// TIA Portal V17 export
// export: Created 2025-05-22T06:00:37.3823488Z, ExportSetting WithDefaults, DisplayName Totally Integrated Automation Portal, DisplayVersion V17 Update 8, DisplayName TIA Portal Openness, DisplayVersion V17 Update 8, DisplayName TIA Portal Version Control Interface, DisplayVersion V17, DisplayName SINAMICS Startdrive Advanced, DisplayVersion V17 SP2, DisplayName SINAMICS Startdrive G110M, G120, G120C, G120D, G120P, G115D, DisplayVersion V17 SP2, DisplayName SINAMICS Startdrive G130, G150, S120, S150, SINAMICS MV, S210, DisplayVersion V17 SP2, DisplayName STEP 7 Professional, DisplayVersion V17 Update 8, DisplayName SINUMERIK ONE STEP 7 Toolbox, DisplayVersion V17 Update 12, DisplayName SINUMERIK ONE PLC Basic Program Plus, DisplayVersion V17 Update 12, DisplayName SINUMERIK 840D sl STEP 7 Toolbox, DisplayVersion V17 Update 12, DisplayName STEP 7 Safety, DisplayVersion V17 Update 6, DisplayName WinCC Advanced, DisplayVersion V17 Update 8
FUNCTION "FC16011_METHOD_CALLS_U1_STA3_MEAS" : Void   // FC16011, LAD
{ S7_Optimized_Access := 'FALSE' }
VERSION : 0.1
// STATUS VALUES:
// 0 = IDLE
// 1 = CALIBRATING
// 2 = ANALYZING DISTANCE
// 3 = ANALYZING LAYER THICKNESS
// -1 = ERROR
// stored: AutoNumber false, IsIECCheckEnabled false, SetENOAutomatically false, UDAEnableTagReadback false
   VAR_TEMP
      AUX_WSTRING_PART_ID_STA3 : WString;
      AUX_WCHARS : Array[0..63] of WChar;
      index : Int;
      ALARM_AUX : Bool;
      STATUS_BLKMOV : Int;   // STATUS BLKMOV
      ZERO : Int;
   END_VAR
   VAR CONSTANT
      VERSIONS_MAJOR : UInt := 2;
      VERSIONS_MINOR : UInt;
      FC_NUMBER : DInt := 16011;
   END_VAR
   VAR_TEMP   // added for the SCL form of the ladder/FBD networks
      _w1 : Bool;
      _w2 : Bool;
      _w3 : Bool;
      _s5time1 : S5Time;
      _w4 : Bool;
   END_VAR
BEGIN

REGION Network 1: ZERO
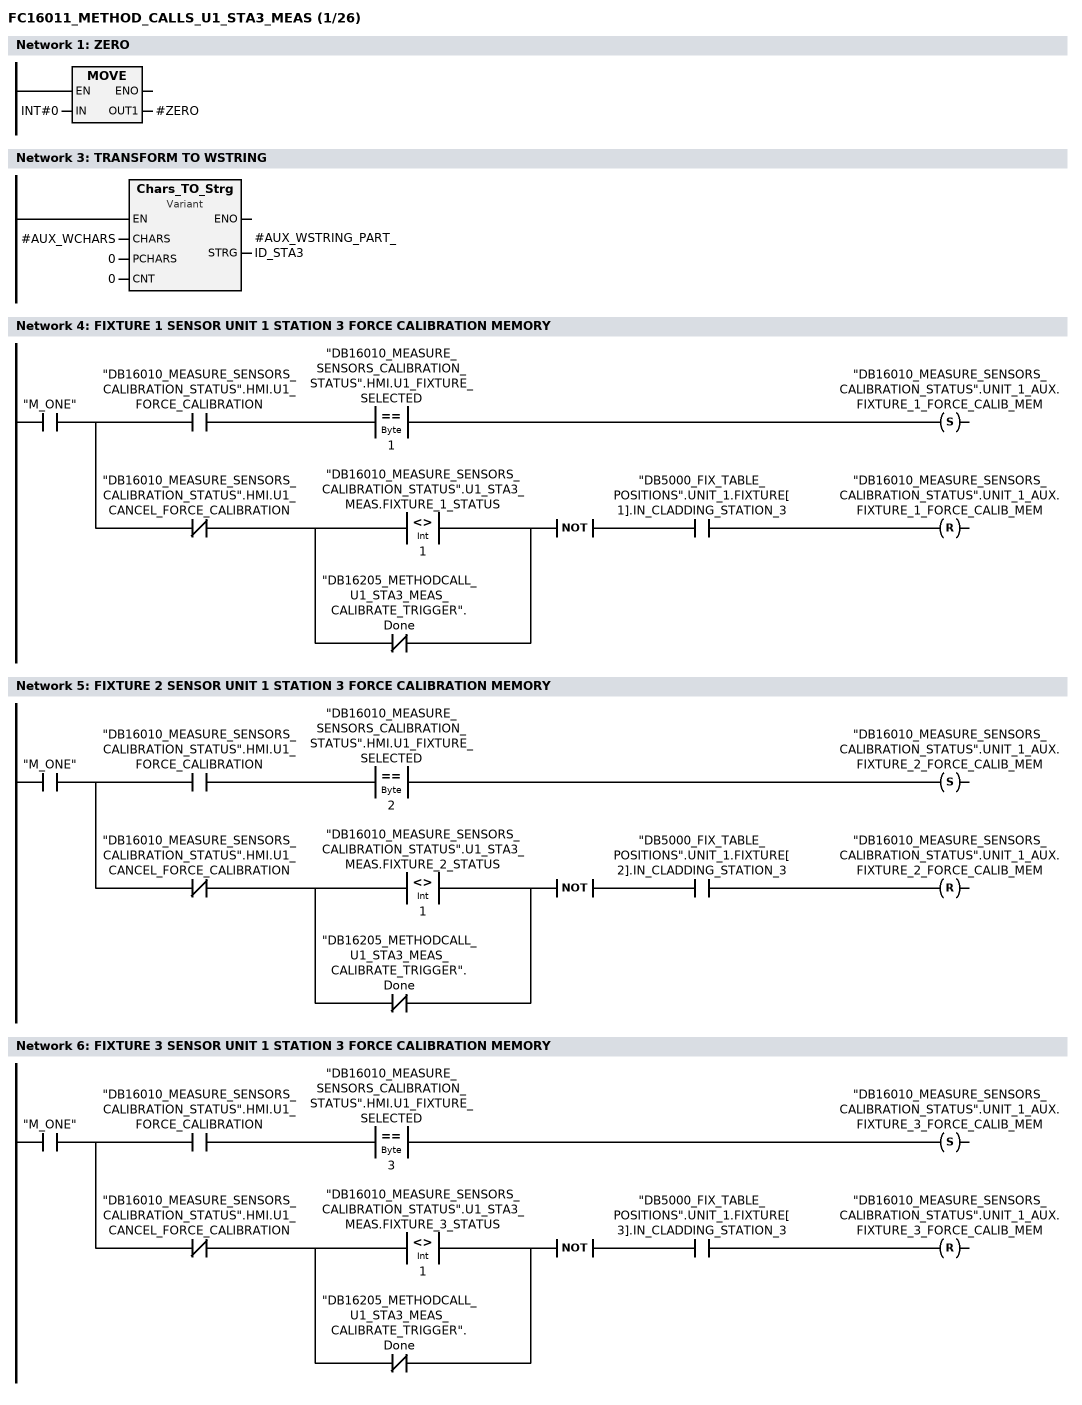
   RUNG wire#powerrail
      { S7_GenerateENO := "TRUE" } Move(in := INT#0, out1 => #ZERO)
   END_RUNG
   // the same network as SCL:
   #ZERO := INT#0;
END_REGION

REGION Network 2 (SCL): TRANSFORM TO WCHARS
   FOR #index := 0 TO 63 DO
       #AUX_WCHARS[#index] := CHAR_TO_WCHAR("DB8000_PART_STATUS".UNIT_1.STATION_3.PART_A.PART_ID[#index]);
   END_FOR;
END_REGION

REGION Network 3: TRANSFORM TO WSTRING
   RUNG wire#powerrail
      { S7_Templates := "[ptr_type := Variant, str_type := WString]" } Chars_TO_Strg(Chars := #AUX_WCHARS, pChars := 0, Cnt := 0, Strg => #AUX_WSTRING_PART_ID_STA3)
   END_RUNG
   // the same network as SCL:
   Chars_TO_Strg(Chars := #AUX_WCHARS, pChars := 0, Cnt := 0, Strg => #AUX_WSTRING_PART_ID_STA3);
END_REGION

REGION Network 4: FIXTURE 1 SENSOR UNIT 1 STATION 3 FORCE CALIBRATION MEMORY
   RUNG wire#powerrail
      Contact( "M_ONE" )
      wire#w1
      Contact( "DB16010_MEASURE_SENSORS_CALIBRATION_STATUS".HMI.U1_FORCE_CALIBRATION )
      { S7_Templates := "SrcType := Byte" } EQ_Contact(in1 := "DB16010_MEASURE_SENSORS_CALIBRATION_STATUS".HMI.U1_FIXTURE_SELECTED, in2 := 1)
      S_Coil( "DB16010_MEASURE_SENSORS_CALIBRATION_STATUS".UNIT_1_AUX.FIXTURE_1_FORCE_CALIB_MEM )
   END_RUNG
   RUNG wire#w1
      I_Contact( "DB16010_MEASURE_SENSORS_CALIBRATION_STATUS".HMI.U1_CANCEL_FORCE_CALIBRATION )
      wire#w2
      { S7_Templates := "SrcType := Int" } NE_Contact(in1 := "DB16010_MEASURE_SENSORS_CALIBRATION_STATUS".U1_STA3_MEAS.FIXTURE_1_STATUS, in2 := 1)
      wire#w3
      Not()
      Contact( "DB5000_FIX_TABLE_POSITIONS".UNIT_1.FIXTURE[1].IN_CLADDING_STATION_3 )
      R_Coil( "DB16010_MEASURE_SENSORS_CALIBRATION_STATUS".UNIT_1_AUX.FIXTURE_1_FORCE_CALIB_MEM )
   END_RUNG
   RUNG wire#w2
      I_Contact( "DB16205_METHODCALL_U1_STA3_MEAS_CALIBRATE_TRIGGER".Done )
   END_RUNG wire#w3
   // the same network as SCL:
   IF "M_ONE" AND "DB16010_MEASURE_SENSORS_CALIBRATION_STATUS".HMI.U1_FORCE_CALIBRATION AND ("DB16010_MEASURE_SENSORS_CALIBRATION_STATUS".HMI.U1_FIXTURE_SELECTED = 1) THEN
       "DB16010_MEASURE_SENSORS_CALIBRATION_STATUS".UNIT_1_AUX.FIXTURE_1_FORCE_CALIB_MEM := TRUE;
   END_IF;
   IF NOT ("M_ONE" AND NOT "DB16010_MEASURE_SENSORS_CALIBRATION_STATUS".HMI.U1_CANCEL_FORCE_CALIBRATION AND (("DB16010_MEASURE_SENSORS_CALIBRATION_STATUS".U1_STA3_MEAS.FIXTURE_1_STATUS <> 1) OR NOT "DB16205_METHODCALL_U1_STA3_MEAS_CALIBRATE_TRIGGER".Done)) AND "DB5000_FIX_TABLE_POSITIONS".UNIT_1.FIXTURE[1].IN_CLADDING_STATION_3 THEN
       "DB16010_MEASURE_SENSORS_CALIBRATION_STATUS".UNIT_1_AUX.FIXTURE_1_FORCE_CALIB_MEM := FALSE;
   END_IF;
END_REGION

REGION Network 5: FIXTURE 2 SENSOR UNIT 1 STATION 3 FORCE CALIBRATION MEMORY
   RUNG wire#powerrail
      Contact( "M_ONE" )
      wire#w1
      Contact( "DB16010_MEASURE_SENSORS_CALIBRATION_STATUS".HMI.U1_FORCE_CALIBRATION )
      { S7_Templates := "SrcType := Byte" } EQ_Contact(in1 := "DB16010_MEASURE_SENSORS_CALIBRATION_STATUS".HMI.U1_FIXTURE_SELECTED, in2 := 2)
      S_Coil( "DB16010_MEASURE_SENSORS_CALIBRATION_STATUS".UNIT_1_AUX.FIXTURE_2_FORCE_CALIB_MEM )
   END_RUNG
   RUNG wire#w1
      I_Contact( "DB16010_MEASURE_SENSORS_CALIBRATION_STATUS".HMI.U1_CANCEL_FORCE_CALIBRATION )
      wire#w2
      { S7_Templates := "SrcType := Int" } NE_Contact(in1 := "DB16010_MEASURE_SENSORS_CALIBRATION_STATUS".U1_STA3_MEAS.FIXTURE_2_STATUS, in2 := 1)
      wire#w3
      Not()
      Contact( "DB5000_FIX_TABLE_POSITIONS".UNIT_1.FIXTURE[2].IN_CLADDING_STATION_3 )
      R_Coil( "DB16010_MEASURE_SENSORS_CALIBRATION_STATUS".UNIT_1_AUX.FIXTURE_2_FORCE_CALIB_MEM )
   END_RUNG
   RUNG wire#w2
      I_Contact( "DB16205_METHODCALL_U1_STA3_MEAS_CALIBRATE_TRIGGER".Done )
   END_RUNG wire#w3
   // the same network as SCL:
   IF "M_ONE" AND "DB16010_MEASURE_SENSORS_CALIBRATION_STATUS".HMI.U1_FORCE_CALIBRATION AND ("DB16010_MEASURE_SENSORS_CALIBRATION_STATUS".HMI.U1_FIXTURE_SELECTED = 2) THEN
       "DB16010_MEASURE_SENSORS_CALIBRATION_STATUS".UNIT_1_AUX.FIXTURE_2_FORCE_CALIB_MEM := TRUE;
   END_IF;
   IF NOT ("M_ONE" AND NOT "DB16010_MEASURE_SENSORS_CALIBRATION_STATUS".HMI.U1_CANCEL_FORCE_CALIBRATION AND (("DB16010_MEASURE_SENSORS_CALIBRATION_STATUS".U1_STA3_MEAS.FIXTURE_2_STATUS <> 1) OR NOT "DB16205_METHODCALL_U1_STA3_MEAS_CALIBRATE_TRIGGER".Done)) AND "DB5000_FIX_TABLE_POSITIONS".UNIT_1.FIXTURE[2].IN_CLADDING_STATION_3 THEN
       "DB16010_MEASURE_SENSORS_CALIBRATION_STATUS".UNIT_1_AUX.FIXTURE_2_FORCE_CALIB_MEM := FALSE;
   END_IF;
END_REGION

REGION Network 6: FIXTURE 3 SENSOR UNIT 1 STATION 3 FORCE CALIBRATION MEMORY
   RUNG wire#powerrail
      Contact( "M_ONE" )
      wire#w1
      Contact( "DB16010_MEASURE_SENSORS_CALIBRATION_STATUS".HMI.U1_FORCE_CALIBRATION )
      { S7_Templates := "SrcType := Byte" } EQ_Contact(in1 := "DB16010_MEASURE_SENSORS_CALIBRATION_STATUS".HMI.U1_FIXTURE_SELECTED, in2 := 3)
      S_Coil( "DB16010_MEASURE_SENSORS_CALIBRATION_STATUS".UNIT_1_AUX.FIXTURE_3_FORCE_CALIB_MEM )
   END_RUNG
   RUNG wire#w1
      I_Contact( "DB16010_MEASURE_SENSORS_CALIBRATION_STATUS".HMI.U1_CANCEL_FORCE_CALIBRATION )
      wire#w2
      { S7_Templates := "SrcType := Int" } NE_Contact(in1 := "DB16010_MEASURE_SENSORS_CALIBRATION_STATUS".U1_STA3_MEAS.FIXTURE_3_STATUS, in2 := 1)
      wire#w3
      Not()
      Contact( "DB5000_FIX_TABLE_POSITIONS".UNIT_1.FIXTURE[3].IN_CLADDING_STATION_3 )
      R_Coil( "DB16010_MEASURE_SENSORS_CALIBRATION_STATUS".UNIT_1_AUX.FIXTURE_3_FORCE_CALIB_MEM )
   END_RUNG
   RUNG wire#w2
      I_Contact( "DB16205_METHODCALL_U1_STA3_MEAS_CALIBRATE_TRIGGER".Done )
   END_RUNG wire#w3
   // the same network as SCL:
   IF "M_ONE" AND "DB16010_MEASURE_SENSORS_CALIBRATION_STATUS".HMI.U1_FORCE_CALIBRATION AND ("DB16010_MEASURE_SENSORS_CALIBRATION_STATUS".HMI.U1_FIXTURE_SELECTED = 3) THEN
       "DB16010_MEASURE_SENSORS_CALIBRATION_STATUS".UNIT_1_AUX.FIXTURE_3_FORCE_CALIB_MEM := TRUE;
   END_IF;
   IF NOT ("M_ONE" AND NOT "DB16010_MEASURE_SENSORS_CALIBRATION_STATUS".HMI.U1_CANCEL_FORCE_CALIBRATION AND (("DB16010_MEASURE_SENSORS_CALIBRATION_STATUS".U1_STA3_MEAS.FIXTURE_3_STATUS <> 1) OR NOT "DB16205_METHODCALL_U1_STA3_MEAS_CALIBRATE_TRIGGER".Done)) AND "DB5000_FIX_TABLE_POSITIONS".UNIT_1.FIXTURE[3].IN_CLADDING_STATION_3 THEN
       "DB16010_MEASURE_SENSORS_CALIBRATION_STATUS".UNIT_1_AUX.FIXTURE_3_FORCE_CALIB_MEM := FALSE;
   END_IF;
END_REGION

REGION Network 7: FIXTURE 4 SENSOR UNIT 1 STATION 3 FORCE CALIBRATION MEMORY
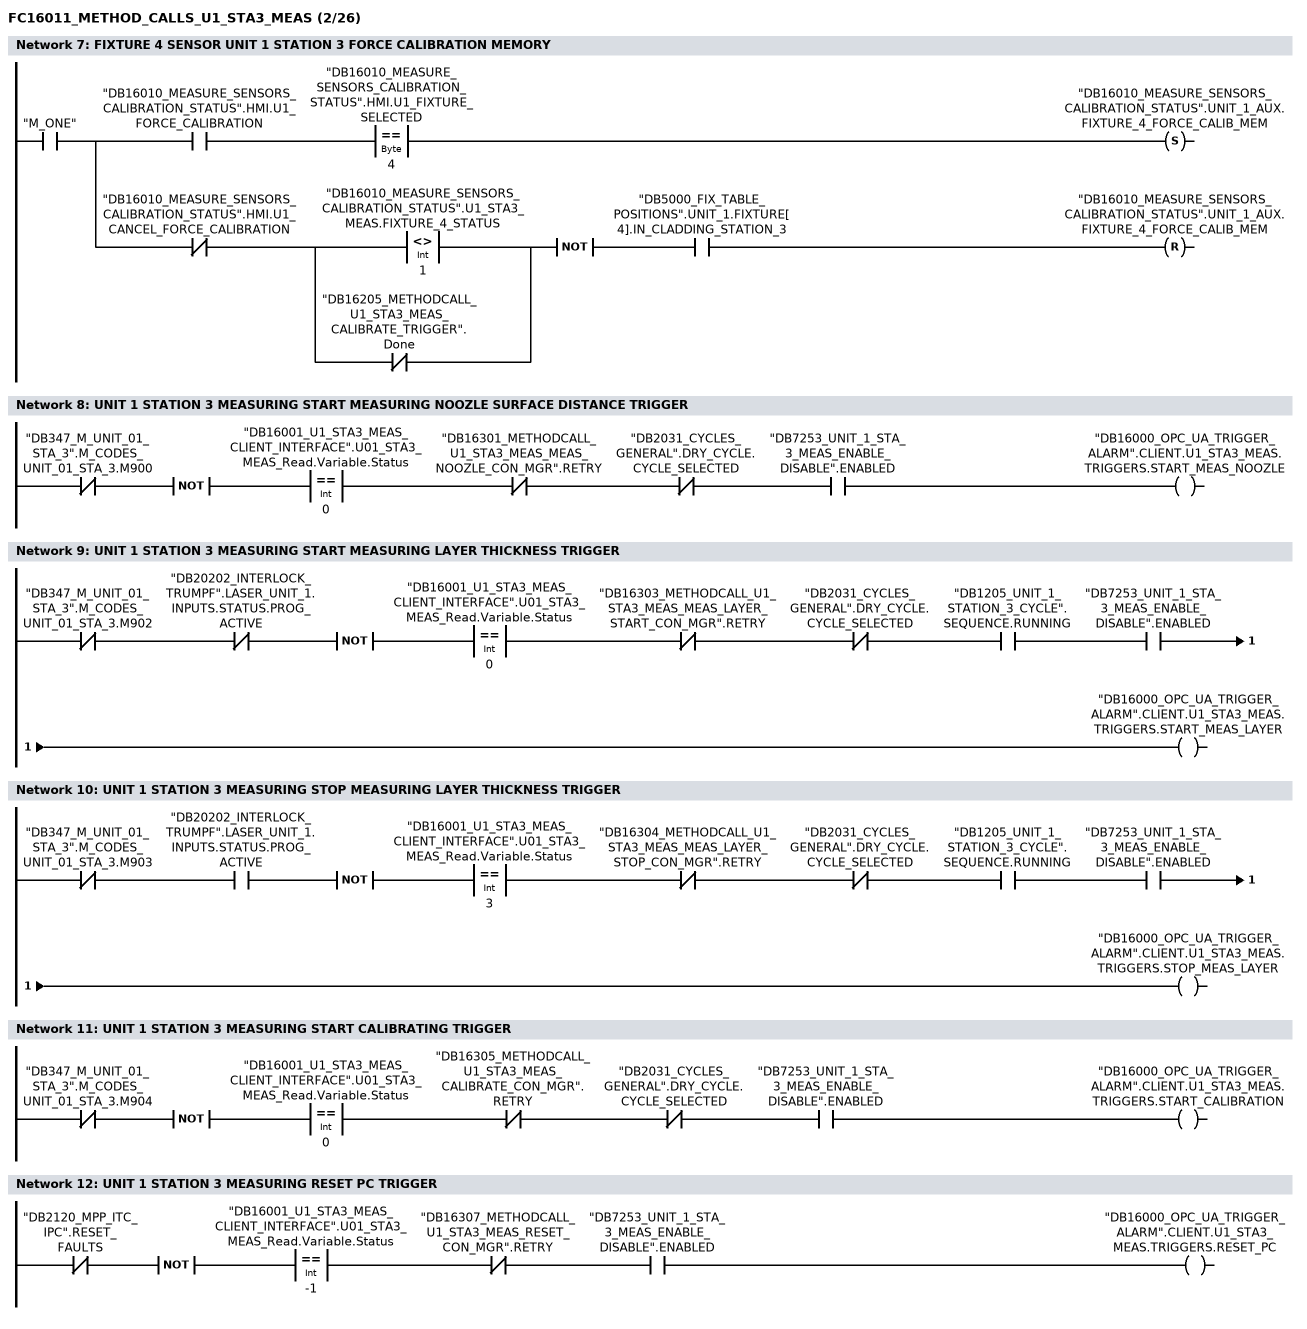
   RUNG wire#powerrail
      Contact( "M_ONE" )
      wire#w1
      Contact( "DB16010_MEASURE_SENSORS_CALIBRATION_STATUS".HMI.U1_FORCE_CALIBRATION )
      { S7_Templates := "SrcType := Byte" } EQ_Contact(in1 := "DB16010_MEASURE_SENSORS_CALIBRATION_STATUS".HMI.U1_FIXTURE_SELECTED, in2 := 4)
      S_Coil( "DB16010_MEASURE_SENSORS_CALIBRATION_STATUS".UNIT_1_AUX.FIXTURE_4_FORCE_CALIB_MEM )
   END_RUNG
   RUNG wire#w1
      I_Contact( "DB16010_MEASURE_SENSORS_CALIBRATION_STATUS".HMI.U1_CANCEL_FORCE_CALIBRATION )
      wire#w2
      { S7_Templates := "SrcType := Int" } NE_Contact(in1 := "DB16010_MEASURE_SENSORS_CALIBRATION_STATUS".U1_STA3_MEAS.FIXTURE_4_STATUS, in2 := 1)
      wire#w3
      Not()
      Contact( "DB5000_FIX_TABLE_POSITIONS".UNIT_1.FIXTURE[4].IN_CLADDING_STATION_3 )
      R_Coil( "DB16010_MEASURE_SENSORS_CALIBRATION_STATUS".UNIT_1_AUX.FIXTURE_4_FORCE_CALIB_MEM )
   END_RUNG
   RUNG wire#w2
      I_Contact( "DB16205_METHODCALL_U1_STA3_MEAS_CALIBRATE_TRIGGER".Done )
   END_RUNG wire#w3
   // the same network as SCL:
   IF "M_ONE" AND "DB16010_MEASURE_SENSORS_CALIBRATION_STATUS".HMI.U1_FORCE_CALIBRATION AND ("DB16010_MEASURE_SENSORS_CALIBRATION_STATUS".HMI.U1_FIXTURE_SELECTED = 4) THEN
       "DB16010_MEASURE_SENSORS_CALIBRATION_STATUS".UNIT_1_AUX.FIXTURE_4_FORCE_CALIB_MEM := TRUE;
   END_IF;
   IF NOT ("M_ONE" AND NOT "DB16010_MEASURE_SENSORS_CALIBRATION_STATUS".HMI.U1_CANCEL_FORCE_CALIBRATION AND (("DB16010_MEASURE_SENSORS_CALIBRATION_STATUS".U1_STA3_MEAS.FIXTURE_4_STATUS <> 1) OR NOT "DB16205_METHODCALL_U1_STA3_MEAS_CALIBRATE_TRIGGER".Done)) AND "DB5000_FIX_TABLE_POSITIONS".UNIT_1.FIXTURE[4].IN_CLADDING_STATION_3 THEN
       "DB16010_MEASURE_SENSORS_CALIBRATION_STATUS".UNIT_1_AUX.FIXTURE_4_FORCE_CALIB_MEM := FALSE;
   END_IF;
END_REGION

REGION Network 8: UNIT 1 STATION 3 MEASURING START MEASURING NOOZLE SURFACE DISTANCE TRIGGER
   RUNG wire#powerrail
      I_Contact( "DB347_M_UNIT_01_STA_3".M_CODES_UNIT_01_STA_3.M900 )
      Not()
      { S7_Templates := "SrcType := Int" } EQ_Contact(in1 := "DB16001_U1_STA3_MEAS_CLIENT_INTERFACE".U01_STA3_MEAS_Read.Variable.Status, in2 := 0)
      I_Contact( "DB16301_METHODCALL_U1_STA3_MEAS_MEAS_NOOZLE_CON_MGR".RETRY )
      I_Contact( "DB2031_CYCLES_GENERAL".DRY_CYCLE.CYCLE_SELECTED )
      Contact( "DB7253_UNIT_1_STA_3_MEAS_ENABLE_DISABLE".ENABLED )
      Coil( "DB16000_OPC_UA_TRIGGER_ALARM".CLIENT.U1_STA3_MEAS.TRIGGERS.START_MEAS_NOOZLE )
   END_RUNG
   // the same network as SCL:
   "DB16000_OPC_UA_TRIGGER_ALARM".CLIENT.U1_STA3_MEAS.TRIGGERS.START_MEAS_NOOZLE := NOT (NOT "DB347_M_UNIT_01_STA_3".M_CODES_UNIT_01_STA_3.M900) AND ("DB16001_U1_STA3_MEAS_CLIENT_INTERFACE".U01_STA3_MEAS_Read.Variable.Status = 0) AND NOT "DB16301_METHODCALL_U1_STA3_MEAS_MEAS_NOOZLE_CON_MGR".RETRY AND NOT "DB2031_CYCLES_GENERAL".DRY_CYCLE.CYCLE_SELECTED AND "DB7253_UNIT_1_STA_3_MEAS_ENABLE_DISABLE".ENABLED;
END_REGION

REGION Network 9: UNIT 1 STATION 3 MEASURING START MEASURING LAYER THICKNESS TRIGGER
   RUNG wire#powerrail
      I_Contact( "DB347_M_UNIT_01_STA_3".M_CODES_UNIT_01_STA_3.M902 )
      I_Contact( "DB20202_INTERLOCK_TRUMPF".LASER_UNIT_1.INPUTS.STATUS.PROG_ACTIVE )
      Not()
      { S7_Templates := "SrcType := Int" } EQ_Contact(in1 := "DB16001_U1_STA3_MEAS_CLIENT_INTERFACE".U01_STA3_MEAS_Read.Variable.Status, in2 := 0)
      I_Contact( "DB16303_METHODCALL_U1_STA3_MEAS_MEAS_LAYER_START_CON_MGR".RETRY )
      I_Contact( "DB2031_CYCLES_GENERAL".DRY_CYCLE.CYCLE_SELECTED )
      Contact( "DB1205_UNIT_1_STATION_3_CYCLE".SEQUENCE.RUNNING )
      Contact( "DB7253_UNIT_1_STA_3_MEAS_ENABLE_DISABLE".ENABLED )
      Coil( "DB16000_OPC_UA_TRIGGER_ALARM".CLIENT.U1_STA3_MEAS.TRIGGERS.START_MEAS_LAYER )
   END_RUNG
   // the same network as SCL:
   "DB16000_OPC_UA_TRIGGER_ALARM".CLIENT.U1_STA3_MEAS.TRIGGERS.START_MEAS_LAYER := NOT (NOT "DB347_M_UNIT_01_STA_3".M_CODES_UNIT_01_STA_3.M902 AND NOT "DB20202_INTERLOCK_TRUMPF".LASER_UNIT_1.INPUTS.STATUS.PROG_ACTIVE) AND ("DB16001_U1_STA3_MEAS_CLIENT_INTERFACE".U01_STA3_MEAS_Read.Variable.Status = 0) AND NOT "DB16303_METHODCALL_U1_STA3_MEAS_MEAS_LAYER_START_CON_MGR".RETRY AND NOT "DB2031_CYCLES_GENERAL".DRY_CYCLE.CYCLE_SELECTED AND "DB1205_UNIT_1_STATION_3_CYCLE".SEQUENCE.RUNNING AND "DB7253_UNIT_1_STA_3_MEAS_ENABLE_DISABLE".ENABLED;
END_REGION

REGION Network 10: UNIT 1 STATION 3 MEASURING STOP MEASURING LAYER THICKNESS TRIGGER
   RUNG wire#powerrail
      I_Contact( "DB347_M_UNIT_01_STA_3".M_CODES_UNIT_01_STA_3.M903 )
      Contact( "DB20202_INTERLOCK_TRUMPF".LASER_UNIT_1.INPUTS.STATUS.PROG_ACTIVE )
      Not()
      { S7_Templates := "SrcType := Int" } EQ_Contact(in1 := "DB16001_U1_STA3_MEAS_CLIENT_INTERFACE".U01_STA3_MEAS_Read.Variable.Status, in2 := 3)
      I_Contact( "DB16304_METHODCALL_U1_STA3_MEAS_MEAS_LAYER_STOP_CON_MGR".RETRY )
      I_Contact( "DB2031_CYCLES_GENERAL".DRY_CYCLE.CYCLE_SELECTED )
      Contact( "DB1205_UNIT_1_STATION_3_CYCLE".SEQUENCE.RUNNING )
      Contact( "DB7253_UNIT_1_STA_3_MEAS_ENABLE_DISABLE".ENABLED )
      Coil( "DB16000_OPC_UA_TRIGGER_ALARM".CLIENT.U1_STA3_MEAS.TRIGGERS.STOP_MEAS_LAYER )
   END_RUNG
   // the same network as SCL:
   "DB16000_OPC_UA_TRIGGER_ALARM".CLIENT.U1_STA3_MEAS.TRIGGERS.STOP_MEAS_LAYER := NOT (NOT "DB347_M_UNIT_01_STA_3".M_CODES_UNIT_01_STA_3.M903 AND "DB20202_INTERLOCK_TRUMPF".LASER_UNIT_1.INPUTS.STATUS.PROG_ACTIVE) AND ("DB16001_U1_STA3_MEAS_CLIENT_INTERFACE".U01_STA3_MEAS_Read.Variable.Status = 3) AND NOT "DB16304_METHODCALL_U1_STA3_MEAS_MEAS_LAYER_STOP_CON_MGR".RETRY AND NOT "DB2031_CYCLES_GENERAL".DRY_CYCLE.CYCLE_SELECTED AND "DB1205_UNIT_1_STATION_3_CYCLE".SEQUENCE.RUNNING AND "DB7253_UNIT_1_STA_3_MEAS_ENABLE_DISABLE".ENABLED;
END_REGION

REGION Network 11: UNIT 1 STATION 3 MEASURING START CALIBRATING TRIGGER
   RUNG wire#powerrail
      I_Contact( "DB347_M_UNIT_01_STA_3".M_CODES_UNIT_01_STA_3.M904 )
      Not()
      { S7_Templates := "SrcType := Int" } EQ_Contact(in1 := "DB16001_U1_STA3_MEAS_CLIENT_INTERFACE".U01_STA3_MEAS_Read.Variable.Status, in2 := 0)
      I_Contact( "DB16305_METHODCALL_U1_STA3_MEAS_CALIBRATE_CON_MGR".RETRY )
      I_Contact( "DB2031_CYCLES_GENERAL".DRY_CYCLE.CYCLE_SELECTED )
      Contact( "DB7253_UNIT_1_STA_3_MEAS_ENABLE_DISABLE".ENABLED )
      Coil( "DB16000_OPC_UA_TRIGGER_ALARM".CLIENT.U1_STA3_MEAS.TRIGGERS.START_CALIBRATION )
   END_RUNG
   // the same network as SCL:
   "DB16000_OPC_UA_TRIGGER_ALARM".CLIENT.U1_STA3_MEAS.TRIGGERS.START_CALIBRATION := NOT (NOT "DB347_M_UNIT_01_STA_3".M_CODES_UNIT_01_STA_3.M904) AND ("DB16001_U1_STA3_MEAS_CLIENT_INTERFACE".U01_STA3_MEAS_Read.Variable.Status = 0) AND NOT "DB16305_METHODCALL_U1_STA3_MEAS_CALIBRATE_CON_MGR".RETRY AND NOT "DB2031_CYCLES_GENERAL".DRY_CYCLE.CYCLE_SELECTED AND "DB7253_UNIT_1_STA_3_MEAS_ENABLE_DISABLE".ENABLED;
END_REGION

REGION Network 12: UNIT 1 STATION 3 MEASURING RESET PC TRIGGER
   RUNG wire#powerrail
      I_Contact( "DB2120_MPP_ITC_IPC".RESET_FAULTS )
      Not()
      { S7_Templates := "SrcType := Int" } EQ_Contact(in1 := "DB16001_U1_STA3_MEAS_CLIENT_INTERFACE".U01_STA3_MEAS_Read.Variable.Status, in2 := -1)
      I_Contact( "DB16307_METHODCALL_U1_STA3_MEAS_RESET_CON_MGR".RETRY )
      Contact( "DB7253_UNIT_1_STA_3_MEAS_ENABLE_DISABLE".ENABLED )
      Coil( "DB16000_OPC_UA_TRIGGER_ALARM".CLIENT.U1_STA3_MEAS.TRIGGERS.RESET_PC )
   END_RUNG
   // the same network as SCL:
   "DB16000_OPC_UA_TRIGGER_ALARM".CLIENT.U1_STA3_MEAS.TRIGGERS.RESET_PC := NOT (NOT "DB2120_MPP_ITC_IPC".RESET_FAULTS) AND ("DB16001_U1_STA3_MEAS_CLIENT_INTERFACE".U01_STA3_MEAS_Read.Variable.Status = (-1)) AND NOT "DB16307_METHODCALL_U1_STA3_MEAS_RESET_CON_MGR".RETRY AND "DB7253_UNIT_1_STA_3_MEAS_ENABLE_DISABLE".ENABLED;
END_REGION

REGION Network 13: UNIT 1 STATION 3 MEASURING READ VARIABLES TRIGGER
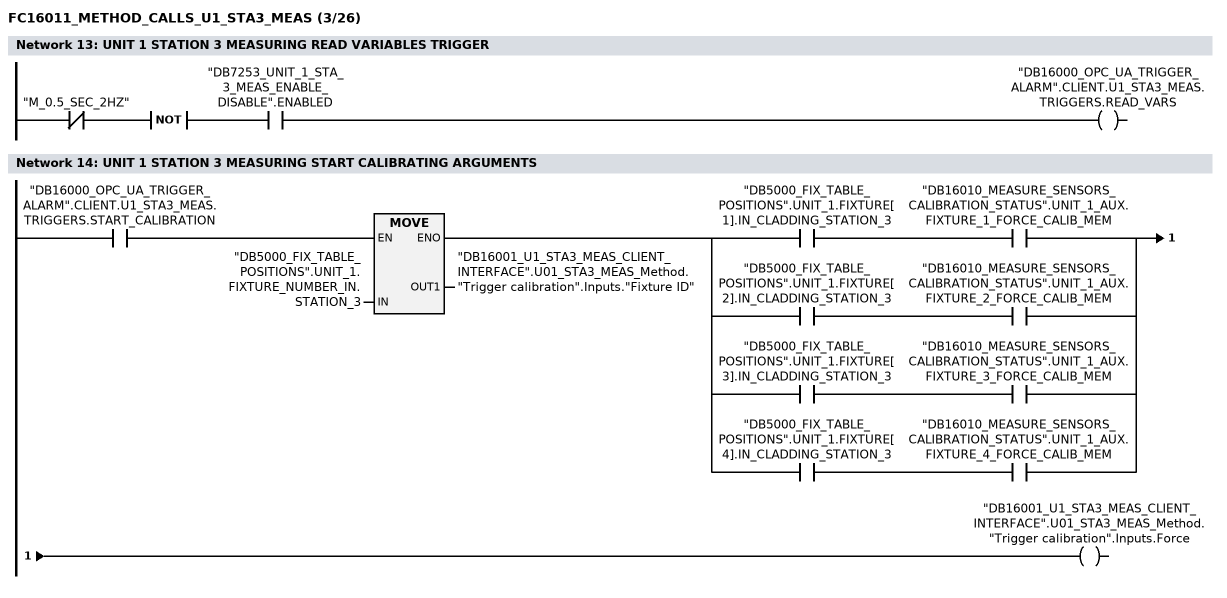
   RUNG wire#powerrail
      I_Contact( "M_0.5_SEC_2HZ" )
      Not()
      Contact( "DB7253_UNIT_1_STA_3_MEAS_ENABLE_DISABLE".ENABLED )
      Coil( "DB16000_OPC_UA_TRIGGER_ALARM".CLIENT.U1_STA3_MEAS.TRIGGERS.READ_VARS )
   END_RUNG
   // the same network as SCL:
   "DB16000_OPC_UA_TRIGGER_ALARM".CLIENT.U1_STA3_MEAS.TRIGGERS.READ_VARS := NOT (NOT "M_0.5_SEC_2HZ") AND "DB7253_UNIT_1_STA_3_MEAS_ENABLE_DISABLE".ENABLED;
END_REGION

REGION Network 14: UNIT 1 STATION 3 MEASURING START CALIBRATING ARGUMENTS
   RUNG wire#powerrail
      Contact( "DB16000_OPC_UA_TRIGGER_ALARM".CLIENT.U1_STA3_MEAS.TRIGGERS.START_CALIBRATION )
      Move(in := "DB5000_FIX_TABLE_POSITIONS".UNIT_1.FIXTURE_NUMBER_IN.STATION_3, out1 => "DB16001_U1_STA3_MEAS_CLIENT_INTERFACE".U01_STA3_MEAS_Method."Trigger calibration".Inputs."Fixture ID")
      wire#w1
      Contact( "DB5000_FIX_TABLE_POSITIONS".UNIT_1.FIXTURE[1].IN_CLADDING_STATION_3 )
      Contact( "DB16010_MEASURE_SENSORS_CALIBRATION_STATUS".UNIT_1_AUX.FIXTURE_1_FORCE_CALIB_MEM )
      wire#w2
      Coil( "DB16001_U1_STA3_MEAS_CLIENT_INTERFACE".U01_STA3_MEAS_Method."Trigger calibration".Inputs.Force )
   END_RUNG
   RUNG wire#w1
      Contact( "DB5000_FIX_TABLE_POSITIONS".UNIT_1.FIXTURE[2].IN_CLADDING_STATION_3 )
      Contact( "DB16010_MEASURE_SENSORS_CALIBRATION_STATUS".UNIT_1_AUX.FIXTURE_2_FORCE_CALIB_MEM )
   END_RUNG wire#w2
   RUNG wire#w1
      Contact( "DB5000_FIX_TABLE_POSITIONS".UNIT_1.FIXTURE[3].IN_CLADDING_STATION_3 )
      Contact( "DB16010_MEASURE_SENSORS_CALIBRATION_STATUS".UNIT_1_AUX.FIXTURE_3_FORCE_CALIB_MEM )
   END_RUNG wire#w2
   RUNG wire#w1
      Contact( "DB5000_FIX_TABLE_POSITIONS".UNIT_1.FIXTURE[4].IN_CLADDING_STATION_3 )
      Contact( "DB16010_MEASURE_SENSORS_CALIBRATION_STATUS".UNIT_1_AUX.FIXTURE_4_FORCE_CALIB_MEM )
   END_RUNG wire#w2
   // the same network as SCL:
   IF "DB16000_OPC_UA_TRIGGER_ALARM".CLIENT.U1_STA3_MEAS.TRIGGERS.START_CALIBRATION THEN
       "DB16001_U1_STA3_MEAS_CLIENT_INTERFACE".U01_STA3_MEAS_Method."Trigger calibration".Inputs."Fixture ID" := "DB5000_FIX_TABLE_POSITIONS".UNIT_1.FIXTURE_NUMBER_IN.STATION_3;
   END_IF;
   "DB16001_U1_STA3_MEAS_CLIENT_INTERFACE".U01_STA3_MEAS_Method."Trigger calibration".Inputs.Force := "DB16000_OPC_UA_TRIGGER_ALARM".CLIENT.U1_STA3_MEAS.TRIGGERS.START_CALIBRATION AND (("DB5000_FIX_TABLE_POSITIONS".UNIT_1.FIXTURE[1].IN_CLADDING_STATION_3 AND "DB16010_MEASURE_SENSORS_CALIBRATION_STATUS".UNIT_1_AUX.FIXTURE_1_FORCE_CALIB_MEM) OR ("DB5000_FIX_TABLE_POSITIONS".UNIT_1.FIXTURE[2].IN_CLADDING_STATION_3 AND "DB16010_MEASURE_SENSORS_CALIBRATION_STATUS".UNIT_1_AUX.FIXTURE_2_FORCE_CALIB_MEM) OR ("DB5000_FIX_TABLE_POSITIONS".UNIT_1.FIXTURE[3].IN_CLADDING_STATION_3 AND "DB16010_MEASURE_SENSORS_CALIBRATION_STATUS".UNIT_1_AUX.FIXTURE_3_FORCE_CALIB_MEM) OR ("DB5000_FIX_TABLE_POSITIONS".UNIT_1.FIXTURE[4].IN_CLADDING_STATION_3 AND "DB16010_MEASURE_SENSORS_CALIBRATION_STATUS".UNIT_1_AUX.FIXTURE_4_FORCE_CALIB_MEM));
END_REGION

REGION Network 15: UNIT 1 STATION 3 MEASURING START MEASURING NOOZLE SURFACE DISTANCE TRIGGER CALL
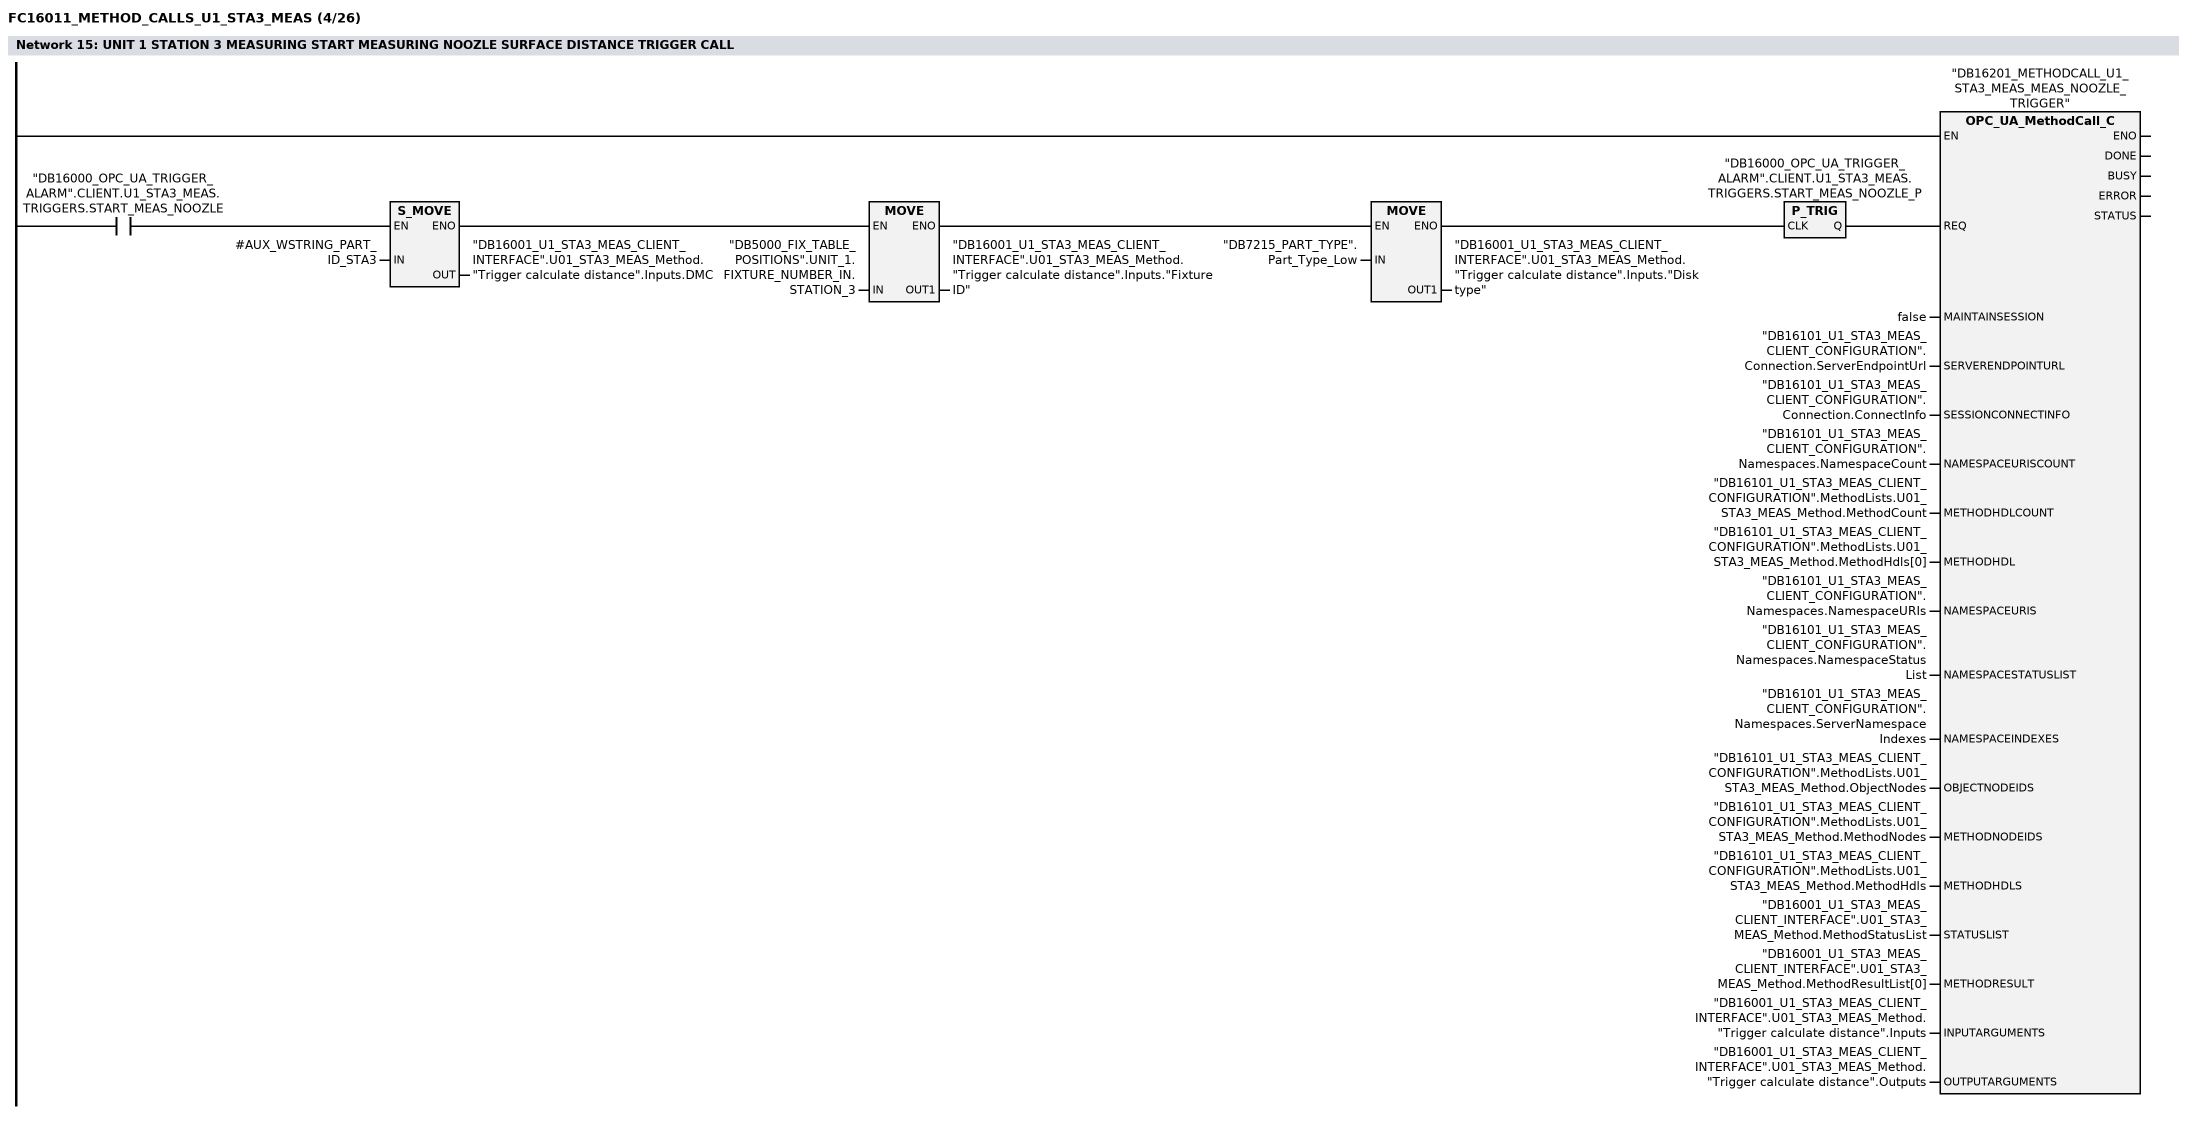
   RUNG wire#powerrail
      "DB16201_METHODCALL_U1_STA3_MEAS_MEAS_NOOZLE_TRIGGER".OPC_UA_MethodCall_C(REQ := wire#w1, MaintainSession := false, ServerEndpointUrl := "DB16101_U1_STA3_MEAS_CLIENT_CONFIGURATION".Connection.ServerEndpointUrl, SessionConnectInfo := "DB16101_U1_STA3_MEAS_CLIENT_CONFIGURATION".Connection.ConnectInfo, NamespaceUrisCount := "DB16101_U1_STA3_MEAS_CLIENT_CONFIGURATION".Namespaces.NamespaceCount, MethodHdlCount := "DB16101_U1_STA3_MEAS_CLIENT_CONFIGURATION".MethodLists.U01_STA3_MEAS_Method.MethodCount, MethodHdl := "DB16101_U1_STA3_MEAS_CLIENT_CONFIGURATION".MethodLists.U01_STA3_MEAS_Method.MethodHdls[0], NamespaceUris := "DB16101_U1_STA3_MEAS_CLIENT_CONFIGURATION".Namespaces.NamespaceURIs, NamespaceStatusList := "DB16101_U1_STA3_MEAS_CLIENT_CONFIGURATION".Namespaces.NamespaceStatusList, NamespaceIndexes := "DB16101_U1_STA3_MEAS_CLIENT_CONFIGURATION".Namespaces.ServerNamespaceIndexes, ObjectNodeIDs := "DB16101_U1_STA3_MEAS_CLIENT_CONFIGURATION".MethodLists.U01_STA3_MEAS_Method.ObjectNodes, MethodNodeIDs := "DB16101_U1_STA3_MEAS_CLIENT_CONFIGURATION".MethodLists.U01_STA3_MEAS_Method.MethodNodes, MethodHdls := "DB16101_U1_STA3_MEAS_CLIENT_CONFIGURATION".MethodLists.U01_STA3_MEAS_Method.MethodHdls, StatusList := "DB16001_U1_STA3_MEAS_CLIENT_INTERFACE".U01_STA3_MEAS_Method.MethodStatusList, MethodResult := "DB16001_U1_STA3_MEAS_CLIENT_INTERFACE".U01_STA3_MEAS_Method.MethodResultList[0], InputArguments := "DB16001_U1_STA3_MEAS_CLIENT_INTERFACE".U01_STA3_MEAS_Method."Trigger calculate distance".Inputs, OutputArguments := "DB16001_U1_STA3_MEAS_CLIENT_INTERFACE".U01_STA3_MEAS_Method."Trigger calculate distance".Outputs, Done =>, Busy =>, Error =>, Status =>)
   END_RUNG
   RUNG wire#powerrail
      Contact( "DB16000_OPC_UA_TRIGGER_ALARM".CLIENT.U1_STA3_MEAS.TRIGGERS.START_MEAS_NOOZLE )
      S_Move(in := #AUX_WSTRING_PART_ID_STA3, out => "DB16001_U1_STA3_MEAS_CLIENT_INTERFACE".U01_STA3_MEAS_Method."Trigger calculate distance".Inputs.DMC)
      Move(in := "DB5000_FIX_TABLE_POSITIONS".UNIT_1.FIXTURE_NUMBER_IN.STATION_3, out1 => "DB16001_U1_STA3_MEAS_CLIENT_INTERFACE".U01_STA3_MEAS_Method."Trigger calculate distance".Inputs."Fixture ID")
      Move(in := "DB7215_PART_TYPE".Part_Type_Low, out1 => "DB16001_U1_STA3_MEAS_CLIENT_INTERFACE".U01_STA3_MEAS_Method."Trigger calculate distance".Inputs."Disk type")
      P_Trig( "DB16000_OPC_UA_TRIGGER_ALARM".CLIENT.U1_STA3_MEAS.TRIGGERS.START_MEAS_NOOZLE_P )
   END_RUNG wire#w1
   // the same network as SCL:
   IF "DB16000_OPC_UA_TRIGGER_ALARM".CLIENT.U1_STA3_MEAS.TRIGGERS.START_MEAS_NOOZLE THEN
       "DB16001_U1_STA3_MEAS_CLIENT_INTERFACE".U01_STA3_MEAS_Method."Trigger calculate distance".Inputs.DMC := #AUX_WSTRING_PART_ID_STA3;
       "DB16001_U1_STA3_MEAS_CLIENT_INTERFACE".U01_STA3_MEAS_Method."Trigger calculate distance".Inputs."Fixture ID" := "DB5000_FIX_TABLE_POSITIONS".UNIT_1.FIXTURE_NUMBER_IN.STATION_3;
       "DB16001_U1_STA3_MEAS_CLIENT_INTERFACE".U01_STA3_MEAS_Method."Trigger calculate distance".Inputs."Disk type" := "DB7215_PART_TYPE".Part_Type_Low;
   END_IF;
   #_w1 := "DB16000_OPC_UA_TRIGGER_ALARM".CLIENT.U1_STA3_MEAS.TRIGGERS.START_MEAS_NOOZLE AND NOT "DB16000_OPC_UA_TRIGGER_ALARM".CLIENT.U1_STA3_MEAS.TRIGGERS.START_MEAS_NOOZLE_P;   // rising edge
   "DB16000_OPC_UA_TRIGGER_ALARM".CLIENT.U1_STA3_MEAS.TRIGGERS.START_MEAS_NOOZLE_P := "DB16000_OPC_UA_TRIGGER_ALARM".CLIENT.U1_STA3_MEAS.TRIGGERS.START_MEAS_NOOZLE;
   "DB16201_METHODCALL_U1_STA3_MEAS_MEAS_NOOZLE_TRIGGER"(REQ := #_w1,   // OPC_UA_MethodCall_C
                           MaintainSession := false,
                           ServerEndpointUrl := "DB16101_U1_STA3_MEAS_CLIENT_CONFIGURATION".Connection.ServerEndpointUrl,
                           SessionConnectInfo := "DB16101_U1_STA3_MEAS_CLIENT_CONFIGURATION".Connection.ConnectInfo,
                           NamespaceUrisCount := "DB16101_U1_STA3_MEAS_CLIENT_CONFIGURATION".Namespaces.NamespaceCount,
                           MethodHdlCount := "DB16101_U1_STA3_MEAS_CLIENT_CONFIGURATION".MethodLists.U01_STA3_MEAS_Method.MethodCount,
                           MethodHdl := "DB16101_U1_STA3_MEAS_CLIENT_CONFIGURATION".MethodLists.U01_STA3_MEAS_Method.MethodHdls[0],
                           NamespaceUris := "DB16101_U1_STA3_MEAS_CLIENT_CONFIGURATION".Namespaces.NamespaceURIs,
                           NamespaceStatusList := "DB16101_U1_STA3_MEAS_CLIENT_CONFIGURATION".Namespaces.NamespaceStatusList,
                           NamespaceIndexes := "DB16101_U1_STA3_MEAS_CLIENT_CONFIGURATION".Namespaces.ServerNamespaceIndexes,
                           ObjectNodeIDs := "DB16101_U1_STA3_MEAS_CLIENT_CONFIGURATION".MethodLists.U01_STA3_MEAS_Method.ObjectNodes,
                           MethodNodeIDs := "DB16101_U1_STA3_MEAS_CLIENT_CONFIGURATION".MethodLists.U01_STA3_MEAS_Method.MethodNodes,
                           MethodHdls := "DB16101_U1_STA3_MEAS_CLIENT_CONFIGURATION".MethodLists.U01_STA3_MEAS_Method.MethodHdls,
                           StatusList := "DB16001_U1_STA3_MEAS_CLIENT_INTERFACE".U01_STA3_MEAS_Method.MethodStatusList,
                           MethodResult := "DB16001_U1_STA3_MEAS_CLIENT_INTERFACE".U01_STA3_MEAS_Method.MethodResultList[0],
                           InputArguments := "DB16001_U1_STA3_MEAS_CLIENT_INTERFACE".U01_STA3_MEAS_Method."Trigger calculate distance".Inputs,
                           OutputArguments := "DB16001_U1_STA3_MEAS_CLIENT_INTERFACE".U01_STA3_MEAS_Method."Trigger calculate distance".Outputs);
END_REGION

REGION Network 16: UNIT 1 STATION 3 MEASURING START MEASURING LAYER THICKNESS TRIGGER CALL
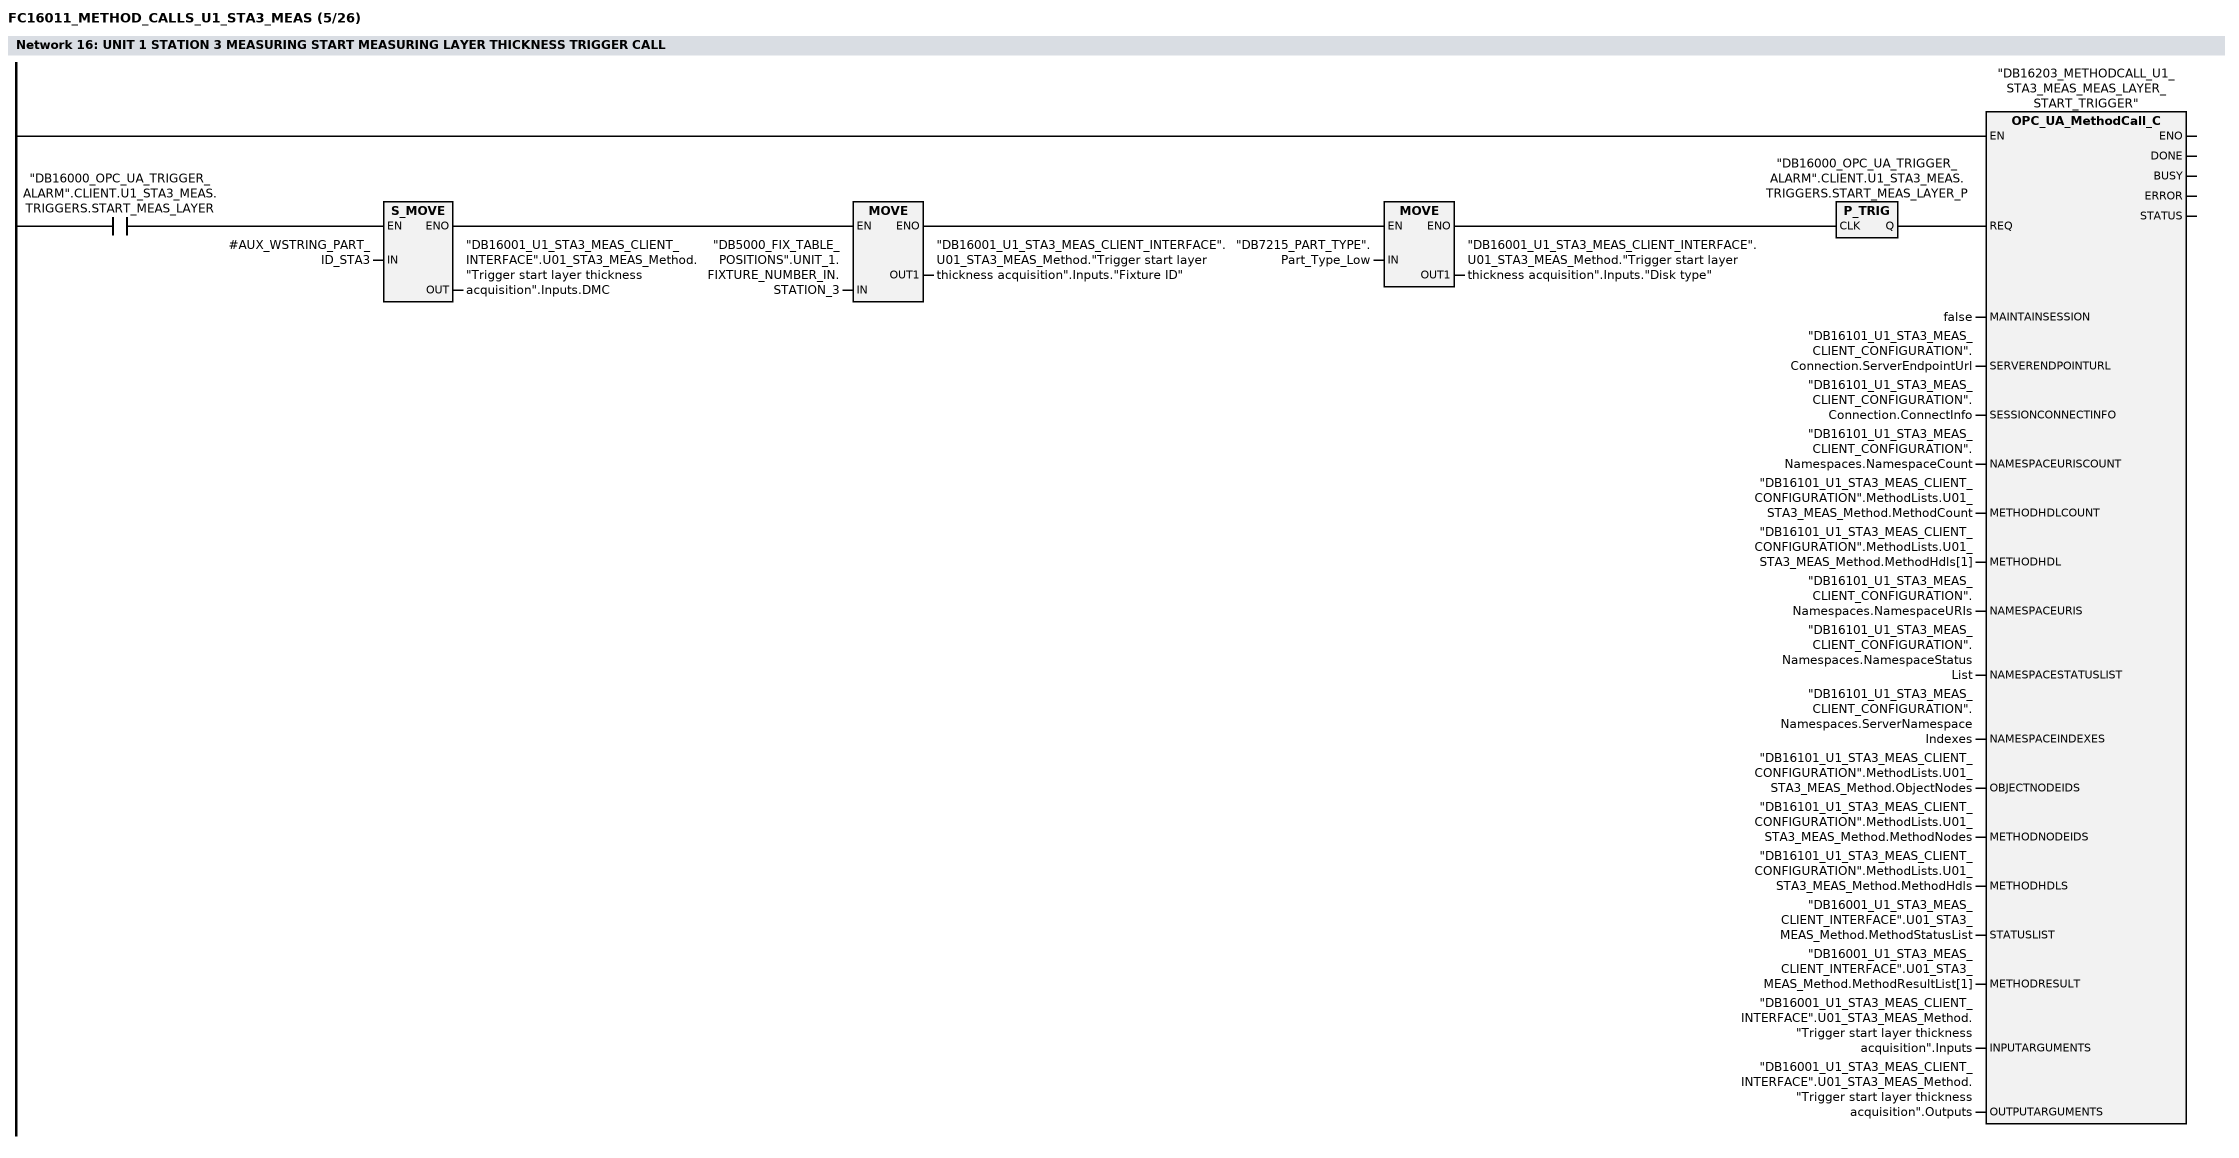
   RUNG wire#powerrail
      "DB16203_METHODCALL_U1_STA3_MEAS_MEAS_LAYER_START_TRIGGER".OPC_UA_MethodCall_C(REQ := wire#w1, MaintainSession := false, ServerEndpointUrl := "DB16101_U1_STA3_MEAS_CLIENT_CONFIGURATION".Connection.ServerEndpointUrl, SessionConnectInfo := "DB16101_U1_STA3_MEAS_CLIENT_CONFIGURATION".Connection.ConnectInfo, NamespaceUrisCount := "DB16101_U1_STA3_MEAS_CLIENT_CONFIGURATION".Namespaces.NamespaceCount, MethodHdlCount := "DB16101_U1_STA3_MEAS_CLIENT_CONFIGURATION".MethodLists.U01_STA3_MEAS_Method.MethodCount, MethodHdl := "DB16101_U1_STA3_MEAS_CLIENT_CONFIGURATION".MethodLists.U01_STA3_MEAS_Method.MethodHdls[1], NamespaceUris := "DB16101_U1_STA3_MEAS_CLIENT_CONFIGURATION".Namespaces.NamespaceURIs, NamespaceStatusList := "DB16101_U1_STA3_MEAS_CLIENT_CONFIGURATION".Namespaces.NamespaceStatusList, NamespaceIndexes := "DB16101_U1_STA3_MEAS_CLIENT_CONFIGURATION".Namespaces.ServerNamespaceIndexes, ObjectNodeIDs := "DB16101_U1_STA3_MEAS_CLIENT_CONFIGURATION".MethodLists.U01_STA3_MEAS_Method.ObjectNodes, MethodNodeIDs := "DB16101_U1_STA3_MEAS_CLIENT_CONFIGURATION".MethodLists.U01_STA3_MEAS_Method.MethodNodes, MethodHdls := "DB16101_U1_STA3_MEAS_CLIENT_CONFIGURATION".MethodLists.U01_STA3_MEAS_Method.MethodHdls, StatusList := "DB16001_U1_STA3_MEAS_CLIENT_INTERFACE".U01_STA3_MEAS_Method.MethodStatusList, MethodResult := "DB16001_U1_STA3_MEAS_CLIENT_INTERFACE".U01_STA3_MEAS_Method.MethodResultList[1], InputArguments := "DB16001_U1_STA3_MEAS_CLIENT_INTERFACE".U01_STA3_MEAS_Method."Trigger start layer thickness acquisition".Inputs, OutputArguments := "DB16001_U1_STA3_MEAS_CLIENT_INTERFACE".U01_STA3_MEAS_Method."Trigger start layer thickness acquisition".Outputs, Done =>, Busy =>, Error =>, Status =>)
   END_RUNG
   RUNG wire#powerrail
      Contact( "DB16000_OPC_UA_TRIGGER_ALARM".CLIENT.U1_STA3_MEAS.TRIGGERS.START_MEAS_LAYER )
      S_Move(in := #AUX_WSTRING_PART_ID_STA3, out => "DB16001_U1_STA3_MEAS_CLIENT_INTERFACE".U01_STA3_MEAS_Method."Trigger start layer thickness acquisition".Inputs.DMC)
      Move(in := "DB5000_FIX_TABLE_POSITIONS".UNIT_1.FIXTURE_NUMBER_IN.STATION_3, out1 => "DB16001_U1_STA3_MEAS_CLIENT_INTERFACE".U01_STA3_MEAS_Method."Trigger start layer thickness acquisition".Inputs."Fixture ID")
      Move(in := "DB7215_PART_TYPE".Part_Type_Low, out1 => "DB16001_U1_STA3_MEAS_CLIENT_INTERFACE".U01_STA3_MEAS_Method."Trigger start layer thickness acquisition".Inputs."Disk type")
      P_Trig( "DB16000_OPC_UA_TRIGGER_ALARM".CLIENT.U1_STA3_MEAS.TRIGGERS.START_MEAS_LAYER_P )
   END_RUNG wire#w1
   // the same network as SCL:
   IF "DB16000_OPC_UA_TRIGGER_ALARM".CLIENT.U1_STA3_MEAS.TRIGGERS.START_MEAS_LAYER THEN
       "DB16001_U1_STA3_MEAS_CLIENT_INTERFACE".U01_STA3_MEAS_Method."Trigger start layer thickness acquisition".Inputs.DMC := #AUX_WSTRING_PART_ID_STA3;
       "DB16001_U1_STA3_MEAS_CLIENT_INTERFACE".U01_STA3_MEAS_Method."Trigger start layer thickness acquisition".Inputs."Fixture ID" := "DB5000_FIX_TABLE_POSITIONS".UNIT_1.FIXTURE_NUMBER_IN.STATION_3;
       "DB16001_U1_STA3_MEAS_CLIENT_INTERFACE".U01_STA3_MEAS_Method."Trigger start layer thickness acquisition".Inputs."Disk type" := "DB7215_PART_TYPE".Part_Type_Low;
   END_IF;
   #_w1 := "DB16000_OPC_UA_TRIGGER_ALARM".CLIENT.U1_STA3_MEAS.TRIGGERS.START_MEAS_LAYER AND NOT "DB16000_OPC_UA_TRIGGER_ALARM".CLIENT.U1_STA3_MEAS.TRIGGERS.START_MEAS_LAYER_P;   // rising edge
   "DB16000_OPC_UA_TRIGGER_ALARM".CLIENT.U1_STA3_MEAS.TRIGGERS.START_MEAS_LAYER_P := "DB16000_OPC_UA_TRIGGER_ALARM".CLIENT.U1_STA3_MEAS.TRIGGERS.START_MEAS_LAYER;
   "DB16203_METHODCALL_U1_STA3_MEAS_MEAS_LAYER_START_TRIGGER"(REQ := #_w1,   // OPC_UA_MethodCall_C
                           MaintainSession := false,
                           ServerEndpointUrl := "DB16101_U1_STA3_MEAS_CLIENT_CONFIGURATION".Connection.ServerEndpointUrl,
                           SessionConnectInfo := "DB16101_U1_STA3_MEAS_CLIENT_CONFIGURATION".Connection.ConnectInfo,
                           NamespaceUrisCount := "DB16101_U1_STA3_MEAS_CLIENT_CONFIGURATION".Namespaces.NamespaceCount,
                           MethodHdlCount := "DB16101_U1_STA3_MEAS_CLIENT_CONFIGURATION".MethodLists.U01_STA3_MEAS_Method.MethodCount,
                           MethodHdl := "DB16101_U1_STA3_MEAS_CLIENT_CONFIGURATION".MethodLists.U01_STA3_MEAS_Method.MethodHdls[1],
                           NamespaceUris := "DB16101_U1_STA3_MEAS_CLIENT_CONFIGURATION".Namespaces.NamespaceURIs,
                           NamespaceStatusList := "DB16101_U1_STA3_MEAS_CLIENT_CONFIGURATION".Namespaces.NamespaceStatusList,
                           NamespaceIndexes := "DB16101_U1_STA3_MEAS_CLIENT_CONFIGURATION".Namespaces.ServerNamespaceIndexes,
                           ObjectNodeIDs := "DB16101_U1_STA3_MEAS_CLIENT_CONFIGURATION".MethodLists.U01_STA3_MEAS_Method.ObjectNodes,
                           MethodNodeIDs := "DB16101_U1_STA3_MEAS_CLIENT_CONFIGURATION".MethodLists.U01_STA3_MEAS_Method.MethodNodes,
                           MethodHdls := "DB16101_U1_STA3_MEAS_CLIENT_CONFIGURATION".MethodLists.U01_STA3_MEAS_Method.MethodHdls,
                           StatusList := "DB16001_U1_STA3_MEAS_CLIENT_INTERFACE".U01_STA3_MEAS_Method.MethodStatusList,
                           MethodResult := "DB16001_U1_STA3_MEAS_CLIENT_INTERFACE".U01_STA3_MEAS_Method.MethodResultList[1],
                           InputArguments := "DB16001_U1_STA3_MEAS_CLIENT_INTERFACE".U01_STA3_MEAS_Method."Trigger start layer thickness acquisition".Inputs,
                           OutputArguments := "DB16001_U1_STA3_MEAS_CLIENT_INTERFACE".U01_STA3_MEAS_Method."Trigger start layer thickness acquisition".Outputs);
END_REGION

REGION Network 17: UNIT 1 STATION 3 MEASURING STOP MEASURING LAYER THICKNESS TRIGGER CALL
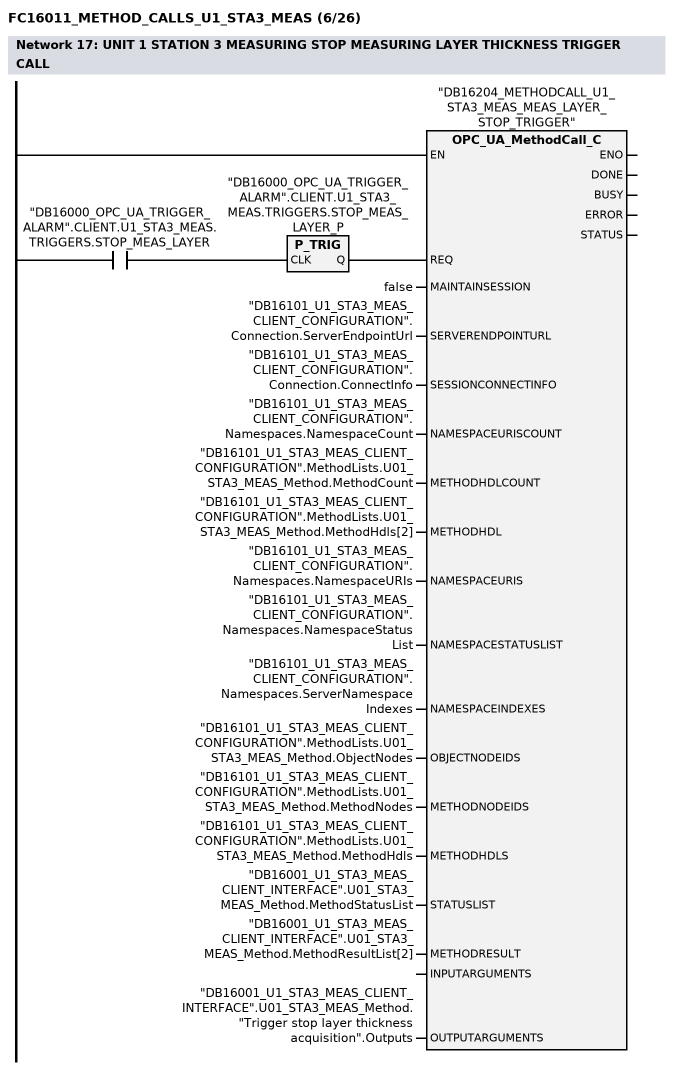
   RUNG wire#powerrail
      "DB16204_METHODCALL_U1_STA3_MEAS_MEAS_LAYER_STOP_TRIGGER".OPC_UA_MethodCall_C(REQ := wire#w1, MaintainSession := false, ServerEndpointUrl := "DB16101_U1_STA3_MEAS_CLIENT_CONFIGURATION".Connection.ServerEndpointUrl, SessionConnectInfo := "DB16101_U1_STA3_MEAS_CLIENT_CONFIGURATION".Connection.ConnectInfo, NamespaceUrisCount := "DB16101_U1_STA3_MEAS_CLIENT_CONFIGURATION".Namespaces.NamespaceCount, MethodHdlCount := "DB16101_U1_STA3_MEAS_CLIENT_CONFIGURATION".MethodLists.U01_STA3_MEAS_Method.MethodCount, MethodHdl := "DB16101_U1_STA3_MEAS_CLIENT_CONFIGURATION".MethodLists.U01_STA3_MEAS_Method.MethodHdls[2], NamespaceUris := "DB16101_U1_STA3_MEAS_CLIENT_CONFIGURATION".Namespaces.NamespaceURIs, NamespaceStatusList := "DB16101_U1_STA3_MEAS_CLIENT_CONFIGURATION".Namespaces.NamespaceStatusList, NamespaceIndexes := "DB16101_U1_STA3_MEAS_CLIENT_CONFIGURATION".Namespaces.ServerNamespaceIndexes, ObjectNodeIDs := "DB16101_U1_STA3_MEAS_CLIENT_CONFIGURATION".MethodLists.U01_STA3_MEAS_Method.ObjectNodes, MethodNodeIDs := "DB16101_U1_STA3_MEAS_CLIENT_CONFIGURATION".MethodLists.U01_STA3_MEAS_Method.MethodNodes, MethodHdls := "DB16101_U1_STA3_MEAS_CLIENT_CONFIGURATION".MethodLists.U01_STA3_MEAS_Method.MethodHdls, StatusList := "DB16001_U1_STA3_MEAS_CLIENT_INTERFACE".U01_STA3_MEAS_Method.MethodStatusList, MethodResult := "DB16001_U1_STA3_MEAS_CLIENT_INTERFACE".U01_STA3_MEAS_Method.MethodResultList[2], InputArguments :=, OutputArguments := "DB16001_U1_STA3_MEAS_CLIENT_INTERFACE".U01_STA3_MEAS_Method."Trigger stop layer thickness acquisition".Outputs, Done =>, Busy =>, Error =>, Status =>)
   END_RUNG
   RUNG wire#powerrail
      Contact( "DB16000_OPC_UA_TRIGGER_ALARM".CLIENT.U1_STA3_MEAS.TRIGGERS.STOP_MEAS_LAYER )
      P_Trig( "DB16000_OPC_UA_TRIGGER_ALARM".CLIENT.U1_STA3_MEAS.TRIGGERS.STOP_MEAS_LAYER_P )
   END_RUNG wire#w1
   // the same network as SCL:
   #_w1 := "DB16000_OPC_UA_TRIGGER_ALARM".CLIENT.U1_STA3_MEAS.TRIGGERS.STOP_MEAS_LAYER AND NOT "DB16000_OPC_UA_TRIGGER_ALARM".CLIENT.U1_STA3_MEAS.TRIGGERS.STOP_MEAS_LAYER_P;   // rising edge
   "DB16000_OPC_UA_TRIGGER_ALARM".CLIENT.U1_STA3_MEAS.TRIGGERS.STOP_MEAS_LAYER_P := "DB16000_OPC_UA_TRIGGER_ALARM".CLIENT.U1_STA3_MEAS.TRIGGERS.STOP_MEAS_LAYER;
   "DB16204_METHODCALL_U1_STA3_MEAS_MEAS_LAYER_STOP_TRIGGER"(REQ := #_w1,   // OPC_UA_MethodCall_C
                           MaintainSession := false,
                           ServerEndpointUrl := "DB16101_U1_STA3_MEAS_CLIENT_CONFIGURATION".Connection.ServerEndpointUrl,
                           SessionConnectInfo := "DB16101_U1_STA3_MEAS_CLIENT_CONFIGURATION".Connection.ConnectInfo,
                           NamespaceUrisCount := "DB16101_U1_STA3_MEAS_CLIENT_CONFIGURATION".Namespaces.NamespaceCount,
                           MethodHdlCount := "DB16101_U1_STA3_MEAS_CLIENT_CONFIGURATION".MethodLists.U01_STA3_MEAS_Method.MethodCount,
                           MethodHdl := "DB16101_U1_STA3_MEAS_CLIENT_CONFIGURATION".MethodLists.U01_STA3_MEAS_Method.MethodHdls[2],
                           NamespaceUris := "DB16101_U1_STA3_MEAS_CLIENT_CONFIGURATION".Namespaces.NamespaceURIs,
                           NamespaceStatusList := "DB16101_U1_STA3_MEAS_CLIENT_CONFIGURATION".Namespaces.NamespaceStatusList,
                           NamespaceIndexes := "DB16101_U1_STA3_MEAS_CLIENT_CONFIGURATION".Namespaces.ServerNamespaceIndexes,
                           ObjectNodeIDs := "DB16101_U1_STA3_MEAS_CLIENT_CONFIGURATION".MethodLists.U01_STA3_MEAS_Method.ObjectNodes,
                           MethodNodeIDs := "DB16101_U1_STA3_MEAS_CLIENT_CONFIGURATION".MethodLists.U01_STA3_MEAS_Method.MethodNodes,
                           MethodHdls := "DB16101_U1_STA3_MEAS_CLIENT_CONFIGURATION".MethodLists.U01_STA3_MEAS_Method.MethodHdls,
                           StatusList := "DB16001_U1_STA3_MEAS_CLIENT_INTERFACE".U01_STA3_MEAS_Method.MethodStatusList,
                           MethodResult := "DB16001_U1_STA3_MEAS_CLIENT_INTERFACE".U01_STA3_MEAS_Method.MethodResultList[2],
                           OutputArguments := "DB16001_U1_STA3_MEAS_CLIENT_INTERFACE".U01_STA3_MEAS_Method."Trigger stop layer thickness acquisition".Outputs);
END_REGION

REGION Network 18: UNIT 1 STATION 3 MEASURING START CALIBRATING TRIGGER CALL
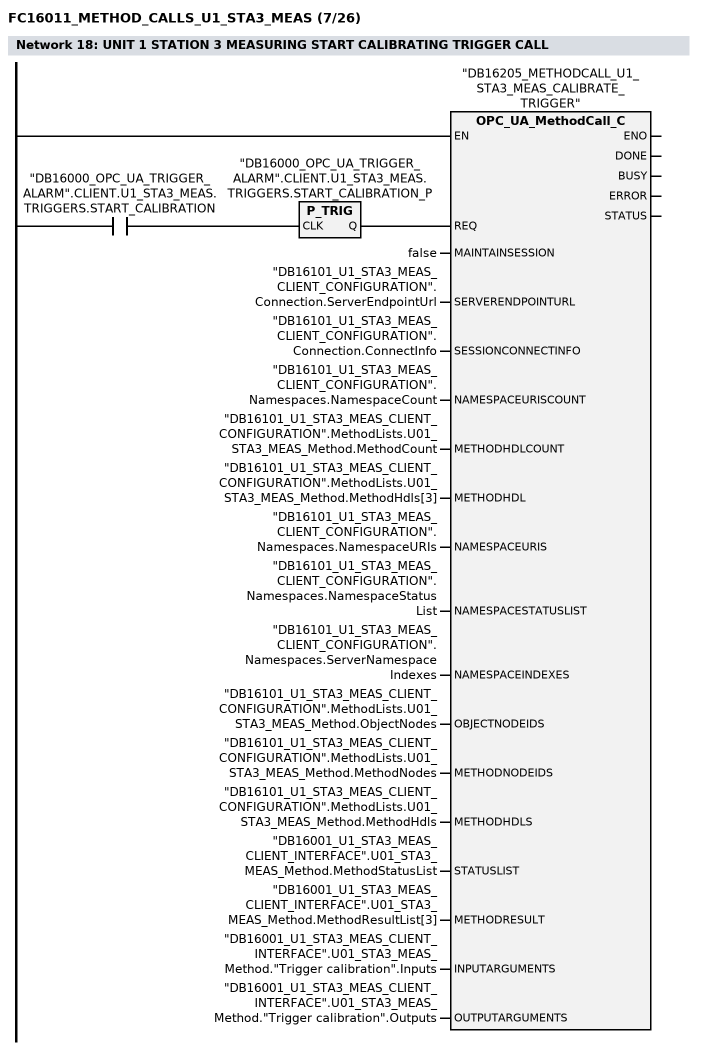
   RUNG wire#powerrail
      "DB16205_METHODCALL_U1_STA3_MEAS_CALIBRATE_TRIGGER".OPC_UA_MethodCall_C(REQ := wire#w1, MaintainSession := false, ServerEndpointUrl := "DB16101_U1_STA3_MEAS_CLIENT_CONFIGURATION".Connection.ServerEndpointUrl, SessionConnectInfo := "DB16101_U1_STA3_MEAS_CLIENT_CONFIGURATION".Connection.ConnectInfo, NamespaceUrisCount := "DB16101_U1_STA3_MEAS_CLIENT_CONFIGURATION".Namespaces.NamespaceCount, MethodHdlCount := "DB16101_U1_STA3_MEAS_CLIENT_CONFIGURATION".MethodLists.U01_STA3_MEAS_Method.MethodCount, MethodHdl := "DB16101_U1_STA3_MEAS_CLIENT_CONFIGURATION".MethodLists.U01_STA3_MEAS_Method.MethodHdls[3], NamespaceUris := "DB16101_U1_STA3_MEAS_CLIENT_CONFIGURATION".Namespaces.NamespaceURIs, NamespaceStatusList := "DB16101_U1_STA3_MEAS_CLIENT_CONFIGURATION".Namespaces.NamespaceStatusList, NamespaceIndexes := "DB16101_U1_STA3_MEAS_CLIENT_CONFIGURATION".Namespaces.ServerNamespaceIndexes, ObjectNodeIDs := "DB16101_U1_STA3_MEAS_CLIENT_CONFIGURATION".MethodLists.U01_STA3_MEAS_Method.ObjectNodes, MethodNodeIDs := "DB16101_U1_STA3_MEAS_CLIENT_CONFIGURATION".MethodLists.U01_STA3_MEAS_Method.MethodNodes, MethodHdls := "DB16101_U1_STA3_MEAS_CLIENT_CONFIGURATION".MethodLists.U01_STA3_MEAS_Method.MethodHdls, StatusList := "DB16001_U1_STA3_MEAS_CLIENT_INTERFACE".U01_STA3_MEAS_Method.MethodStatusList, MethodResult := "DB16001_U1_STA3_MEAS_CLIENT_INTERFACE".U01_STA3_MEAS_Method.MethodResultList[3], InputArguments := "DB16001_U1_STA3_MEAS_CLIENT_INTERFACE".U01_STA3_MEAS_Method."Trigger calibration".Inputs, OutputArguments := "DB16001_U1_STA3_MEAS_CLIENT_INTERFACE".U01_STA3_MEAS_Method."Trigger calibration".Outputs, Done =>, Busy =>, Error =>, Status =>)
   END_RUNG
   RUNG wire#powerrail
      Contact( "DB16000_OPC_UA_TRIGGER_ALARM".CLIENT.U1_STA3_MEAS.TRIGGERS.START_CALIBRATION )
      P_Trig( "DB16000_OPC_UA_TRIGGER_ALARM".CLIENT.U1_STA3_MEAS.TRIGGERS.START_CALIBRATION_P )
   END_RUNG wire#w1
   // the same network as SCL:
   #_w1 := "DB16000_OPC_UA_TRIGGER_ALARM".CLIENT.U1_STA3_MEAS.TRIGGERS.START_CALIBRATION AND NOT "DB16000_OPC_UA_TRIGGER_ALARM".CLIENT.U1_STA3_MEAS.TRIGGERS.START_CALIBRATION_P;   // rising edge
   "DB16000_OPC_UA_TRIGGER_ALARM".CLIENT.U1_STA3_MEAS.TRIGGERS.START_CALIBRATION_P := "DB16000_OPC_UA_TRIGGER_ALARM".CLIENT.U1_STA3_MEAS.TRIGGERS.START_CALIBRATION;
   "DB16205_METHODCALL_U1_STA3_MEAS_CALIBRATE_TRIGGER"(REQ := #_w1,   // OPC_UA_MethodCall_C
                           MaintainSession := false,
                           ServerEndpointUrl := "DB16101_U1_STA3_MEAS_CLIENT_CONFIGURATION".Connection.ServerEndpointUrl,
                           SessionConnectInfo := "DB16101_U1_STA3_MEAS_CLIENT_CONFIGURATION".Connection.ConnectInfo,
                           NamespaceUrisCount := "DB16101_U1_STA3_MEAS_CLIENT_CONFIGURATION".Namespaces.NamespaceCount,
                           MethodHdlCount := "DB16101_U1_STA3_MEAS_CLIENT_CONFIGURATION".MethodLists.U01_STA3_MEAS_Method.MethodCount,
                           MethodHdl := "DB16101_U1_STA3_MEAS_CLIENT_CONFIGURATION".MethodLists.U01_STA3_MEAS_Method.MethodHdls[3],
                           NamespaceUris := "DB16101_U1_STA3_MEAS_CLIENT_CONFIGURATION".Namespaces.NamespaceURIs,
                           NamespaceStatusList := "DB16101_U1_STA3_MEAS_CLIENT_CONFIGURATION".Namespaces.NamespaceStatusList,
                           NamespaceIndexes := "DB16101_U1_STA3_MEAS_CLIENT_CONFIGURATION".Namespaces.ServerNamespaceIndexes,
                           ObjectNodeIDs := "DB16101_U1_STA3_MEAS_CLIENT_CONFIGURATION".MethodLists.U01_STA3_MEAS_Method.ObjectNodes,
                           MethodNodeIDs := "DB16101_U1_STA3_MEAS_CLIENT_CONFIGURATION".MethodLists.U01_STA3_MEAS_Method.MethodNodes,
                           MethodHdls := "DB16101_U1_STA3_MEAS_CLIENT_CONFIGURATION".MethodLists.U01_STA3_MEAS_Method.MethodHdls,
                           StatusList := "DB16001_U1_STA3_MEAS_CLIENT_INTERFACE".U01_STA3_MEAS_Method.MethodStatusList,
                           MethodResult := "DB16001_U1_STA3_MEAS_CLIENT_INTERFACE".U01_STA3_MEAS_Method.MethodResultList[3],
                           InputArguments := "DB16001_U1_STA3_MEAS_CLIENT_INTERFACE".U01_STA3_MEAS_Method."Trigger calibration".Inputs,
                           OutputArguments := "DB16001_U1_STA3_MEAS_CLIENT_INTERFACE".U01_STA3_MEAS_Method."Trigger calibration".Outputs);
END_REGION

REGION Network 19: UNIT 1 STATION 3 MEASURING RESET PC TRIGGER CALL
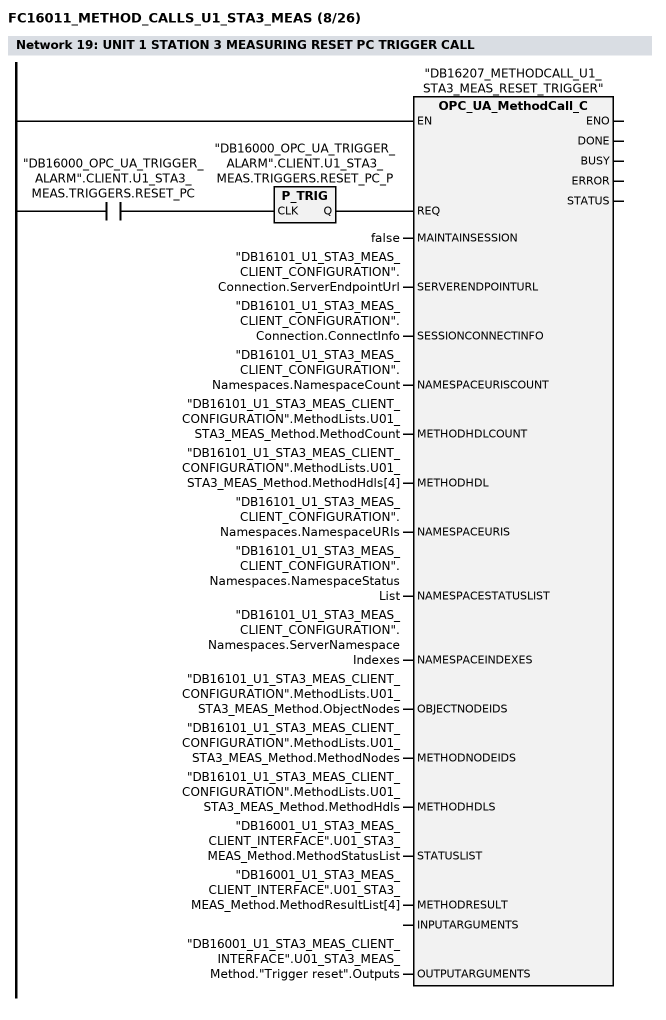
   RUNG wire#powerrail
      "DB16207_METHODCALL_U1_STA3_MEAS_RESET_TRIGGER".OPC_UA_MethodCall_C(REQ := wire#w1, MaintainSession := false, ServerEndpointUrl := "DB16101_U1_STA3_MEAS_CLIENT_CONFIGURATION".Connection.ServerEndpointUrl, SessionConnectInfo := "DB16101_U1_STA3_MEAS_CLIENT_CONFIGURATION".Connection.ConnectInfo, NamespaceUrisCount := "DB16101_U1_STA3_MEAS_CLIENT_CONFIGURATION".Namespaces.NamespaceCount, MethodHdlCount := "DB16101_U1_STA3_MEAS_CLIENT_CONFIGURATION".MethodLists.U01_STA3_MEAS_Method.MethodCount, MethodHdl := "DB16101_U1_STA3_MEAS_CLIENT_CONFIGURATION".MethodLists.U01_STA3_MEAS_Method.MethodHdls[4], NamespaceUris := "DB16101_U1_STA3_MEAS_CLIENT_CONFIGURATION".Namespaces.NamespaceURIs, NamespaceStatusList := "DB16101_U1_STA3_MEAS_CLIENT_CONFIGURATION".Namespaces.NamespaceStatusList, NamespaceIndexes := "DB16101_U1_STA3_MEAS_CLIENT_CONFIGURATION".Namespaces.ServerNamespaceIndexes, ObjectNodeIDs := "DB16101_U1_STA3_MEAS_CLIENT_CONFIGURATION".MethodLists.U01_STA3_MEAS_Method.ObjectNodes, MethodNodeIDs := "DB16101_U1_STA3_MEAS_CLIENT_CONFIGURATION".MethodLists.U01_STA3_MEAS_Method.MethodNodes, MethodHdls := "DB16101_U1_STA3_MEAS_CLIENT_CONFIGURATION".MethodLists.U01_STA3_MEAS_Method.MethodHdls, StatusList := "DB16001_U1_STA3_MEAS_CLIENT_INTERFACE".U01_STA3_MEAS_Method.MethodStatusList, MethodResult := "DB16001_U1_STA3_MEAS_CLIENT_INTERFACE".U01_STA3_MEAS_Method.MethodResultList[4], InputArguments :=, OutputArguments := "DB16001_U1_STA3_MEAS_CLIENT_INTERFACE".U01_STA3_MEAS_Method."Trigger reset".Outputs, Done =>, Busy =>, Error =>, Status =>)
   END_RUNG
   RUNG wire#powerrail
      Contact( "DB16000_OPC_UA_TRIGGER_ALARM".CLIENT.U1_STA3_MEAS.TRIGGERS.RESET_PC )
      P_Trig( "DB16000_OPC_UA_TRIGGER_ALARM".CLIENT.U1_STA3_MEAS.TRIGGERS.RESET_PC_P )
   END_RUNG wire#w1
   // the same network as SCL:
   #_w1 := "DB16000_OPC_UA_TRIGGER_ALARM".CLIENT.U1_STA3_MEAS.TRIGGERS.RESET_PC AND NOT "DB16000_OPC_UA_TRIGGER_ALARM".CLIENT.U1_STA3_MEAS.TRIGGERS.RESET_PC_P;   // rising edge
   "DB16000_OPC_UA_TRIGGER_ALARM".CLIENT.U1_STA3_MEAS.TRIGGERS.RESET_PC_P := "DB16000_OPC_UA_TRIGGER_ALARM".CLIENT.U1_STA3_MEAS.TRIGGERS.RESET_PC;
   "DB16207_METHODCALL_U1_STA3_MEAS_RESET_TRIGGER"(REQ := #_w1,   // OPC_UA_MethodCall_C
                           MaintainSession := false,
                           ServerEndpointUrl := "DB16101_U1_STA3_MEAS_CLIENT_CONFIGURATION".Connection.ServerEndpointUrl,
                           SessionConnectInfo := "DB16101_U1_STA3_MEAS_CLIENT_CONFIGURATION".Connection.ConnectInfo,
                           NamespaceUrisCount := "DB16101_U1_STA3_MEAS_CLIENT_CONFIGURATION".Namespaces.NamespaceCount,
                           MethodHdlCount := "DB16101_U1_STA3_MEAS_CLIENT_CONFIGURATION".MethodLists.U01_STA3_MEAS_Method.MethodCount,
                           MethodHdl := "DB16101_U1_STA3_MEAS_CLIENT_CONFIGURATION".MethodLists.U01_STA3_MEAS_Method.MethodHdls[4],
                           NamespaceUris := "DB16101_U1_STA3_MEAS_CLIENT_CONFIGURATION".Namespaces.NamespaceURIs,
                           NamespaceStatusList := "DB16101_U1_STA3_MEAS_CLIENT_CONFIGURATION".Namespaces.NamespaceStatusList,
                           NamespaceIndexes := "DB16101_U1_STA3_MEAS_CLIENT_CONFIGURATION".Namespaces.ServerNamespaceIndexes,
                           ObjectNodeIDs := "DB16101_U1_STA3_MEAS_CLIENT_CONFIGURATION".MethodLists.U01_STA3_MEAS_Method.ObjectNodes,
                           MethodNodeIDs := "DB16101_U1_STA3_MEAS_CLIENT_CONFIGURATION".MethodLists.U01_STA3_MEAS_Method.MethodNodes,
                           MethodHdls := "DB16101_U1_STA3_MEAS_CLIENT_CONFIGURATION".MethodLists.U01_STA3_MEAS_Method.MethodHdls,
                           StatusList := "DB16001_U1_STA3_MEAS_CLIENT_INTERFACE".U01_STA3_MEAS_Method.MethodStatusList,
                           MethodResult := "DB16001_U1_STA3_MEAS_CLIENT_INTERFACE".U01_STA3_MEAS_Method.MethodResultList[4],
                           OutputArguments := "DB16001_U1_STA3_MEAS_CLIENT_INTERFACE".U01_STA3_MEAS_Method."Trigger reset".Outputs);
END_REGION

REGION Network 20: UNIT 1 STATION 3 MEASURING READ VARIABLES TRIGGER CALL
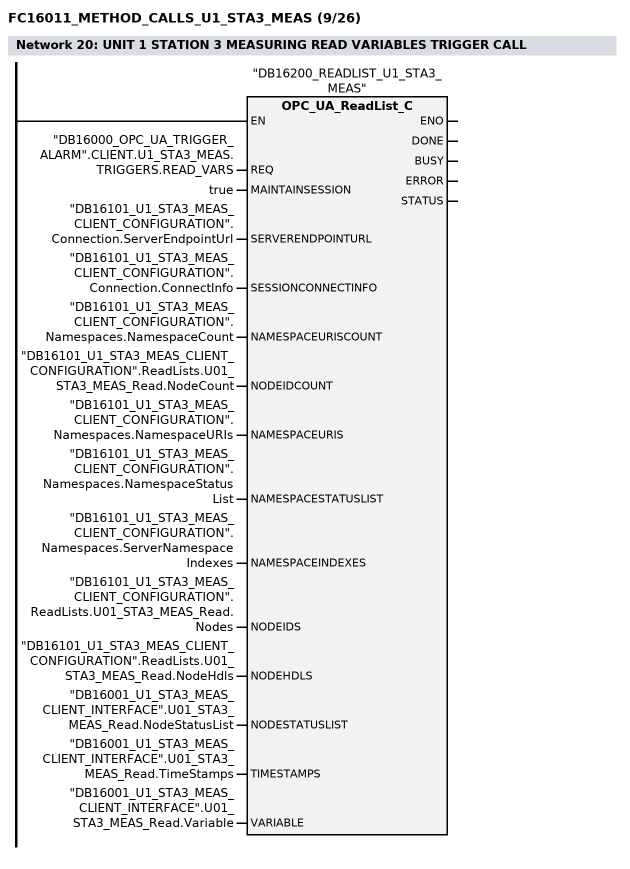
   RUNG wire#powerrail
      "DB16200_READLIST_U1_STA3_MEAS".OPC_UA_ReadList_C(REQ := "DB16000_OPC_UA_TRIGGER_ALARM".CLIENT.U1_STA3_MEAS.TRIGGERS.READ_VARS, MaintainSession := true, ServerEndpointUrl := "DB16101_U1_STA3_MEAS_CLIENT_CONFIGURATION".Connection.ServerEndpointUrl, SessionConnectInfo := "DB16101_U1_STA3_MEAS_CLIENT_CONFIGURATION".Connection.ConnectInfo, NamespaceUrisCount := "DB16101_U1_STA3_MEAS_CLIENT_CONFIGURATION".Namespaces.NamespaceCount, NodeIDCount := "DB16101_U1_STA3_MEAS_CLIENT_CONFIGURATION".ReadLists.U01_STA3_MEAS_Read.NodeCount, NamespaceUris := "DB16101_U1_STA3_MEAS_CLIENT_CONFIGURATION".Namespaces.NamespaceURIs, NamespaceStatusList := "DB16101_U1_STA3_MEAS_CLIENT_CONFIGURATION".Namespaces.NamespaceStatusList, NamespaceIndexes := "DB16101_U1_STA3_MEAS_CLIENT_CONFIGURATION".Namespaces.ServerNamespaceIndexes, NodeIDs := "DB16101_U1_STA3_MEAS_CLIENT_CONFIGURATION".ReadLists.U01_STA3_MEAS_Read.Nodes, NodeHdls := "DB16101_U1_STA3_MEAS_CLIENT_CONFIGURATION".ReadLists.U01_STA3_MEAS_Read.NodeHdls, NodeStatusList := "DB16001_U1_STA3_MEAS_CLIENT_INTERFACE".U01_STA3_MEAS_Read.NodeStatusList, Timestamps := "DB16001_U1_STA3_MEAS_CLIENT_INTERFACE".U01_STA3_MEAS_Read.TimeStamps, Variable := "DB16001_U1_STA3_MEAS_CLIENT_INTERFACE".U01_STA3_MEAS_Read.Variable, Done =>, Busy =>, Error =>, Status =>)
   END_RUNG
   // the same network as SCL:
   "DB16200_READLIST_U1_STA3_MEAS"(REQ := "DB16000_OPC_UA_TRIGGER_ALARM".CLIENT.U1_STA3_MEAS.TRIGGERS.READ_VARS,   // OPC_UA_ReadList_C
                           MaintainSession := true,
                           ServerEndpointUrl := "DB16101_U1_STA3_MEAS_CLIENT_CONFIGURATION".Connection.ServerEndpointUrl,
                           SessionConnectInfo := "DB16101_U1_STA3_MEAS_CLIENT_CONFIGURATION".Connection.ConnectInfo,
                           NamespaceUrisCount := "DB16101_U1_STA3_MEAS_CLIENT_CONFIGURATION".Namespaces.NamespaceCount,
                           NodeIDCount := "DB16101_U1_STA3_MEAS_CLIENT_CONFIGURATION".ReadLists.U01_STA3_MEAS_Read.NodeCount,
                           NamespaceUris := "DB16101_U1_STA3_MEAS_CLIENT_CONFIGURATION".Namespaces.NamespaceURIs,
                           NamespaceStatusList := "DB16101_U1_STA3_MEAS_CLIENT_CONFIGURATION".Namespaces.NamespaceStatusList,
                           NamespaceIndexes := "DB16101_U1_STA3_MEAS_CLIENT_CONFIGURATION".Namespaces.ServerNamespaceIndexes,
                           NodeIDs := "DB16101_U1_STA3_MEAS_CLIENT_CONFIGURATION".ReadLists.U01_STA3_MEAS_Read.Nodes,
                           NodeHdls := "DB16101_U1_STA3_MEAS_CLIENT_CONFIGURATION".ReadLists.U01_STA3_MEAS_Read.NodeHdls,
                           NodeStatusList := "DB16001_U1_STA3_MEAS_CLIENT_INTERFACE".U01_STA3_MEAS_Read.NodeStatusList,
                           Timestamps := "DB16001_U1_STA3_MEAS_CLIENT_INTERFACE".U01_STA3_MEAS_Read.TimeStamps,
                           Variable := "DB16001_U1_STA3_MEAS_CLIENT_INTERFACE".U01_STA3_MEAS_Read.Variable);
END_REGION

REGION Network 21: UNIT 1 STATION 3 MEASURING MEASURING NOZZLE SURFACE DISTANCE TRIGGER RETRY
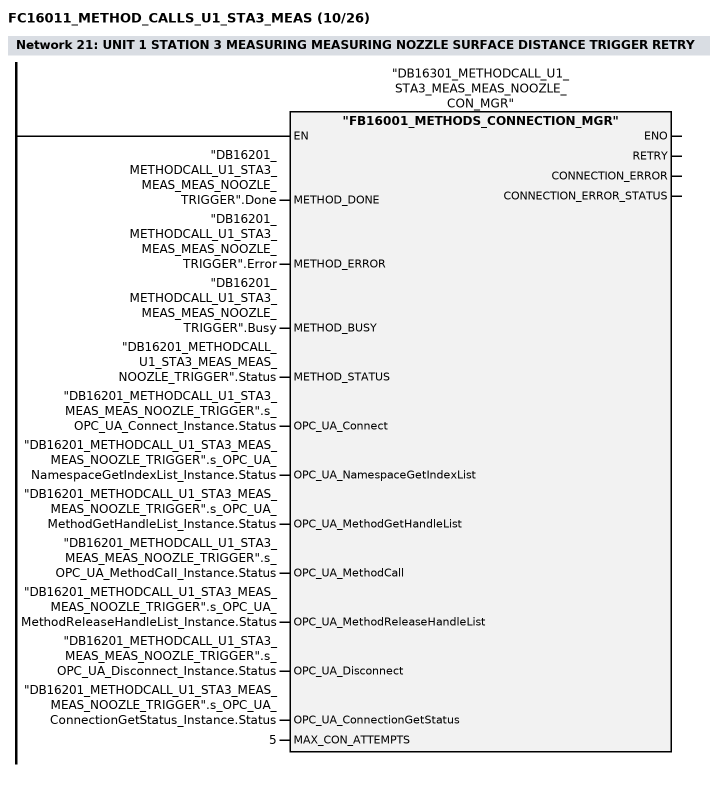
   RUNG wire#powerrail
      "DB16301_METHODCALL_U1_STA3_MEAS_MEAS_NOOZLE_CON_MGR"(METHOD_DONE := "DB16201_METHODCALL_U1_STA3_MEAS_MEAS_NOOZLE_TRIGGER".Done, METHOD_ERROR := "DB16201_METHODCALL_U1_STA3_MEAS_MEAS_NOOZLE_TRIGGER".Error, METHOD_BUSY := "DB16201_METHODCALL_U1_STA3_MEAS_MEAS_NOOZLE_TRIGGER".Busy, METHOD_STATUS := "DB16201_METHODCALL_U1_STA3_MEAS_MEAS_NOOZLE_TRIGGER".Status, OPC_UA_Connect := "DB16201_METHODCALL_U1_STA3_MEAS_MEAS_NOOZLE_TRIGGER".s_OPC_UA_Connect_Instance.Status, OPC_UA_NamespaceGetIndexList := "DB16201_METHODCALL_U1_STA3_MEAS_MEAS_NOOZLE_TRIGGER".s_OPC_UA_NamespaceGetIndexList_Instance.Status, OPC_UA_MethodGetHandleList := "DB16201_METHODCALL_U1_STA3_MEAS_MEAS_NOOZLE_TRIGGER".s_OPC_UA_MethodGetHandleList_Instance.Status, OPC_UA_MethodCall := "DB16201_METHODCALL_U1_STA3_MEAS_MEAS_NOOZLE_TRIGGER".s_OPC_UA_MethodCall_Instance.Status, OPC_UA_MethodReleaseHandleList := "DB16201_METHODCALL_U1_STA3_MEAS_MEAS_NOOZLE_TRIGGER".s_OPC_UA_MethodReleaseHandleList_Instance.Status, OPC_UA_Disconnect := "DB16201_METHODCALL_U1_STA3_MEAS_MEAS_NOOZLE_TRIGGER".s_OPC_UA_Disconnect_Instance.Status, OPC_UA_ConnectionGetStatus := "DB16201_METHODCALL_U1_STA3_MEAS_MEAS_NOOZLE_TRIGGER".s_OPC_UA_ConnectionGetStatus_Instance.Status, MAX_CON_ATTEMPTS := 5, RETRY =>, CONNECTION_ERROR =>, CONNECTION_ERROR_STATUS =>)
   END_RUNG
   // the same network as SCL:
   "DB16301_METHODCALL_U1_STA3_MEAS_MEAS_NOOZLE_CON_MGR"(METHOD_DONE := "DB16201_METHODCALL_U1_STA3_MEAS_MEAS_NOOZLE_TRIGGER".Done,   // "FB16001_METHODS_CONNECTION_MGR"
                           METHOD_ERROR := "DB16201_METHODCALL_U1_STA3_MEAS_MEAS_NOOZLE_TRIGGER".Error,
                           METHOD_BUSY := "DB16201_METHODCALL_U1_STA3_MEAS_MEAS_NOOZLE_TRIGGER".Busy,
                           METHOD_STATUS := "DB16201_METHODCALL_U1_STA3_MEAS_MEAS_NOOZLE_TRIGGER".Status,
                           OPC_UA_Connect := "DB16201_METHODCALL_U1_STA3_MEAS_MEAS_NOOZLE_TRIGGER".s_OPC_UA_Connect_Instance.Status,
                           OPC_UA_NamespaceGetIndexList := "DB16201_METHODCALL_U1_STA3_MEAS_MEAS_NOOZLE_TRIGGER".s_OPC_UA_NamespaceGetIndexList_Instance.Status,
                           OPC_UA_MethodGetHandleList := "DB16201_METHODCALL_U1_STA3_MEAS_MEAS_NOOZLE_TRIGGER".s_OPC_UA_MethodGetHandleList_Instance.Status,
                           OPC_UA_MethodCall := "DB16201_METHODCALL_U1_STA3_MEAS_MEAS_NOOZLE_TRIGGER".s_OPC_UA_MethodCall_Instance.Status,
                           OPC_UA_MethodReleaseHandleList := "DB16201_METHODCALL_U1_STA3_MEAS_MEAS_NOOZLE_TRIGGER".s_OPC_UA_MethodReleaseHandleList_Instance.Status,
                           OPC_UA_Disconnect := "DB16201_METHODCALL_U1_STA3_MEAS_MEAS_NOOZLE_TRIGGER".s_OPC_UA_Disconnect_Instance.Status,
                           OPC_UA_ConnectionGetStatus := "DB16201_METHODCALL_U1_STA3_MEAS_MEAS_NOOZLE_TRIGGER".s_OPC_UA_ConnectionGetStatus_Instance.Status,
                           MAX_CON_ATTEMPTS := 5);
END_REGION

REGION Network 22: UNIT 1 STATION 3 MEASURING START MEASURING LAYER THICKNESS TRIGGER RETRY
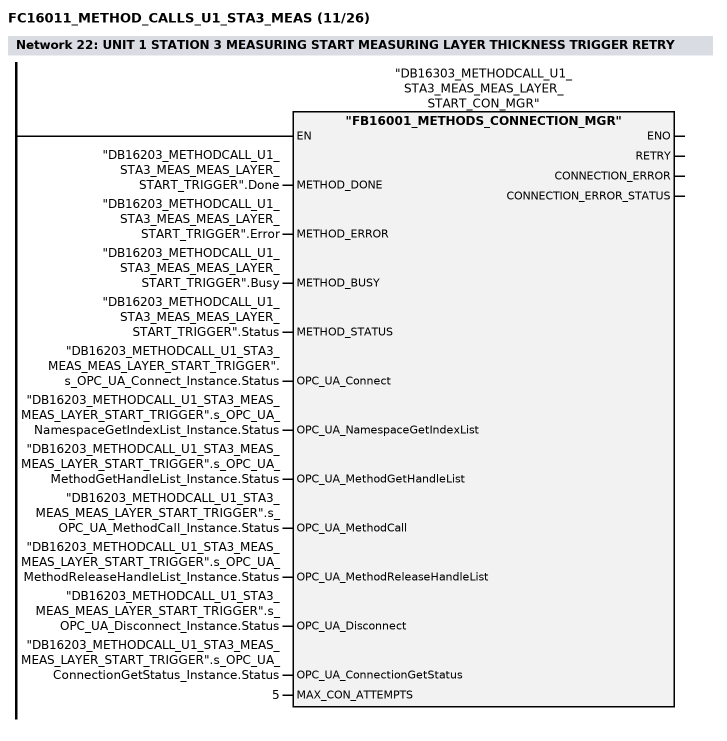
   RUNG wire#powerrail
      "DB16303_METHODCALL_U1_STA3_MEAS_MEAS_LAYER_START_CON_MGR"(METHOD_DONE := "DB16203_METHODCALL_U1_STA3_MEAS_MEAS_LAYER_START_TRIGGER".Done, METHOD_ERROR := "DB16203_METHODCALL_U1_STA3_MEAS_MEAS_LAYER_START_TRIGGER".Error, METHOD_BUSY := "DB16203_METHODCALL_U1_STA3_MEAS_MEAS_LAYER_START_TRIGGER".Busy, METHOD_STATUS := "DB16203_METHODCALL_U1_STA3_MEAS_MEAS_LAYER_START_TRIGGER".Status, OPC_UA_Connect := "DB16203_METHODCALL_U1_STA3_MEAS_MEAS_LAYER_START_TRIGGER".s_OPC_UA_Connect_Instance.Status, OPC_UA_NamespaceGetIndexList := "DB16203_METHODCALL_U1_STA3_MEAS_MEAS_LAYER_START_TRIGGER".s_OPC_UA_NamespaceGetIndexList_Instance.Status, OPC_UA_MethodGetHandleList := "DB16203_METHODCALL_U1_STA3_MEAS_MEAS_LAYER_START_TRIGGER".s_OPC_UA_MethodGetHandleList_Instance.Status, OPC_UA_MethodCall := "DB16203_METHODCALL_U1_STA3_MEAS_MEAS_LAYER_START_TRIGGER".s_OPC_UA_MethodCall_Instance.Status, OPC_UA_MethodReleaseHandleList := "DB16203_METHODCALL_U1_STA3_MEAS_MEAS_LAYER_START_TRIGGER".s_OPC_UA_MethodReleaseHandleList_Instance.Status, OPC_UA_Disconnect := "DB16203_METHODCALL_U1_STA3_MEAS_MEAS_LAYER_START_TRIGGER".s_OPC_UA_Disconnect_Instance.Status, OPC_UA_ConnectionGetStatus := "DB16203_METHODCALL_U1_STA3_MEAS_MEAS_LAYER_START_TRIGGER".s_OPC_UA_ConnectionGetStatus_Instance.Status, MAX_CON_ATTEMPTS := 5, RETRY =>, CONNECTION_ERROR =>, CONNECTION_ERROR_STATUS =>)
   END_RUNG
   // the same network as SCL:
   "DB16303_METHODCALL_U1_STA3_MEAS_MEAS_LAYER_START_CON_MGR"(METHOD_DONE := "DB16203_METHODCALL_U1_STA3_MEAS_MEAS_LAYER_START_TRIGGER".Done,   // "FB16001_METHODS_CONNECTION_MGR"
                           METHOD_ERROR := "DB16203_METHODCALL_U1_STA3_MEAS_MEAS_LAYER_START_TRIGGER".Error,
                           METHOD_BUSY := "DB16203_METHODCALL_U1_STA3_MEAS_MEAS_LAYER_START_TRIGGER".Busy,
                           METHOD_STATUS := "DB16203_METHODCALL_U1_STA3_MEAS_MEAS_LAYER_START_TRIGGER".Status,
                           OPC_UA_Connect := "DB16203_METHODCALL_U1_STA3_MEAS_MEAS_LAYER_START_TRIGGER".s_OPC_UA_Connect_Instance.Status,
                           OPC_UA_NamespaceGetIndexList := "DB16203_METHODCALL_U1_STA3_MEAS_MEAS_LAYER_START_TRIGGER".s_OPC_UA_NamespaceGetIndexList_Instance.Status,
                           OPC_UA_MethodGetHandleList := "DB16203_METHODCALL_U1_STA3_MEAS_MEAS_LAYER_START_TRIGGER".s_OPC_UA_MethodGetHandleList_Instance.Status,
                           OPC_UA_MethodCall := "DB16203_METHODCALL_U1_STA3_MEAS_MEAS_LAYER_START_TRIGGER".s_OPC_UA_MethodCall_Instance.Status,
                           OPC_UA_MethodReleaseHandleList := "DB16203_METHODCALL_U1_STA3_MEAS_MEAS_LAYER_START_TRIGGER".s_OPC_UA_MethodReleaseHandleList_Instance.Status,
                           OPC_UA_Disconnect := "DB16203_METHODCALL_U1_STA3_MEAS_MEAS_LAYER_START_TRIGGER".s_OPC_UA_Disconnect_Instance.Status,
                           OPC_UA_ConnectionGetStatus := "DB16203_METHODCALL_U1_STA3_MEAS_MEAS_LAYER_START_TRIGGER".s_OPC_UA_ConnectionGetStatus_Instance.Status,
                           MAX_CON_ATTEMPTS := 5);
END_REGION

REGION Network 23: UNIT 1 STATION 3 MEASURING STOP MEASURING LAYER THICKNESS TRIGGER RETRY
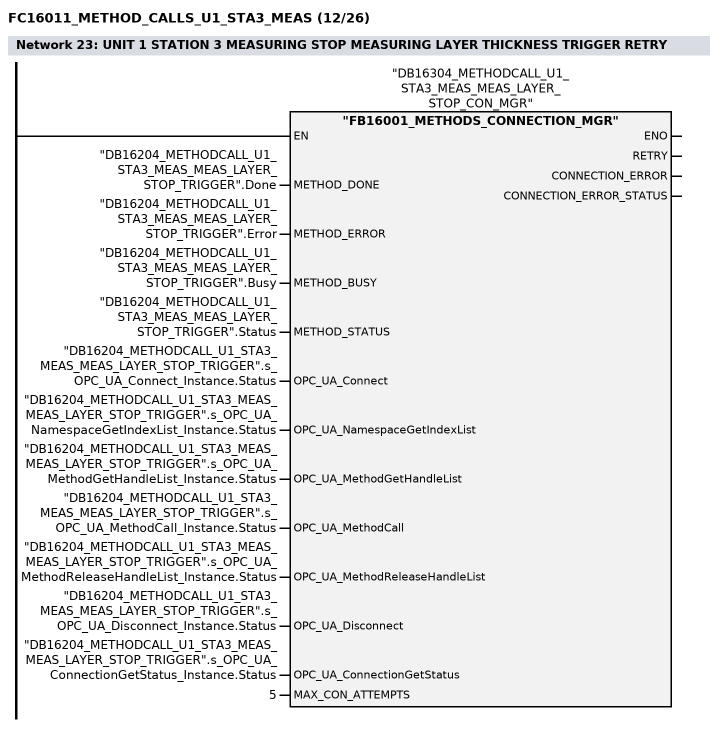
   RUNG wire#powerrail
      "DB16304_METHODCALL_U1_STA3_MEAS_MEAS_LAYER_STOP_CON_MGR"(METHOD_DONE := "DB16204_METHODCALL_U1_STA3_MEAS_MEAS_LAYER_STOP_TRIGGER".Done, METHOD_ERROR := "DB16204_METHODCALL_U1_STA3_MEAS_MEAS_LAYER_STOP_TRIGGER".Error, METHOD_BUSY := "DB16204_METHODCALL_U1_STA3_MEAS_MEAS_LAYER_STOP_TRIGGER".Busy, METHOD_STATUS := "DB16204_METHODCALL_U1_STA3_MEAS_MEAS_LAYER_STOP_TRIGGER".Status, OPC_UA_Connect := "DB16204_METHODCALL_U1_STA3_MEAS_MEAS_LAYER_STOP_TRIGGER".s_OPC_UA_Connect_Instance.Status, OPC_UA_NamespaceGetIndexList := "DB16204_METHODCALL_U1_STA3_MEAS_MEAS_LAYER_STOP_TRIGGER".s_OPC_UA_NamespaceGetIndexList_Instance.Status, OPC_UA_MethodGetHandleList := "DB16204_METHODCALL_U1_STA3_MEAS_MEAS_LAYER_STOP_TRIGGER".s_OPC_UA_MethodGetHandleList_Instance.Status, OPC_UA_MethodCall := "DB16204_METHODCALL_U1_STA3_MEAS_MEAS_LAYER_STOP_TRIGGER".s_OPC_UA_MethodCall_Instance.Status, OPC_UA_MethodReleaseHandleList := "DB16204_METHODCALL_U1_STA3_MEAS_MEAS_LAYER_STOP_TRIGGER".s_OPC_UA_MethodReleaseHandleList_Instance.Status, OPC_UA_Disconnect := "DB16204_METHODCALL_U1_STA3_MEAS_MEAS_LAYER_STOP_TRIGGER".s_OPC_UA_Disconnect_Instance.Status, OPC_UA_ConnectionGetStatus := "DB16204_METHODCALL_U1_STA3_MEAS_MEAS_LAYER_STOP_TRIGGER".s_OPC_UA_ConnectionGetStatus_Instance.Status, MAX_CON_ATTEMPTS := 5, RETRY =>, CONNECTION_ERROR =>, CONNECTION_ERROR_STATUS =>)
   END_RUNG
   // the same network as SCL:
   "DB16304_METHODCALL_U1_STA3_MEAS_MEAS_LAYER_STOP_CON_MGR"(METHOD_DONE := "DB16204_METHODCALL_U1_STA3_MEAS_MEAS_LAYER_STOP_TRIGGER".Done,   // "FB16001_METHODS_CONNECTION_MGR"
                           METHOD_ERROR := "DB16204_METHODCALL_U1_STA3_MEAS_MEAS_LAYER_STOP_TRIGGER".Error,
                           METHOD_BUSY := "DB16204_METHODCALL_U1_STA3_MEAS_MEAS_LAYER_STOP_TRIGGER".Busy,
                           METHOD_STATUS := "DB16204_METHODCALL_U1_STA3_MEAS_MEAS_LAYER_STOP_TRIGGER".Status,
                           OPC_UA_Connect := "DB16204_METHODCALL_U1_STA3_MEAS_MEAS_LAYER_STOP_TRIGGER".s_OPC_UA_Connect_Instance.Status,
                           OPC_UA_NamespaceGetIndexList := "DB16204_METHODCALL_U1_STA3_MEAS_MEAS_LAYER_STOP_TRIGGER".s_OPC_UA_NamespaceGetIndexList_Instance.Status,
                           OPC_UA_MethodGetHandleList := "DB16204_METHODCALL_U1_STA3_MEAS_MEAS_LAYER_STOP_TRIGGER".s_OPC_UA_MethodGetHandleList_Instance.Status,
                           OPC_UA_MethodCall := "DB16204_METHODCALL_U1_STA3_MEAS_MEAS_LAYER_STOP_TRIGGER".s_OPC_UA_MethodCall_Instance.Status,
                           OPC_UA_MethodReleaseHandleList := "DB16204_METHODCALL_U1_STA3_MEAS_MEAS_LAYER_STOP_TRIGGER".s_OPC_UA_MethodReleaseHandleList_Instance.Status,
                           OPC_UA_Disconnect := "DB16204_METHODCALL_U1_STA3_MEAS_MEAS_LAYER_STOP_TRIGGER".s_OPC_UA_Disconnect_Instance.Status,
                           OPC_UA_ConnectionGetStatus := "DB16204_METHODCALL_U1_STA3_MEAS_MEAS_LAYER_STOP_TRIGGER".s_OPC_UA_ConnectionGetStatus_Instance.Status,
                           MAX_CON_ATTEMPTS := 5);
END_REGION

REGION Network 24: UNIT 1 STATION 3 MEASURING CALIBRATING TRIGGER RETRY
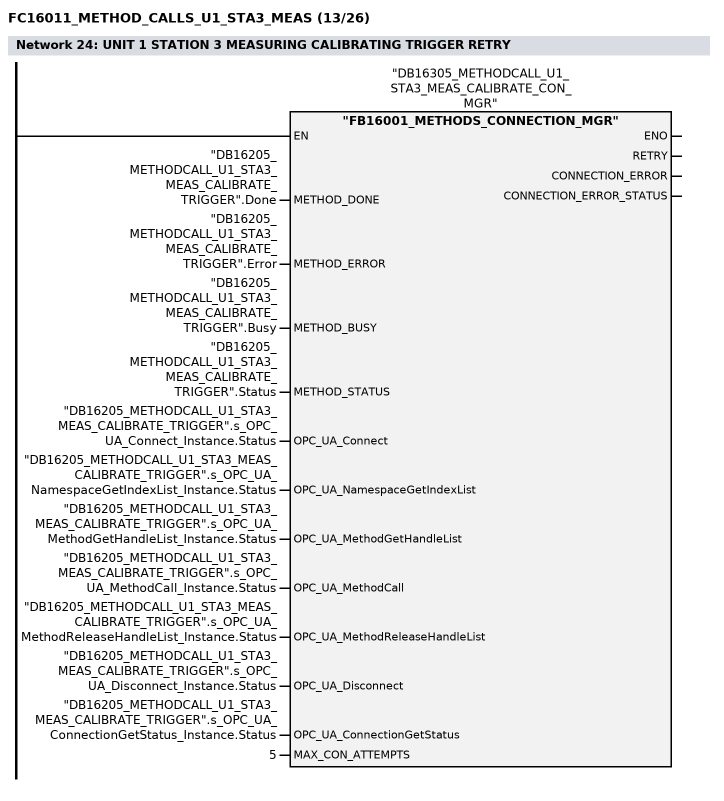
   RUNG wire#powerrail
      "DB16305_METHODCALL_U1_STA3_MEAS_CALIBRATE_CON_MGR"(METHOD_DONE := "DB16205_METHODCALL_U1_STA3_MEAS_CALIBRATE_TRIGGER".Done, METHOD_ERROR := "DB16205_METHODCALL_U1_STA3_MEAS_CALIBRATE_TRIGGER".Error, METHOD_BUSY := "DB16205_METHODCALL_U1_STA3_MEAS_CALIBRATE_TRIGGER".Busy, METHOD_STATUS := "DB16205_METHODCALL_U1_STA3_MEAS_CALIBRATE_TRIGGER".Status, OPC_UA_Connect := "DB16205_METHODCALL_U1_STA3_MEAS_CALIBRATE_TRIGGER".s_OPC_UA_Connect_Instance.Status, OPC_UA_NamespaceGetIndexList := "DB16205_METHODCALL_U1_STA3_MEAS_CALIBRATE_TRIGGER".s_OPC_UA_NamespaceGetIndexList_Instance.Status, OPC_UA_MethodGetHandleList := "DB16205_METHODCALL_U1_STA3_MEAS_CALIBRATE_TRIGGER".s_OPC_UA_MethodGetHandleList_Instance.Status, OPC_UA_MethodCall := "DB16205_METHODCALL_U1_STA3_MEAS_CALIBRATE_TRIGGER".s_OPC_UA_MethodCall_Instance.Status, OPC_UA_MethodReleaseHandleList := "DB16205_METHODCALL_U1_STA3_MEAS_CALIBRATE_TRIGGER".s_OPC_UA_MethodReleaseHandleList_Instance.Status, OPC_UA_Disconnect := "DB16205_METHODCALL_U1_STA3_MEAS_CALIBRATE_TRIGGER".s_OPC_UA_Disconnect_Instance.Status, OPC_UA_ConnectionGetStatus := "DB16205_METHODCALL_U1_STA3_MEAS_CALIBRATE_TRIGGER".s_OPC_UA_ConnectionGetStatus_Instance.Status, MAX_CON_ATTEMPTS := 5, RETRY =>, CONNECTION_ERROR =>, CONNECTION_ERROR_STATUS =>)
   END_RUNG
   // the same network as SCL:
   "DB16305_METHODCALL_U1_STA3_MEAS_CALIBRATE_CON_MGR"(METHOD_DONE := "DB16205_METHODCALL_U1_STA3_MEAS_CALIBRATE_TRIGGER".Done,   // "FB16001_METHODS_CONNECTION_MGR"
                           METHOD_ERROR := "DB16205_METHODCALL_U1_STA3_MEAS_CALIBRATE_TRIGGER".Error,
                           METHOD_BUSY := "DB16205_METHODCALL_U1_STA3_MEAS_CALIBRATE_TRIGGER".Busy,
                           METHOD_STATUS := "DB16205_METHODCALL_U1_STA3_MEAS_CALIBRATE_TRIGGER".Status,
                           OPC_UA_Connect := "DB16205_METHODCALL_U1_STA3_MEAS_CALIBRATE_TRIGGER".s_OPC_UA_Connect_Instance.Status,
                           OPC_UA_NamespaceGetIndexList := "DB16205_METHODCALL_U1_STA3_MEAS_CALIBRATE_TRIGGER".s_OPC_UA_NamespaceGetIndexList_Instance.Status,
                           OPC_UA_MethodGetHandleList := "DB16205_METHODCALL_U1_STA3_MEAS_CALIBRATE_TRIGGER".s_OPC_UA_MethodGetHandleList_Instance.Status,
                           OPC_UA_MethodCall := "DB16205_METHODCALL_U1_STA3_MEAS_CALIBRATE_TRIGGER".s_OPC_UA_MethodCall_Instance.Status,
                           OPC_UA_MethodReleaseHandleList := "DB16205_METHODCALL_U1_STA3_MEAS_CALIBRATE_TRIGGER".s_OPC_UA_MethodReleaseHandleList_Instance.Status,
                           OPC_UA_Disconnect := "DB16205_METHODCALL_U1_STA3_MEAS_CALIBRATE_TRIGGER".s_OPC_UA_Disconnect_Instance.Status,
                           OPC_UA_ConnectionGetStatus := "DB16205_METHODCALL_U1_STA3_MEAS_CALIBRATE_TRIGGER".s_OPC_UA_ConnectionGetStatus_Instance.Status,
                           MAX_CON_ATTEMPTS := 5);
END_REGION

REGION Network 25: UNIT 1 STATION 3 MEASURING RESET TRIGGER RETRY
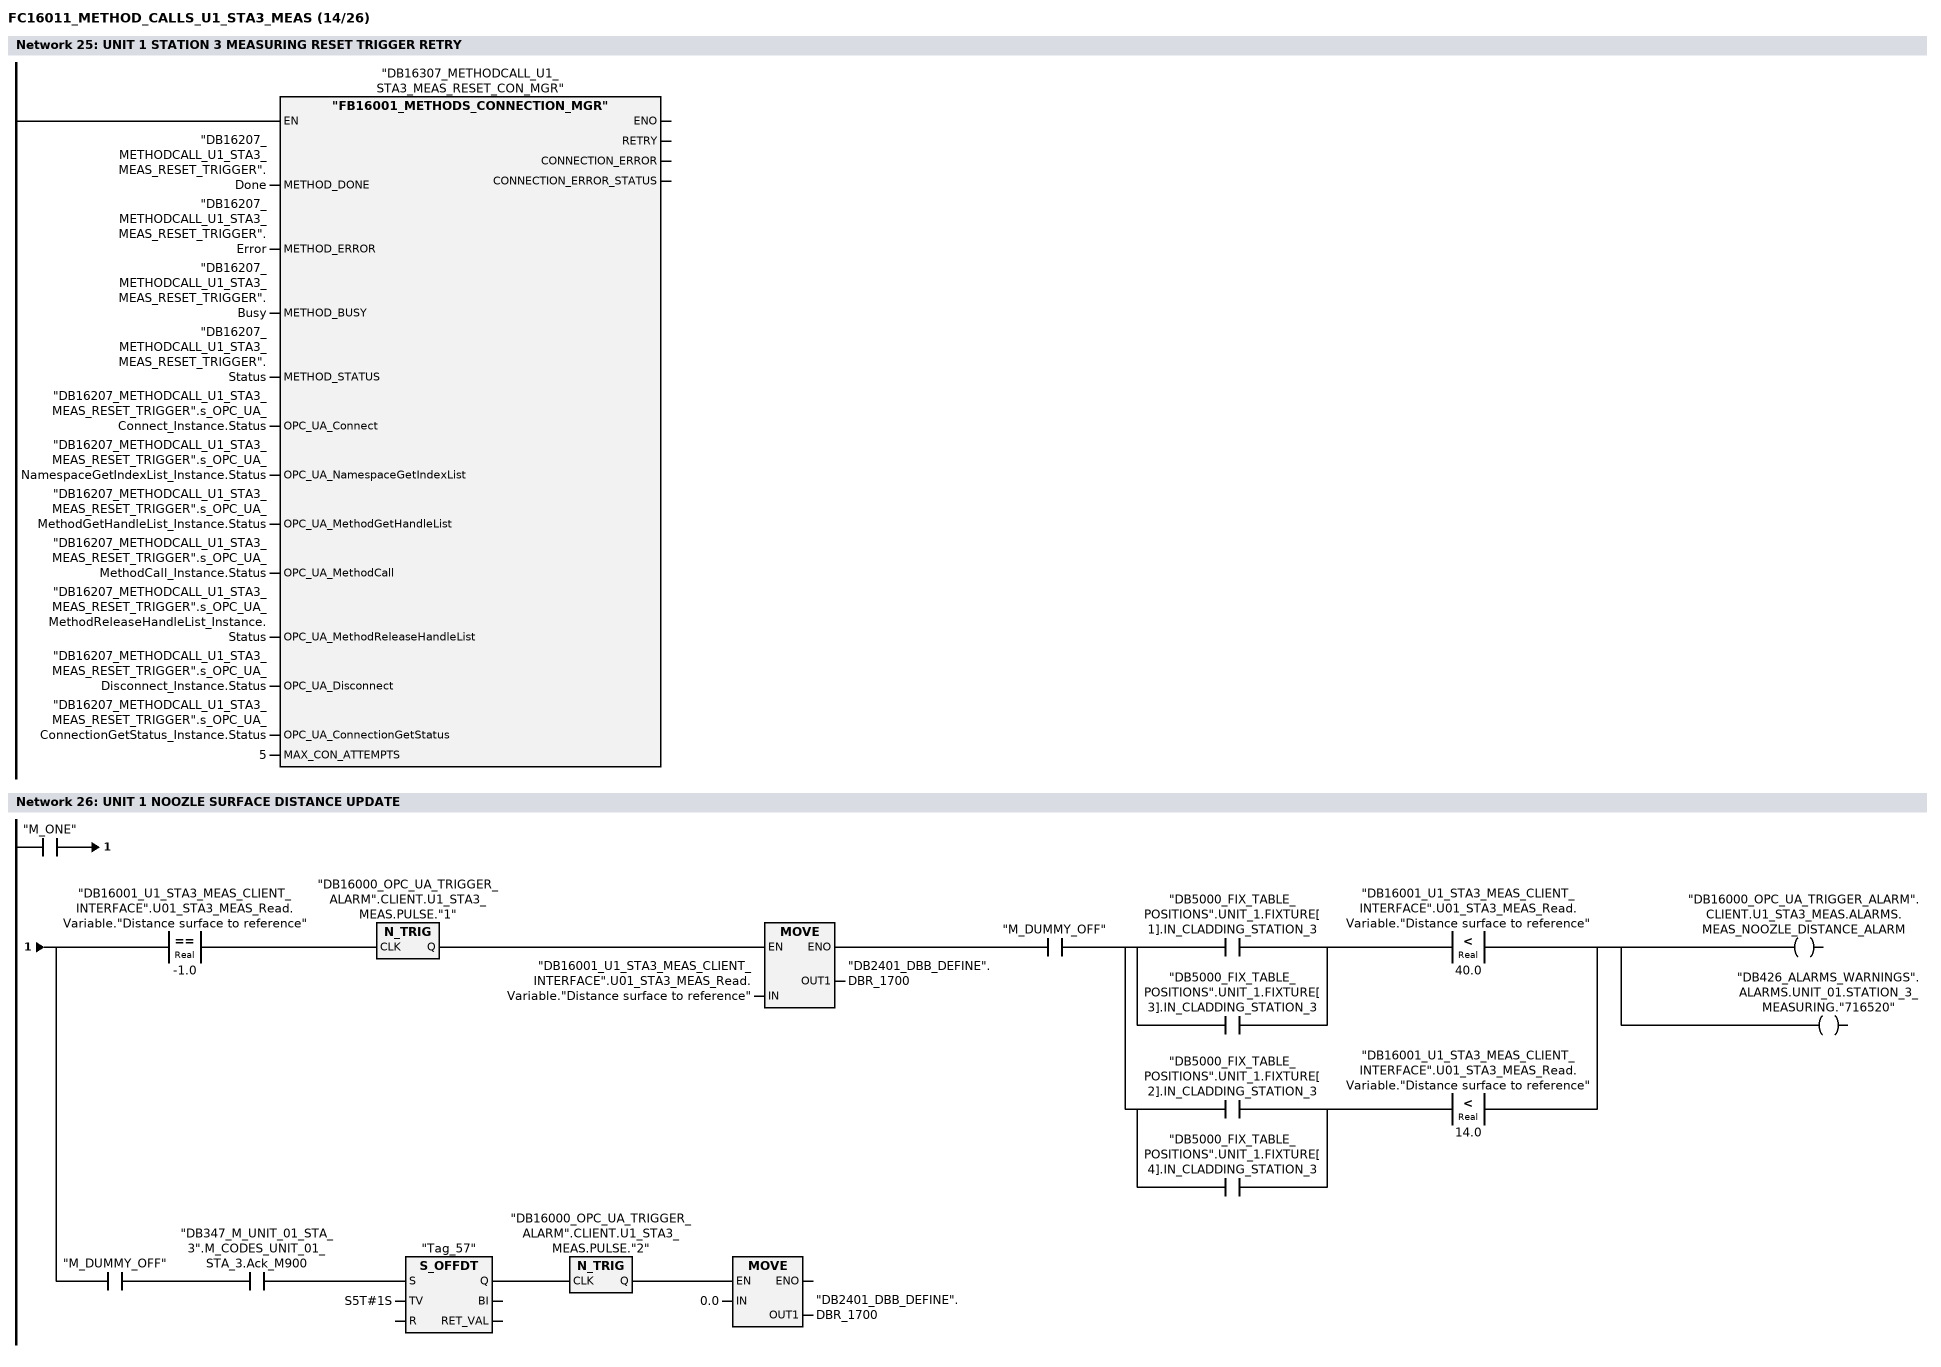
   RUNG wire#powerrail
      "DB16307_METHODCALL_U1_STA3_MEAS_RESET_CON_MGR"(METHOD_DONE := "DB16207_METHODCALL_U1_STA3_MEAS_RESET_TRIGGER".Done, METHOD_ERROR := "DB16207_METHODCALL_U1_STA3_MEAS_RESET_TRIGGER".Error, METHOD_BUSY := "DB16207_METHODCALL_U1_STA3_MEAS_RESET_TRIGGER".Busy, METHOD_STATUS := "DB16207_METHODCALL_U1_STA3_MEAS_RESET_TRIGGER".Status, OPC_UA_Connect := "DB16207_METHODCALL_U1_STA3_MEAS_RESET_TRIGGER".s_OPC_UA_Connect_Instance.Status, OPC_UA_NamespaceGetIndexList := "DB16207_METHODCALL_U1_STA3_MEAS_RESET_TRIGGER".s_OPC_UA_NamespaceGetIndexList_Instance.Status, OPC_UA_MethodGetHandleList := "DB16207_METHODCALL_U1_STA3_MEAS_RESET_TRIGGER".s_OPC_UA_MethodGetHandleList_Instance.Status, OPC_UA_MethodCall := "DB16207_METHODCALL_U1_STA3_MEAS_RESET_TRIGGER".s_OPC_UA_MethodCall_Instance.Status, OPC_UA_MethodReleaseHandleList := "DB16207_METHODCALL_U1_STA3_MEAS_RESET_TRIGGER".s_OPC_UA_MethodReleaseHandleList_Instance.Status, OPC_UA_Disconnect := "DB16207_METHODCALL_U1_STA3_MEAS_RESET_TRIGGER".s_OPC_UA_Disconnect_Instance.Status, OPC_UA_ConnectionGetStatus := "DB16207_METHODCALL_U1_STA3_MEAS_RESET_TRIGGER".s_OPC_UA_ConnectionGetStatus_Instance.Status, MAX_CON_ATTEMPTS := 5, RETRY =>, CONNECTION_ERROR =>, CONNECTION_ERROR_STATUS =>)
   END_RUNG
   // the same network as SCL:
   "DB16307_METHODCALL_U1_STA3_MEAS_RESET_CON_MGR"(METHOD_DONE := "DB16207_METHODCALL_U1_STA3_MEAS_RESET_TRIGGER".Done,   // "FB16001_METHODS_CONNECTION_MGR"
                           METHOD_ERROR := "DB16207_METHODCALL_U1_STA3_MEAS_RESET_TRIGGER".Error,
                           METHOD_BUSY := "DB16207_METHODCALL_U1_STA3_MEAS_RESET_TRIGGER".Busy,
                           METHOD_STATUS := "DB16207_METHODCALL_U1_STA3_MEAS_RESET_TRIGGER".Status,
                           OPC_UA_Connect := "DB16207_METHODCALL_U1_STA3_MEAS_RESET_TRIGGER".s_OPC_UA_Connect_Instance.Status,
                           OPC_UA_NamespaceGetIndexList := "DB16207_METHODCALL_U1_STA3_MEAS_RESET_TRIGGER".s_OPC_UA_NamespaceGetIndexList_Instance.Status,
                           OPC_UA_MethodGetHandleList := "DB16207_METHODCALL_U1_STA3_MEAS_RESET_TRIGGER".s_OPC_UA_MethodGetHandleList_Instance.Status,
                           OPC_UA_MethodCall := "DB16207_METHODCALL_U1_STA3_MEAS_RESET_TRIGGER".s_OPC_UA_MethodCall_Instance.Status,
                           OPC_UA_MethodReleaseHandleList := "DB16207_METHODCALL_U1_STA3_MEAS_RESET_TRIGGER".s_OPC_UA_MethodReleaseHandleList_Instance.Status,
                           OPC_UA_Disconnect := "DB16207_METHODCALL_U1_STA3_MEAS_RESET_TRIGGER".s_OPC_UA_Disconnect_Instance.Status,
                           OPC_UA_ConnectionGetStatus := "DB16207_METHODCALL_U1_STA3_MEAS_RESET_TRIGGER".s_OPC_UA_ConnectionGetStatus_Instance.Status,
                           MAX_CON_ATTEMPTS := 5);
END_REGION

REGION Network 26: UNIT 1 NOOZLE SURFACE DISTANCE UPDATE
   RUNG wire#powerrail
      Contact( "M_ONE" )
      wire#w1
      { S7_Templates := "SrcType := Real" } EQ_Contact(in1 := "DB16001_U1_STA3_MEAS_CLIENT_INTERFACE".U01_STA3_MEAS_Read.Variable."Distance surface to reference", in2 := -1.0)
      N_Trig( "DB16000_OPC_UA_TRIGGER_ALARM".CLIENT.U1_STA3_MEAS.PULSE."1" )
      Move(in := "DB16001_U1_STA3_MEAS_CLIENT_INTERFACE".U01_STA3_MEAS_Read.Variable."Distance surface to reference", out1 => "DB2401_DBB_DEFINE".DBR_1700)
      Contact( "M_DUMMY_OFF" )
      wire#w2
      Contact( "DB5000_FIX_TABLE_POSITIONS".UNIT_1.FIXTURE[1].IN_CLADDING_STATION_3 )
      wire#w3
      { S7_Templates := "SrcType := Real" } LT_Contact(in1 := "DB16001_U1_STA3_MEAS_CLIENT_INTERFACE".U01_STA3_MEAS_Read.Variable."Distance surface to reference", in2 := 40.0)
      wire#w4
      Coil( "DB16000_OPC_UA_TRIGGER_ALARM".CLIENT.U1_STA3_MEAS.ALARMS.MEAS_NOOZLE_DISTANCE_ALARM )
   END_RUNG
   RUNG wire#w2
      Contact( "DB5000_FIX_TABLE_POSITIONS".UNIT_1.FIXTURE[3].IN_CLADDING_STATION_3 )
   END_RUNG wire#w3
   RUNG wire#w2
      Contact( "DB5000_FIX_TABLE_POSITIONS".UNIT_1.FIXTURE[2].IN_CLADDING_STATION_3 )
      wire#w5
      { S7_Templates := "SrcType := Real" } LT_Contact(in1 := "DB16001_U1_STA3_MEAS_CLIENT_INTERFACE".U01_STA3_MEAS_Read.Variable."Distance surface to reference", in2 := 14.0)
   END_RUNG wire#w4
   RUNG wire#w2
      Contact( "DB5000_FIX_TABLE_POSITIONS".UNIT_1.FIXTURE[4].IN_CLADDING_STATION_3 )
   END_RUNG wire#w5
   RUNG wire#w4
      Coil( "DB426_ALARMS_WARNINGS".ALARMS.UNIT_01.STATION_3_MEASURING."716520" )
   END_RUNG
   RUNG wire#w1
      Contact( "M_DUMMY_OFF" )
      Contact( "DB347_M_UNIT_01_STA_3".M_CODES_UNIT_01_STA_3.Ack_M900 )
      S_OFFDT(T_NO := "Tag_57", TV := S5T#1S, R :=, BI =>, RET_VAL =>)
      N_Trig( "DB16000_OPC_UA_TRIGGER_ALARM".CLIENT.U1_STA3_MEAS.PULSE."2" )
      Move(in := 0.0, out1 => "DB2401_DBB_DEFINE".DBR_1700)
   END_RUNG
   // the same network as SCL:
   #_w1 := "M_ONE" AND ("DB16001_U1_STA3_MEAS_CLIENT_INTERFACE".U01_STA3_MEAS_Read.Variable."Distance surface to reference" = (-1.0));
   #_w2 := NOT #_w1 AND "DB16000_OPC_UA_TRIGGER_ALARM".CLIENT.U1_STA3_MEAS.PULSE."1";   // falling edge
   "DB16000_OPC_UA_TRIGGER_ALARM".CLIENT.U1_STA3_MEAS.PULSE."1" := #_w1;
   IF #_w2 THEN
       "DB2401_DBB_DEFINE".DBR_1700 := "DB16001_U1_STA3_MEAS_CLIENT_INTERFACE".U01_STA3_MEAS_Read.Variable."Distance surface to reference";
   END_IF;
   "DB16000_OPC_UA_TRIGGER_ALARM".CLIENT.U1_STA3_MEAS.ALARMS.MEAS_NOOZLE_DISTANCE_ALARM := #_w2 AND "M_DUMMY_OFF" AND ((("DB5000_FIX_TABLE_POSITIONS".UNIT_1.FIXTURE[1].IN_CLADDING_STATION_3 OR "DB5000_FIX_TABLE_POSITIONS".UNIT_1.FIXTURE[3].IN_CLADDING_STATION_3) AND ("DB16001_U1_STA3_MEAS_CLIENT_INTERFACE".U01_STA3_MEAS_Read.Variable."Distance surface to reference" < 40.0)) OR (("DB5000_FIX_TABLE_POSITIONS".UNIT_1.FIXTURE[2].IN_CLADDING_STATION_3 OR "DB5000_FIX_TABLE_POSITIONS".UNIT_1.FIXTURE[4].IN_CLADDING_STATION_3) AND ("DB16001_U1_STA3_MEAS_CLIENT_INTERFACE".U01_STA3_MEAS_Read.Variable."Distance surface to reference" < 14.0)));
   "DB426_ALARMS_WARNINGS".ALARMS.UNIT_01.STATION_3_MEASURING."716520" := "DB16000_OPC_UA_TRIGGER_ALARM".CLIENT.U1_STA3_MEAS.ALARMS.MEAS_NOOZLE_DISTANCE_ALARM;
   #_s5time1 := S_OFFDT(T_NO := "Tag_57",
                        S := "M_ONE" AND "M_DUMMY_OFF" AND "DB347_M_UNIT_01_STA_3".M_CODES_UNIT_01_STA_3.Ack_M900,
                        TV := S5T#1S,
                        Q => #_w3);
   #_w4 := NOT #_w3 AND "DB16000_OPC_UA_TRIGGER_ALARM".CLIENT.U1_STA3_MEAS.PULSE."2";   // falling edge
   "DB16000_OPC_UA_TRIGGER_ALARM".CLIENT.U1_STA3_MEAS.PULSE."2" := #_w3;
   IF #_w4 THEN "DB2401_DBB_DEFINE".DBR_1700 := 0.0; END_IF;
END_REGION

REGION Network 27: UNIT 1 FIXTURES CALIBRATION STATUS UPDATE
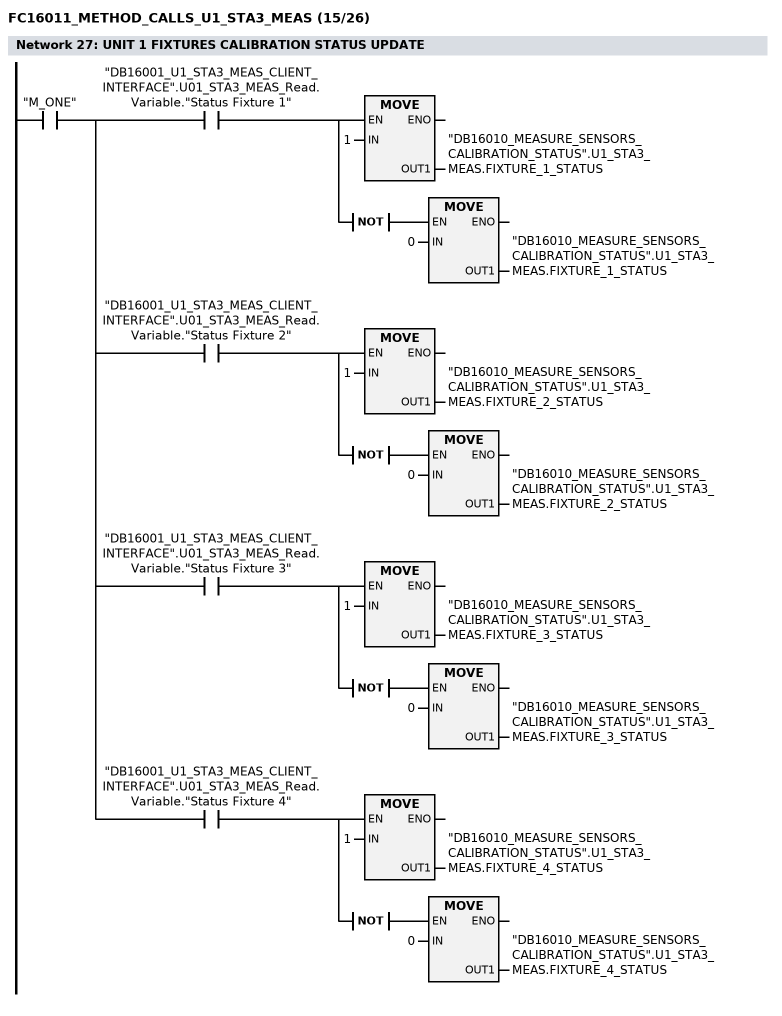
   RUNG wire#powerrail
      Contact( "M_ONE" )
      wire#w1
      Contact( "DB16001_U1_STA3_MEAS_CLIENT_INTERFACE".U01_STA3_MEAS_Read.Variable."Status Fixture 1" )
      wire#w2
      Move(in := 1, out1 => "DB16010_MEASURE_SENSORS_CALIBRATION_STATUS".U1_STA3_MEAS.FIXTURE_1_STATUS)
   END_RUNG
   RUNG wire#w2
      Not()
      Move(in := 0, out1 => "DB16010_MEASURE_SENSORS_CALIBRATION_STATUS".U1_STA3_MEAS.FIXTURE_1_STATUS)
   END_RUNG
   RUNG wire#w1
      Contact( "DB16001_U1_STA3_MEAS_CLIENT_INTERFACE".U01_STA3_MEAS_Read.Variable."Status Fixture 2" )
      wire#w3
      Move(in := 1, out1 => "DB16010_MEASURE_SENSORS_CALIBRATION_STATUS".U1_STA3_MEAS.FIXTURE_2_STATUS)
   END_RUNG
   RUNG wire#w3
      Not()
      Move(in := 0, out1 => "DB16010_MEASURE_SENSORS_CALIBRATION_STATUS".U1_STA3_MEAS.FIXTURE_2_STATUS)
   END_RUNG
   RUNG wire#w1
      Contact( "DB16001_U1_STA3_MEAS_CLIENT_INTERFACE".U01_STA3_MEAS_Read.Variable."Status Fixture 3" )
      wire#w4
      Move(in := 1, out1 => "DB16010_MEASURE_SENSORS_CALIBRATION_STATUS".U1_STA3_MEAS.FIXTURE_3_STATUS)
   END_RUNG
   RUNG wire#w4
      Not()
      Move(in := 0, out1 => "DB16010_MEASURE_SENSORS_CALIBRATION_STATUS".U1_STA3_MEAS.FIXTURE_3_STATUS)
   END_RUNG
   RUNG wire#w1
      Contact( "DB16001_U1_STA3_MEAS_CLIENT_INTERFACE".U01_STA3_MEAS_Read.Variable."Status Fixture 4" )
      wire#w5
      Move(in := 1, out1 => "DB16010_MEASURE_SENSORS_CALIBRATION_STATUS".U1_STA3_MEAS.FIXTURE_4_STATUS)
   END_RUNG
   RUNG wire#w5
      Not()
      Move(in := 0, out1 => "DB16010_MEASURE_SENSORS_CALIBRATION_STATUS".U1_STA3_MEAS.FIXTURE_4_STATUS)
   END_RUNG
   // the same network as SCL:
   #_w1 := "M_ONE" AND "DB16001_U1_STA3_MEAS_CLIENT_INTERFACE".U01_STA3_MEAS_Read.Variable."Status Fixture 1";
   IF #_w1 THEN "DB16010_MEASURE_SENSORS_CALIBRATION_STATUS".U1_STA3_MEAS.FIXTURE_1_STATUS := 1; END_IF;
   IF NOT #_w1 THEN "DB16010_MEASURE_SENSORS_CALIBRATION_STATUS".U1_STA3_MEAS.FIXTURE_1_STATUS := 0; END_IF;
   #_w2 := "M_ONE" AND "DB16001_U1_STA3_MEAS_CLIENT_INTERFACE".U01_STA3_MEAS_Read.Variable."Status Fixture 2";
   IF #_w2 THEN "DB16010_MEASURE_SENSORS_CALIBRATION_STATUS".U1_STA3_MEAS.FIXTURE_2_STATUS := 1; END_IF;
   IF NOT #_w2 THEN "DB16010_MEASURE_SENSORS_CALIBRATION_STATUS".U1_STA3_MEAS.FIXTURE_2_STATUS := 0; END_IF;
   #_w3 := "M_ONE" AND "DB16001_U1_STA3_MEAS_CLIENT_INTERFACE".U01_STA3_MEAS_Read.Variable."Status Fixture 3";
   IF #_w3 THEN "DB16010_MEASURE_SENSORS_CALIBRATION_STATUS".U1_STA3_MEAS.FIXTURE_3_STATUS := 1; END_IF;
   IF NOT #_w3 THEN "DB16010_MEASURE_SENSORS_CALIBRATION_STATUS".U1_STA3_MEAS.FIXTURE_3_STATUS := 0; END_IF;
   #_w4 := "M_ONE" AND "DB16001_U1_STA3_MEAS_CLIENT_INTERFACE".U01_STA3_MEAS_Read.Variable."Status Fixture 4";
   IF #_w4 THEN "DB16010_MEASURE_SENSORS_CALIBRATION_STATUS".U1_STA3_MEAS.FIXTURE_4_STATUS := 1; END_IF;
   IF NOT #_w4 THEN "DB16010_MEASURE_SENSORS_CALIBRATION_STATUS".U1_STA3_MEAS.FIXTURE_4_STATUS := 0; END_IF;
END_REGION

REGION Network 28: UNIT 1 STATION 3 MEASURING MEASURING NOZZLE SURFACE DISTANCE METHOD CONNECTION ALARM
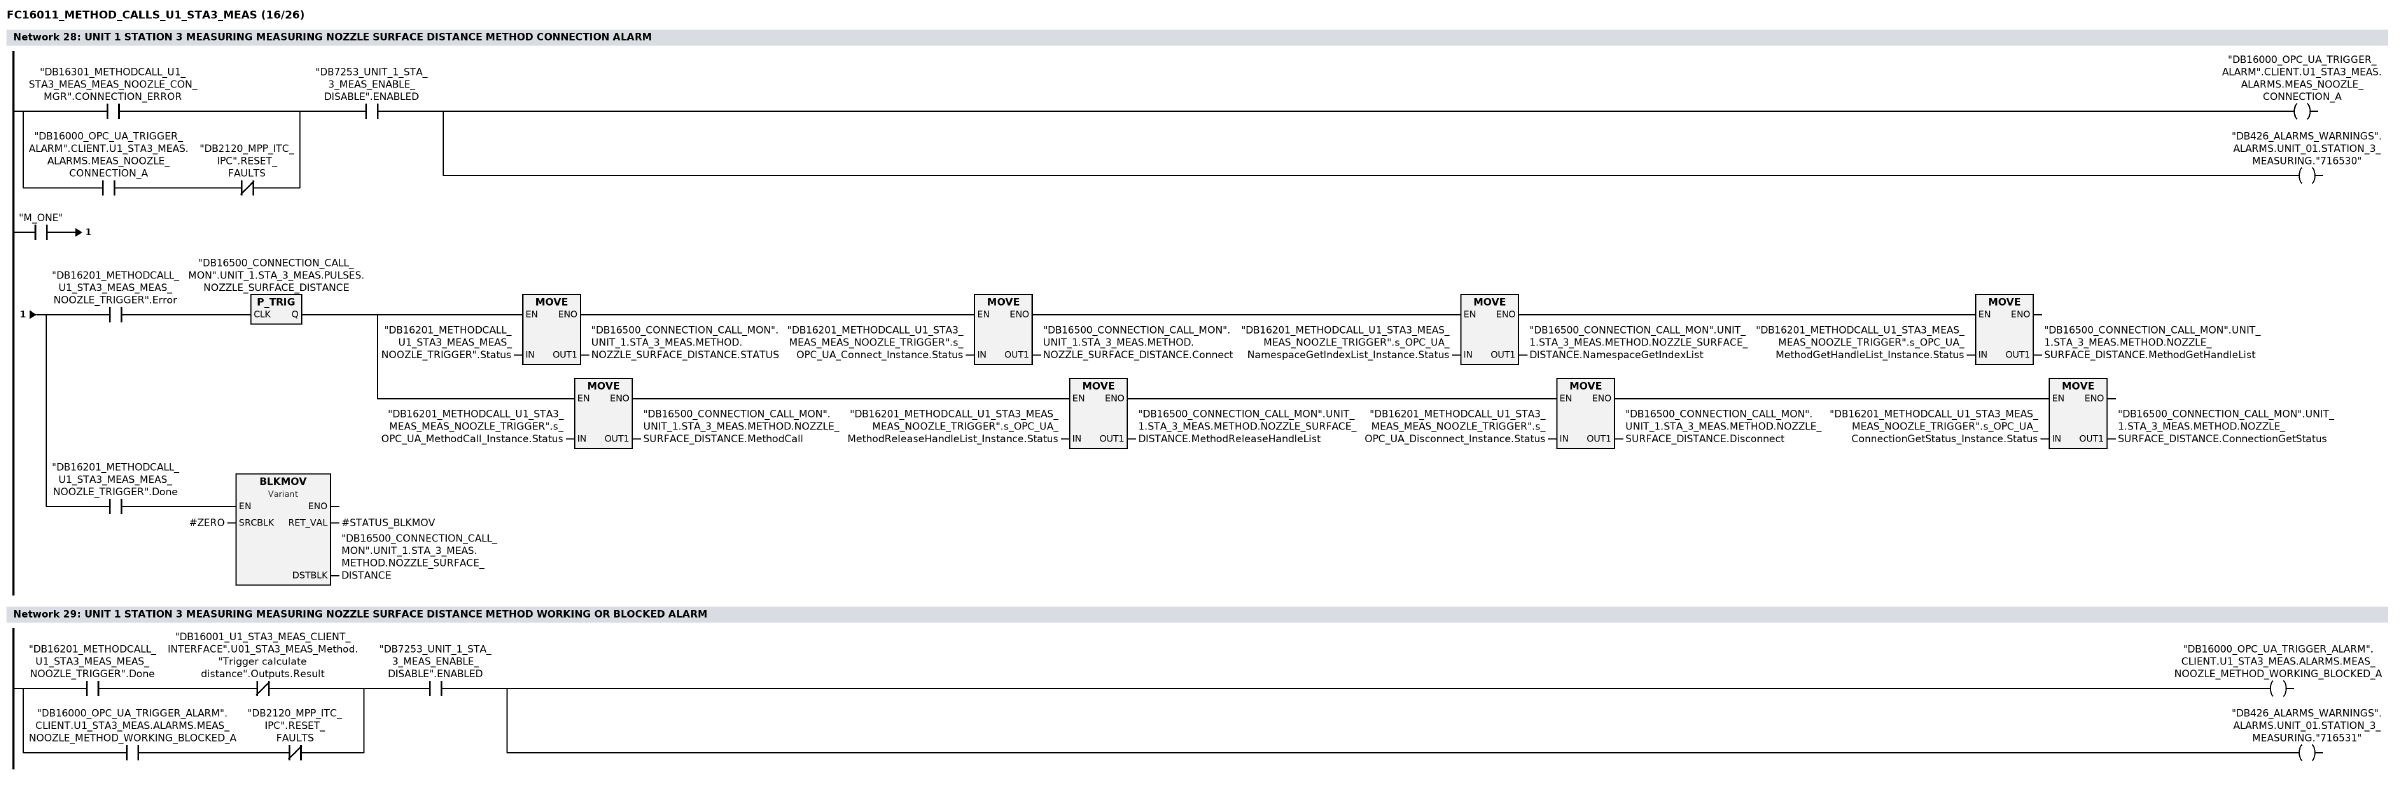
   RUNG wire#powerrail
      Contact( "DB16301_METHODCALL_U1_STA3_MEAS_MEAS_NOOZLE_CON_MGR".CONNECTION_ERROR )
      wire#w1
      Contact( "DB7253_UNIT_1_STA_3_MEAS_ENABLE_DISABLE".ENABLED )
      wire#w2
      Coil( "DB16000_OPC_UA_TRIGGER_ALARM".CLIENT.U1_STA3_MEAS.ALARMS.MEAS_NOOZLE_CONNECTION_A )
   END_RUNG
   RUNG wire#powerrail
      Contact( "DB16000_OPC_UA_TRIGGER_ALARM".CLIENT.U1_STA3_MEAS.ALARMS.MEAS_NOOZLE_CONNECTION_A )
      I_Contact( "DB2120_MPP_ITC_IPC".RESET_FAULTS )
   END_RUNG wire#w1
   RUNG wire#w2
      Coil( "DB426_ALARMS_WARNINGS".ALARMS.UNIT_01.STATION_3_MEASURING."716530" )
   END_RUNG
   RUNG wire#powerrail
      Contact( "M_ONE" )
      wire#w3
      Contact( "DB16201_METHODCALL_U1_STA3_MEAS_MEAS_NOOZLE_TRIGGER".Error )
      P_Trig( "DB16500_CONNECTION_CALL_MON".UNIT_1.STA_3_MEAS.PULSES.NOZZLE_SURFACE_DISTANCE )
      wire#w4
      Move(in := "DB16201_METHODCALL_U1_STA3_MEAS_MEAS_NOOZLE_TRIGGER".Status, out1 => "DB16500_CONNECTION_CALL_MON".UNIT_1.STA_3_MEAS.METHOD.NOZZLE_SURFACE_DISTANCE.STATUS)
      Move(in := "DB16201_METHODCALL_U1_STA3_MEAS_MEAS_NOOZLE_TRIGGER".s_OPC_UA_Connect_Instance.Status, out1 => "DB16500_CONNECTION_CALL_MON".UNIT_1.STA_3_MEAS.METHOD.NOZZLE_SURFACE_DISTANCE.Connect)
      Move(in := "DB16201_METHODCALL_U1_STA3_MEAS_MEAS_NOOZLE_TRIGGER".s_OPC_UA_NamespaceGetIndexList_Instance.Status, out1 => "DB16500_CONNECTION_CALL_MON".UNIT_1.STA_3_MEAS.METHOD.NOZZLE_SURFACE_DISTANCE.NamespaceGetIndexList)
      Move(in := "DB16201_METHODCALL_U1_STA3_MEAS_MEAS_NOOZLE_TRIGGER".s_OPC_UA_MethodGetHandleList_Instance.Status, out1 => "DB16500_CONNECTION_CALL_MON".UNIT_1.STA_3_MEAS.METHOD.NOZZLE_SURFACE_DISTANCE.MethodGetHandleList)
   END_RUNG
   RUNG wire#w4
      Move(in := "DB16201_METHODCALL_U1_STA3_MEAS_MEAS_NOOZLE_TRIGGER".s_OPC_UA_MethodCall_Instance.Status, out1 => "DB16500_CONNECTION_CALL_MON".UNIT_1.STA_3_MEAS.METHOD.NOZZLE_SURFACE_DISTANCE.MethodCall)
      Move(in := "DB16201_METHODCALL_U1_STA3_MEAS_MEAS_NOOZLE_TRIGGER".s_OPC_UA_MethodReleaseHandleList_Instance.Status, out1 => "DB16500_CONNECTION_CALL_MON".UNIT_1.STA_3_MEAS.METHOD.NOZZLE_SURFACE_DISTANCE.MethodReleaseHandleList)
      Move(in := "DB16201_METHODCALL_U1_STA3_MEAS_MEAS_NOOZLE_TRIGGER".s_OPC_UA_Disconnect_Instance.Status, out1 => "DB16500_CONNECTION_CALL_MON".UNIT_1.STA_3_MEAS.METHOD.NOZZLE_SURFACE_DISTANCE.Disconnect)
      Move(in := "DB16201_METHODCALL_U1_STA3_MEAS_MEAS_NOOZLE_TRIGGER".s_OPC_UA_ConnectionGetStatus_Instance.Status, out1 => "DB16500_CONNECTION_CALL_MON".UNIT_1.STA_3_MEAS.METHOD.NOZZLE_SURFACE_DISTANCE.ConnectionGetStatus)
   END_RUNG
   RUNG wire#w3
      Contact( "DB16201_METHODCALL_U1_STA3_MEAS_MEAS_NOOZLE_TRIGGER".Done )
      { S7_Templates := "blk_type := Variant" } BLKMOV(SRCBLK := #ZERO, RET_VAL => #STATUS_BLKMOV, DSTBLK => "DB16500_CONNECTION_CALL_MON".UNIT_1.STA_3_MEAS.METHOD.NOZZLE_SURFACE_DISTANCE)
   END_RUNG
   // the same network as SCL:
   "DB16000_OPC_UA_TRIGGER_ALARM".CLIENT.U1_STA3_MEAS.ALARMS.MEAS_NOOZLE_CONNECTION_A := ("DB16301_METHODCALL_U1_STA3_MEAS_MEAS_NOOZLE_CON_MGR".CONNECTION_ERROR OR ("DB16000_OPC_UA_TRIGGER_ALARM".CLIENT.U1_STA3_MEAS.ALARMS.MEAS_NOOZLE_CONNECTION_A AND NOT "DB2120_MPP_ITC_IPC".RESET_FAULTS)) AND "DB7253_UNIT_1_STA_3_MEAS_ENABLE_DISABLE".ENABLED;
   "DB426_ALARMS_WARNINGS".ALARMS.UNIT_01.STATION_3_MEASURING."716530" := "DB16000_OPC_UA_TRIGGER_ALARM".CLIENT.U1_STA3_MEAS.ALARMS.MEAS_NOOZLE_CONNECTION_A;
   #_w1 := "M_ONE" AND "DB16201_METHODCALL_U1_STA3_MEAS_MEAS_NOOZLE_TRIGGER".Error;
   #_w2 := #_w1 AND NOT "DB16500_CONNECTION_CALL_MON".UNIT_1.STA_3_MEAS.PULSES.NOZZLE_SURFACE_DISTANCE;   // rising edge
   "DB16500_CONNECTION_CALL_MON".UNIT_1.STA_3_MEAS.PULSES.NOZZLE_SURFACE_DISTANCE := #_w1;
   IF #_w2 THEN
       "DB16500_CONNECTION_CALL_MON".UNIT_1.STA_3_MEAS.METHOD.NOZZLE_SURFACE_DISTANCE.STATUS := "DB16201_METHODCALL_U1_STA3_MEAS_MEAS_NOOZLE_TRIGGER".Status;
       "DB16500_CONNECTION_CALL_MON".UNIT_1.STA_3_MEAS.METHOD.NOZZLE_SURFACE_DISTANCE.Connect := "DB16201_METHODCALL_U1_STA3_MEAS_MEAS_NOOZLE_TRIGGER".s_OPC_UA_Connect_Instance.Status;
       "DB16500_CONNECTION_CALL_MON".UNIT_1.STA_3_MEAS.METHOD.NOZZLE_SURFACE_DISTANCE.NamespaceGetIndexList := "DB16201_METHODCALL_U1_STA3_MEAS_MEAS_NOOZLE_TRIGGER".s_OPC_UA_NamespaceGetIndexList_Instance.Status;
       "DB16500_CONNECTION_CALL_MON".UNIT_1.STA_3_MEAS.METHOD.NOZZLE_SURFACE_DISTANCE.MethodGetHandleList := "DB16201_METHODCALL_U1_STA3_MEAS_MEAS_NOOZLE_TRIGGER".s_OPC_UA_MethodGetHandleList_Instance.Status;
       "DB16500_CONNECTION_CALL_MON".UNIT_1.STA_3_MEAS.METHOD.NOZZLE_SURFACE_DISTANCE.MethodCall := "DB16201_METHODCALL_U1_STA3_MEAS_MEAS_NOOZLE_TRIGGER".s_OPC_UA_MethodCall_Instance.Status;
       "DB16500_CONNECTION_CALL_MON".UNIT_1.STA_3_MEAS.METHOD.NOZZLE_SURFACE_DISTANCE.MethodReleaseHandleList := "DB16201_METHODCALL_U1_STA3_MEAS_MEAS_NOOZLE_TRIGGER".s_OPC_UA_MethodReleaseHandleList_Instance.Status;
       "DB16500_CONNECTION_CALL_MON".UNIT_1.STA_3_MEAS.METHOD.NOZZLE_SURFACE_DISTANCE.Disconnect := "DB16201_METHODCALL_U1_STA3_MEAS_MEAS_NOOZLE_TRIGGER".s_OPC_UA_Disconnect_Instance.Status;
       "DB16500_CONNECTION_CALL_MON".UNIT_1.STA_3_MEAS.METHOD.NOZZLE_SURFACE_DISTANCE.ConnectionGetStatus := "DB16201_METHODCALL_U1_STA3_MEAS_MEAS_NOOZLE_TRIGGER".s_OPC_UA_ConnectionGetStatus_Instance.Status;
   END_IF;
   IF "M_ONE" AND "DB16201_METHODCALL_U1_STA3_MEAS_MEAS_NOOZLE_TRIGGER".Done THEN
       #STATUS_BLKMOV := BLKMOV(SRCBLK := #ZERO,
                               DSTBLK => "DB16500_CONNECTION_CALL_MON".UNIT_1.STA_3_MEAS.METHOD.NOZZLE_SURFACE_DISTANCE);
   END_IF;
END_REGION

REGION Network 29: UNIT 1 STATION 3 MEASURING MEASURING NOZZLE SURFACE DISTANCE METHOD WORKING OR BLOCKED ALARM
   RUNG wire#powerrail
      Contact( "DB16201_METHODCALL_U1_STA3_MEAS_MEAS_NOOZLE_TRIGGER".Done )
      I_Contact( "DB16001_U1_STA3_MEAS_CLIENT_INTERFACE".U01_STA3_MEAS_Method."Trigger calculate distance".Outputs.Result )
      wire#w1
      Contact( "DB7253_UNIT_1_STA_3_MEAS_ENABLE_DISABLE".ENABLED )
      wire#w2
      Coil( "DB16000_OPC_UA_TRIGGER_ALARM".CLIENT.U1_STA3_MEAS.ALARMS.MEAS_NOOZLE_METHOD_WORKING_BLOCKED_A )
   END_RUNG
   RUNG wire#powerrail
      Contact( "DB16000_OPC_UA_TRIGGER_ALARM".CLIENT.U1_STA3_MEAS.ALARMS.MEAS_NOOZLE_METHOD_WORKING_BLOCKED_A )
      I_Contact( "DB2120_MPP_ITC_IPC".RESET_FAULTS )
   END_RUNG wire#w1
   RUNG wire#w2
      Coil( "DB426_ALARMS_WARNINGS".ALARMS.UNIT_01.STATION_3_MEASURING."716531" )
   END_RUNG
   // the same network as SCL:
   "DB16000_OPC_UA_TRIGGER_ALARM".CLIENT.U1_STA3_MEAS.ALARMS.MEAS_NOOZLE_METHOD_WORKING_BLOCKED_A := (("DB16201_METHODCALL_U1_STA3_MEAS_MEAS_NOOZLE_TRIGGER".Done AND NOT "DB16001_U1_STA3_MEAS_CLIENT_INTERFACE".U01_STA3_MEAS_Method."Trigger calculate distance".Outputs.Result) OR ("DB16000_OPC_UA_TRIGGER_ALARM".CLIENT.U1_STA3_MEAS.ALARMS.MEAS_NOOZLE_METHOD_WORKING_BLOCKED_A AND NOT "DB2120_MPP_ITC_IPC".RESET_FAULTS)) AND "DB7253_UNIT_1_STA_3_MEAS_ENABLE_DISABLE".ENABLED;
   "DB426_ALARMS_WARNINGS".ALARMS.UNIT_01.STATION_3_MEASURING."716531" := "DB16000_OPC_UA_TRIGGER_ALARM".CLIENT.U1_STA3_MEAS.ALARMS.MEAS_NOOZLE_METHOD_WORKING_BLOCKED_A;
END_REGION

REGION Network 30: UNIT 1 STATION 3 MEASURING START MEASURING LAYER THICKNESS METHOD CONNECTION ALARM
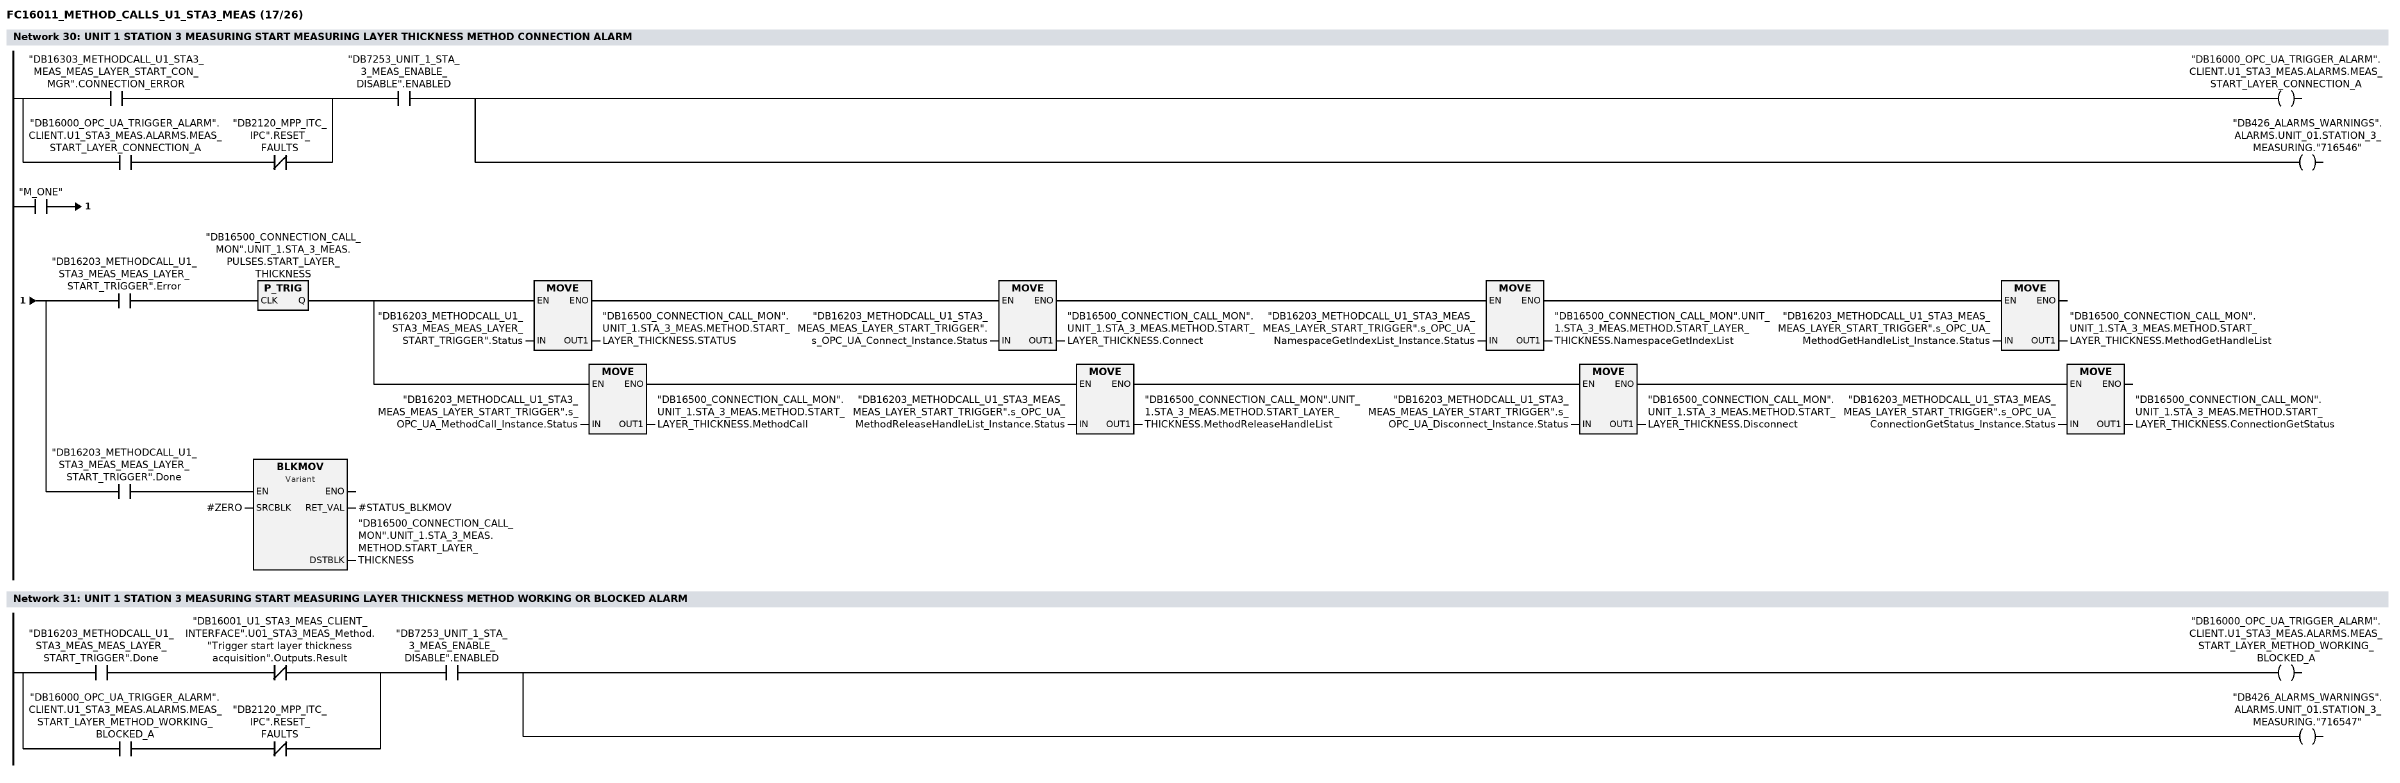
   RUNG wire#powerrail
      Contact( "DB16303_METHODCALL_U1_STA3_MEAS_MEAS_LAYER_START_CON_MGR".CONNECTION_ERROR )
      wire#w1
      Contact( "DB7253_UNIT_1_STA_3_MEAS_ENABLE_DISABLE".ENABLED )
      wire#w2
      Coil( "DB16000_OPC_UA_TRIGGER_ALARM".CLIENT.U1_STA3_MEAS.ALARMS.MEAS_START_LAYER_CONNECTION_A )
   END_RUNG
   RUNG wire#powerrail
      Contact( "DB16000_OPC_UA_TRIGGER_ALARM".CLIENT.U1_STA3_MEAS.ALARMS.MEAS_START_LAYER_CONNECTION_A )
      I_Contact( "DB2120_MPP_ITC_IPC".RESET_FAULTS )
   END_RUNG wire#w1
   RUNG wire#w2
      Coil( "DB426_ALARMS_WARNINGS".ALARMS.UNIT_01.STATION_3_MEASURING."716546" )
   END_RUNG
   RUNG wire#powerrail
      Contact( "M_ONE" )
      wire#w3
      Contact( "DB16203_METHODCALL_U1_STA3_MEAS_MEAS_LAYER_START_TRIGGER".Error )
      P_Trig( "DB16500_CONNECTION_CALL_MON".UNIT_1.STA_3_MEAS.PULSES.START_LAYER_THICKNESS )
      wire#w4
      Move(in := "DB16203_METHODCALL_U1_STA3_MEAS_MEAS_LAYER_START_TRIGGER".Status, out1 => "DB16500_CONNECTION_CALL_MON".UNIT_1.STA_3_MEAS.METHOD.START_LAYER_THICKNESS.STATUS)
      Move(in := "DB16203_METHODCALL_U1_STA3_MEAS_MEAS_LAYER_START_TRIGGER".s_OPC_UA_Connect_Instance.Status, out1 => "DB16500_CONNECTION_CALL_MON".UNIT_1.STA_3_MEAS.METHOD.START_LAYER_THICKNESS.Connect)
      Move(in := "DB16203_METHODCALL_U1_STA3_MEAS_MEAS_LAYER_START_TRIGGER".s_OPC_UA_NamespaceGetIndexList_Instance.Status, out1 => "DB16500_CONNECTION_CALL_MON".UNIT_1.STA_3_MEAS.METHOD.START_LAYER_THICKNESS.NamespaceGetIndexList)
      Move(in := "DB16203_METHODCALL_U1_STA3_MEAS_MEAS_LAYER_START_TRIGGER".s_OPC_UA_MethodGetHandleList_Instance.Status, out1 => "DB16500_CONNECTION_CALL_MON".UNIT_1.STA_3_MEAS.METHOD.START_LAYER_THICKNESS.MethodGetHandleList)
   END_RUNG
   RUNG wire#w4
      Move(in := "DB16203_METHODCALL_U1_STA3_MEAS_MEAS_LAYER_START_TRIGGER".s_OPC_UA_MethodCall_Instance.Status, out1 => "DB16500_CONNECTION_CALL_MON".UNIT_1.STA_3_MEAS.METHOD.START_LAYER_THICKNESS.MethodCall)
      Move(in := "DB16203_METHODCALL_U1_STA3_MEAS_MEAS_LAYER_START_TRIGGER".s_OPC_UA_MethodReleaseHandleList_Instance.Status, out1 => "DB16500_CONNECTION_CALL_MON".UNIT_1.STA_3_MEAS.METHOD.START_LAYER_THICKNESS.MethodReleaseHandleList)
      Move(in := "DB16203_METHODCALL_U1_STA3_MEAS_MEAS_LAYER_START_TRIGGER".s_OPC_UA_Disconnect_Instance.Status, out1 => "DB16500_CONNECTION_CALL_MON".UNIT_1.STA_3_MEAS.METHOD.START_LAYER_THICKNESS.Disconnect)
      Move(in := "DB16203_METHODCALL_U1_STA3_MEAS_MEAS_LAYER_START_TRIGGER".s_OPC_UA_ConnectionGetStatus_Instance.Status, out1 => "DB16500_CONNECTION_CALL_MON".UNIT_1.STA_3_MEAS.METHOD.START_LAYER_THICKNESS.ConnectionGetStatus)
   END_RUNG
   RUNG wire#w3
      Contact( "DB16203_METHODCALL_U1_STA3_MEAS_MEAS_LAYER_START_TRIGGER".Done )
      { S7_Templates := "blk_type := Variant" } BLKMOV(SRCBLK := #ZERO, RET_VAL => #STATUS_BLKMOV, DSTBLK => "DB16500_CONNECTION_CALL_MON".UNIT_1.STA_3_MEAS.METHOD.START_LAYER_THICKNESS)
   END_RUNG
   // the same network as SCL:
   "DB16000_OPC_UA_TRIGGER_ALARM".CLIENT.U1_STA3_MEAS.ALARMS.MEAS_START_LAYER_CONNECTION_A := ("DB16303_METHODCALL_U1_STA3_MEAS_MEAS_LAYER_START_CON_MGR".CONNECTION_ERROR OR ("DB16000_OPC_UA_TRIGGER_ALARM".CLIENT.U1_STA3_MEAS.ALARMS.MEAS_START_LAYER_CONNECTION_A AND NOT "DB2120_MPP_ITC_IPC".RESET_FAULTS)) AND "DB7253_UNIT_1_STA_3_MEAS_ENABLE_DISABLE".ENABLED;
   "DB426_ALARMS_WARNINGS".ALARMS.UNIT_01.STATION_3_MEASURING."716546" := "DB16000_OPC_UA_TRIGGER_ALARM".CLIENT.U1_STA3_MEAS.ALARMS.MEAS_START_LAYER_CONNECTION_A;
   #_w1 := "M_ONE" AND "DB16203_METHODCALL_U1_STA3_MEAS_MEAS_LAYER_START_TRIGGER".Error;
   #_w2 := #_w1 AND NOT "DB16500_CONNECTION_CALL_MON".UNIT_1.STA_3_MEAS.PULSES.START_LAYER_THICKNESS;   // rising edge
   "DB16500_CONNECTION_CALL_MON".UNIT_1.STA_3_MEAS.PULSES.START_LAYER_THICKNESS := #_w1;
   IF #_w2 THEN
       "DB16500_CONNECTION_CALL_MON".UNIT_1.STA_3_MEAS.METHOD.START_LAYER_THICKNESS.STATUS := "DB16203_METHODCALL_U1_STA3_MEAS_MEAS_LAYER_START_TRIGGER".Status;
       "DB16500_CONNECTION_CALL_MON".UNIT_1.STA_3_MEAS.METHOD.START_LAYER_THICKNESS.Connect := "DB16203_METHODCALL_U1_STA3_MEAS_MEAS_LAYER_START_TRIGGER".s_OPC_UA_Connect_Instance.Status;
       "DB16500_CONNECTION_CALL_MON".UNIT_1.STA_3_MEAS.METHOD.START_LAYER_THICKNESS.NamespaceGetIndexList := "DB16203_METHODCALL_U1_STA3_MEAS_MEAS_LAYER_START_TRIGGER".s_OPC_UA_NamespaceGetIndexList_Instance.Status;
       "DB16500_CONNECTION_CALL_MON".UNIT_1.STA_3_MEAS.METHOD.START_LAYER_THICKNESS.MethodGetHandleList := "DB16203_METHODCALL_U1_STA3_MEAS_MEAS_LAYER_START_TRIGGER".s_OPC_UA_MethodGetHandleList_Instance.Status;
       "DB16500_CONNECTION_CALL_MON".UNIT_1.STA_3_MEAS.METHOD.START_LAYER_THICKNESS.MethodCall := "DB16203_METHODCALL_U1_STA3_MEAS_MEAS_LAYER_START_TRIGGER".s_OPC_UA_MethodCall_Instance.Status;
       "DB16500_CONNECTION_CALL_MON".UNIT_1.STA_3_MEAS.METHOD.START_LAYER_THICKNESS.MethodReleaseHandleList := "DB16203_METHODCALL_U1_STA3_MEAS_MEAS_LAYER_START_TRIGGER".s_OPC_UA_MethodReleaseHandleList_Instance.Status;
       "DB16500_CONNECTION_CALL_MON".UNIT_1.STA_3_MEAS.METHOD.START_LAYER_THICKNESS.Disconnect := "DB16203_METHODCALL_U1_STA3_MEAS_MEAS_LAYER_START_TRIGGER".s_OPC_UA_Disconnect_Instance.Status;
       "DB16500_CONNECTION_CALL_MON".UNIT_1.STA_3_MEAS.METHOD.START_LAYER_THICKNESS.ConnectionGetStatus := "DB16203_METHODCALL_U1_STA3_MEAS_MEAS_LAYER_START_TRIGGER".s_OPC_UA_ConnectionGetStatus_Instance.Status;
   END_IF;
   IF "M_ONE" AND "DB16203_METHODCALL_U1_STA3_MEAS_MEAS_LAYER_START_TRIGGER".Done THEN
       #STATUS_BLKMOV := BLKMOV(SRCBLK := #ZERO,
                               DSTBLK => "DB16500_CONNECTION_CALL_MON".UNIT_1.STA_3_MEAS.METHOD.START_LAYER_THICKNESS);
   END_IF;
END_REGION

REGION Network 31: UNIT 1 STATION 3 MEASURING START MEASURING LAYER THICKNESS METHOD WORKING OR BLOCKED ALARM
   RUNG wire#powerrail
      Contact( "DB16203_METHODCALL_U1_STA3_MEAS_MEAS_LAYER_START_TRIGGER".Done )
      I_Contact( "DB16001_U1_STA3_MEAS_CLIENT_INTERFACE".U01_STA3_MEAS_Method."Trigger start layer thickness acquisition".Outputs.Result )
      wire#w1
      Contact( "DB7253_UNIT_1_STA_3_MEAS_ENABLE_DISABLE".ENABLED )
      wire#w2
      Coil( "DB16000_OPC_UA_TRIGGER_ALARM".CLIENT.U1_STA3_MEAS.ALARMS.MEAS_START_LAYER_METHOD_WORKING_BLOCKED_A )
   END_RUNG
   RUNG wire#powerrail
      Contact( "DB16000_OPC_UA_TRIGGER_ALARM".CLIENT.U1_STA3_MEAS.ALARMS.MEAS_START_LAYER_METHOD_WORKING_BLOCKED_A )
      I_Contact( "DB2120_MPP_ITC_IPC".RESET_FAULTS )
   END_RUNG wire#w1
   RUNG wire#w2
      Coil( "DB426_ALARMS_WARNINGS".ALARMS.UNIT_01.STATION_3_MEASURING."716547" )
   END_RUNG
   // the same network as SCL:
   "DB16000_OPC_UA_TRIGGER_ALARM".CLIENT.U1_STA3_MEAS.ALARMS.MEAS_START_LAYER_METHOD_WORKING_BLOCKED_A := (("DB16203_METHODCALL_U1_STA3_MEAS_MEAS_LAYER_START_TRIGGER".Done AND NOT "DB16001_U1_STA3_MEAS_CLIENT_INTERFACE".U01_STA3_MEAS_Method."Trigger start layer thickness acquisition".Outputs.Result) OR ("DB16000_OPC_UA_TRIGGER_ALARM".CLIENT.U1_STA3_MEAS.ALARMS.MEAS_START_LAYER_METHOD_WORKING_BLOCKED_A AND NOT "DB2120_MPP_ITC_IPC".RESET_FAULTS)) AND "DB7253_UNIT_1_STA_3_MEAS_ENABLE_DISABLE".ENABLED;
   "DB426_ALARMS_WARNINGS".ALARMS.UNIT_01.STATION_3_MEASURING."716547" := "DB16000_OPC_UA_TRIGGER_ALARM".CLIENT.U1_STA3_MEAS.ALARMS.MEAS_START_LAYER_METHOD_WORKING_BLOCKED_A;
END_REGION

REGION Network 32: UNIT 1 STATION 3 MEASURING STOP MEASURING LAYER THICKNESS METHOD CONNECTION ALARM
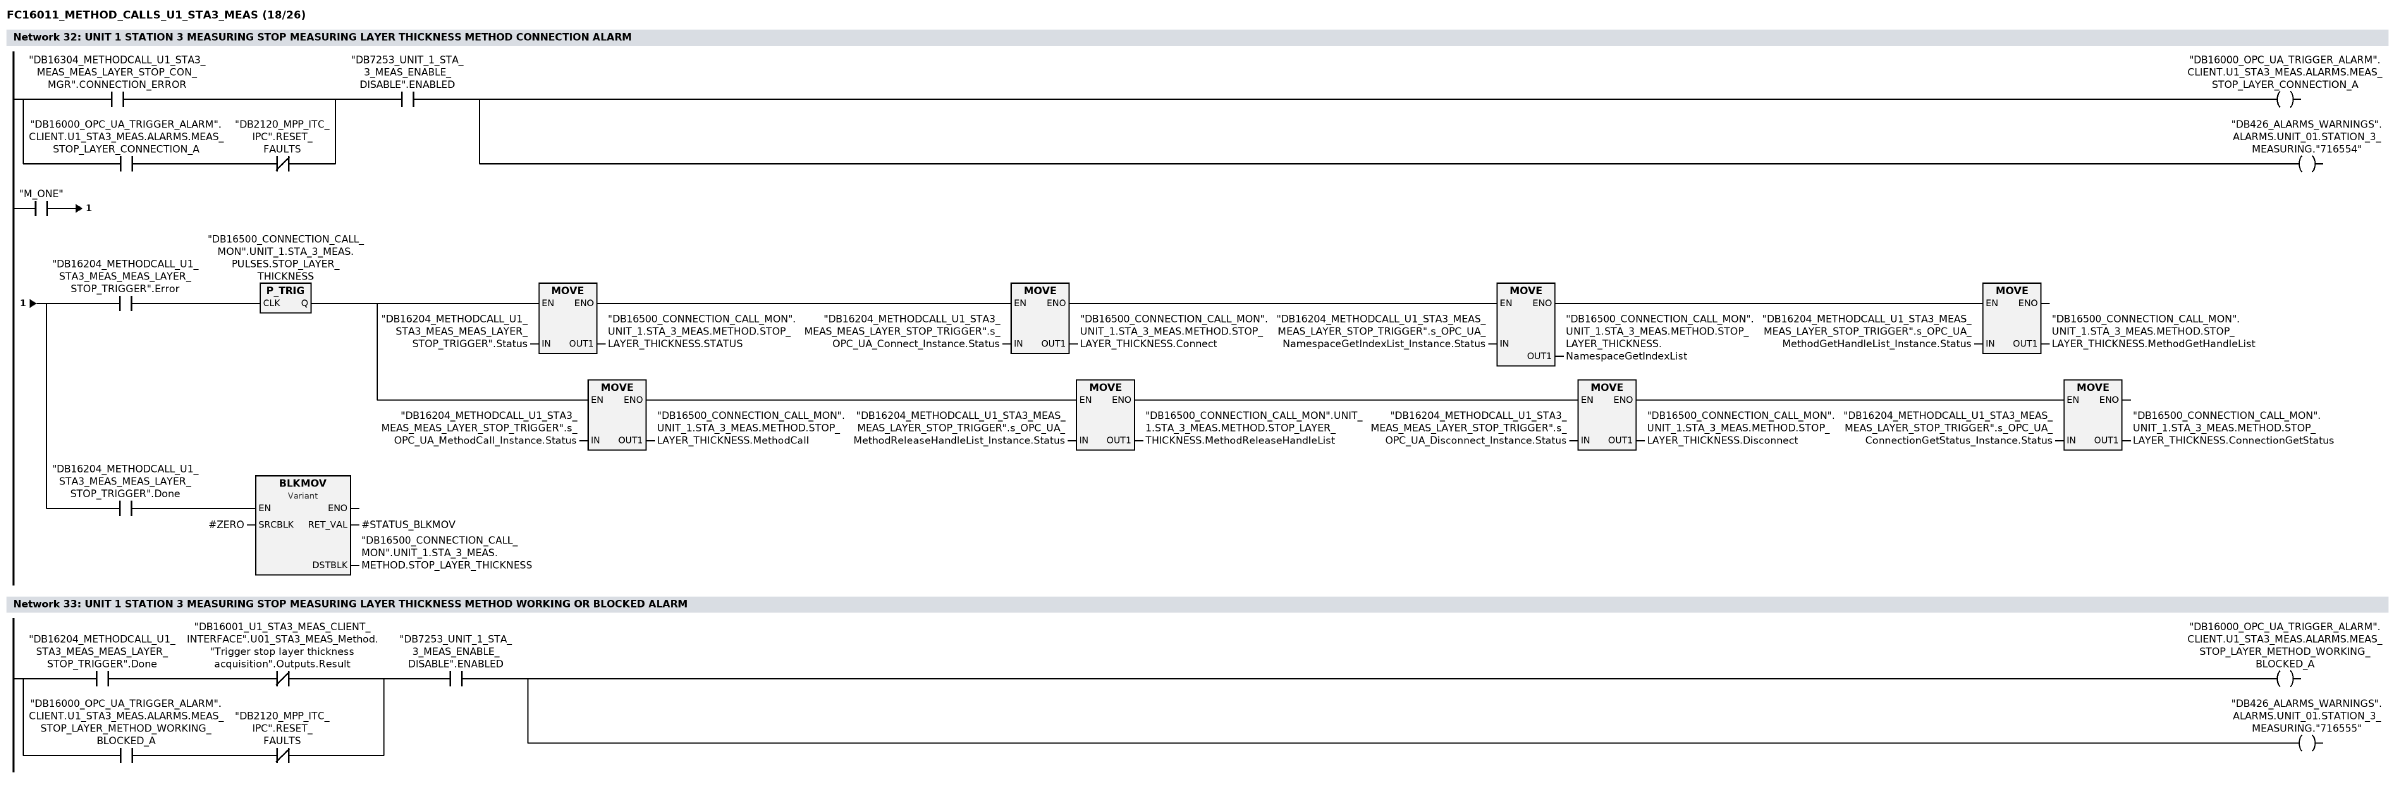
   RUNG wire#powerrail
      Contact( "DB16304_METHODCALL_U1_STA3_MEAS_MEAS_LAYER_STOP_CON_MGR".CONNECTION_ERROR )
      wire#w1
      Contact( "DB7253_UNIT_1_STA_3_MEAS_ENABLE_DISABLE".ENABLED )
      wire#w2
      Coil( "DB16000_OPC_UA_TRIGGER_ALARM".CLIENT.U1_STA3_MEAS.ALARMS.MEAS_STOP_LAYER_CONNECTION_A )
   END_RUNG
   RUNG wire#powerrail
      Contact( "DB16000_OPC_UA_TRIGGER_ALARM".CLIENT.U1_STA3_MEAS.ALARMS.MEAS_STOP_LAYER_CONNECTION_A )
      I_Contact( "DB2120_MPP_ITC_IPC".RESET_FAULTS )
   END_RUNG wire#w1
   RUNG wire#w2
      Coil( "DB426_ALARMS_WARNINGS".ALARMS.UNIT_01.STATION_3_MEASURING."716554" )
   END_RUNG
   RUNG wire#powerrail
      Contact( "M_ONE" )
      wire#w3
      Contact( "DB16204_METHODCALL_U1_STA3_MEAS_MEAS_LAYER_STOP_TRIGGER".Error )
      P_Trig( "DB16500_CONNECTION_CALL_MON".UNIT_1.STA_3_MEAS.PULSES.STOP_LAYER_THICKNESS )
      wire#w4
      Move(in := "DB16204_METHODCALL_U1_STA3_MEAS_MEAS_LAYER_STOP_TRIGGER".Status, out1 => "DB16500_CONNECTION_CALL_MON".UNIT_1.STA_3_MEAS.METHOD.STOP_LAYER_THICKNESS.STATUS)
      Move(in := "DB16204_METHODCALL_U1_STA3_MEAS_MEAS_LAYER_STOP_TRIGGER".s_OPC_UA_Connect_Instance.Status, out1 => "DB16500_CONNECTION_CALL_MON".UNIT_1.STA_3_MEAS.METHOD.STOP_LAYER_THICKNESS.Connect)
      Move(in := "DB16204_METHODCALL_U1_STA3_MEAS_MEAS_LAYER_STOP_TRIGGER".s_OPC_UA_NamespaceGetIndexList_Instance.Status, out1 => "DB16500_CONNECTION_CALL_MON".UNIT_1.STA_3_MEAS.METHOD.STOP_LAYER_THICKNESS.NamespaceGetIndexList)
      Move(in := "DB16204_METHODCALL_U1_STA3_MEAS_MEAS_LAYER_STOP_TRIGGER".s_OPC_UA_MethodGetHandleList_Instance.Status, out1 => "DB16500_CONNECTION_CALL_MON".UNIT_1.STA_3_MEAS.METHOD.STOP_LAYER_THICKNESS.MethodGetHandleList)
   END_RUNG
   RUNG wire#w4
      Move(in := "DB16204_METHODCALL_U1_STA3_MEAS_MEAS_LAYER_STOP_TRIGGER".s_OPC_UA_MethodCall_Instance.Status, out1 => "DB16500_CONNECTION_CALL_MON".UNIT_1.STA_3_MEAS.METHOD.STOP_LAYER_THICKNESS.MethodCall)
      Move(in := "DB16204_METHODCALL_U1_STA3_MEAS_MEAS_LAYER_STOP_TRIGGER".s_OPC_UA_MethodReleaseHandleList_Instance.Status, out1 => "DB16500_CONNECTION_CALL_MON".UNIT_1.STA_3_MEAS.METHOD.STOP_LAYER_THICKNESS.MethodReleaseHandleList)
      Move(in := "DB16204_METHODCALL_U1_STA3_MEAS_MEAS_LAYER_STOP_TRIGGER".s_OPC_UA_Disconnect_Instance.Status, out1 => "DB16500_CONNECTION_CALL_MON".UNIT_1.STA_3_MEAS.METHOD.STOP_LAYER_THICKNESS.Disconnect)
      Move(in := "DB16204_METHODCALL_U1_STA3_MEAS_MEAS_LAYER_STOP_TRIGGER".s_OPC_UA_ConnectionGetStatus_Instance.Status, out1 => "DB16500_CONNECTION_CALL_MON".UNIT_1.STA_3_MEAS.METHOD.STOP_LAYER_THICKNESS.ConnectionGetStatus)
   END_RUNG
   RUNG wire#w3
      Contact( "DB16204_METHODCALL_U1_STA3_MEAS_MEAS_LAYER_STOP_TRIGGER".Done )
      { S7_Templates := "blk_type := Variant" } BLKMOV(SRCBLK := #ZERO, RET_VAL => #STATUS_BLKMOV, DSTBLK => "DB16500_CONNECTION_CALL_MON".UNIT_1.STA_3_MEAS.METHOD.STOP_LAYER_THICKNESS)
   END_RUNG
   // the same network as SCL:
   "DB16000_OPC_UA_TRIGGER_ALARM".CLIENT.U1_STA3_MEAS.ALARMS.MEAS_STOP_LAYER_CONNECTION_A := ("DB16304_METHODCALL_U1_STA3_MEAS_MEAS_LAYER_STOP_CON_MGR".CONNECTION_ERROR OR ("DB16000_OPC_UA_TRIGGER_ALARM".CLIENT.U1_STA3_MEAS.ALARMS.MEAS_STOP_LAYER_CONNECTION_A AND NOT "DB2120_MPP_ITC_IPC".RESET_FAULTS)) AND "DB7253_UNIT_1_STA_3_MEAS_ENABLE_DISABLE".ENABLED;
   "DB426_ALARMS_WARNINGS".ALARMS.UNIT_01.STATION_3_MEASURING."716554" := "DB16000_OPC_UA_TRIGGER_ALARM".CLIENT.U1_STA3_MEAS.ALARMS.MEAS_STOP_LAYER_CONNECTION_A;
   #_w1 := "M_ONE" AND "DB16204_METHODCALL_U1_STA3_MEAS_MEAS_LAYER_STOP_TRIGGER".Error;
   #_w2 := #_w1 AND NOT "DB16500_CONNECTION_CALL_MON".UNIT_1.STA_3_MEAS.PULSES.STOP_LAYER_THICKNESS;   // rising edge
   "DB16500_CONNECTION_CALL_MON".UNIT_1.STA_3_MEAS.PULSES.STOP_LAYER_THICKNESS := #_w1;
   IF #_w2 THEN
       "DB16500_CONNECTION_CALL_MON".UNIT_1.STA_3_MEAS.METHOD.STOP_LAYER_THICKNESS.STATUS := "DB16204_METHODCALL_U1_STA3_MEAS_MEAS_LAYER_STOP_TRIGGER".Status;
       "DB16500_CONNECTION_CALL_MON".UNIT_1.STA_3_MEAS.METHOD.STOP_LAYER_THICKNESS.Connect := "DB16204_METHODCALL_U1_STA3_MEAS_MEAS_LAYER_STOP_TRIGGER".s_OPC_UA_Connect_Instance.Status;
       "DB16500_CONNECTION_CALL_MON".UNIT_1.STA_3_MEAS.METHOD.STOP_LAYER_THICKNESS.NamespaceGetIndexList := "DB16204_METHODCALL_U1_STA3_MEAS_MEAS_LAYER_STOP_TRIGGER".s_OPC_UA_NamespaceGetIndexList_Instance.Status;
       "DB16500_CONNECTION_CALL_MON".UNIT_1.STA_3_MEAS.METHOD.STOP_LAYER_THICKNESS.MethodGetHandleList := "DB16204_METHODCALL_U1_STA3_MEAS_MEAS_LAYER_STOP_TRIGGER".s_OPC_UA_MethodGetHandleList_Instance.Status;
       "DB16500_CONNECTION_CALL_MON".UNIT_1.STA_3_MEAS.METHOD.STOP_LAYER_THICKNESS.MethodCall := "DB16204_METHODCALL_U1_STA3_MEAS_MEAS_LAYER_STOP_TRIGGER".s_OPC_UA_MethodCall_Instance.Status;
       "DB16500_CONNECTION_CALL_MON".UNIT_1.STA_3_MEAS.METHOD.STOP_LAYER_THICKNESS.MethodReleaseHandleList := "DB16204_METHODCALL_U1_STA3_MEAS_MEAS_LAYER_STOP_TRIGGER".s_OPC_UA_MethodReleaseHandleList_Instance.Status;
       "DB16500_CONNECTION_CALL_MON".UNIT_1.STA_3_MEAS.METHOD.STOP_LAYER_THICKNESS.Disconnect := "DB16204_METHODCALL_U1_STA3_MEAS_MEAS_LAYER_STOP_TRIGGER".s_OPC_UA_Disconnect_Instance.Status;
       "DB16500_CONNECTION_CALL_MON".UNIT_1.STA_3_MEAS.METHOD.STOP_LAYER_THICKNESS.ConnectionGetStatus := "DB16204_METHODCALL_U1_STA3_MEAS_MEAS_LAYER_STOP_TRIGGER".s_OPC_UA_ConnectionGetStatus_Instance.Status;
   END_IF;
   IF "M_ONE" AND "DB16204_METHODCALL_U1_STA3_MEAS_MEAS_LAYER_STOP_TRIGGER".Done THEN
       #STATUS_BLKMOV := BLKMOV(SRCBLK := #ZERO,
                               DSTBLK => "DB16500_CONNECTION_CALL_MON".UNIT_1.STA_3_MEAS.METHOD.STOP_LAYER_THICKNESS);
   END_IF;
END_REGION

REGION Network 33: UNIT 1 STATION 3 MEASURING STOP MEASURING LAYER THICKNESS METHOD WORKING OR BLOCKED ALARM
   RUNG wire#powerrail
      Contact( "DB16204_METHODCALL_U1_STA3_MEAS_MEAS_LAYER_STOP_TRIGGER".Done )
      I_Contact( "DB16001_U1_STA3_MEAS_CLIENT_INTERFACE".U01_STA3_MEAS_Method."Trigger stop layer thickness acquisition".Outputs.Result )
      wire#w1
      Contact( "DB7253_UNIT_1_STA_3_MEAS_ENABLE_DISABLE".ENABLED )
      wire#w2
      Coil( "DB16000_OPC_UA_TRIGGER_ALARM".CLIENT.U1_STA3_MEAS.ALARMS.MEAS_STOP_LAYER_METHOD_WORKING_BLOCKED_A )
   END_RUNG
   RUNG wire#powerrail
      Contact( "DB16000_OPC_UA_TRIGGER_ALARM".CLIENT.U1_STA3_MEAS.ALARMS.MEAS_STOP_LAYER_METHOD_WORKING_BLOCKED_A )
      I_Contact( "DB2120_MPP_ITC_IPC".RESET_FAULTS )
   END_RUNG wire#w1
   RUNG wire#w2
      Coil( "DB426_ALARMS_WARNINGS".ALARMS.UNIT_01.STATION_3_MEASURING."716555" )
   END_RUNG
   // the same network as SCL:
   "DB16000_OPC_UA_TRIGGER_ALARM".CLIENT.U1_STA3_MEAS.ALARMS.MEAS_STOP_LAYER_METHOD_WORKING_BLOCKED_A := (("DB16204_METHODCALL_U1_STA3_MEAS_MEAS_LAYER_STOP_TRIGGER".Done AND NOT "DB16001_U1_STA3_MEAS_CLIENT_INTERFACE".U01_STA3_MEAS_Method."Trigger stop layer thickness acquisition".Outputs.Result) OR ("DB16000_OPC_UA_TRIGGER_ALARM".CLIENT.U1_STA3_MEAS.ALARMS.MEAS_STOP_LAYER_METHOD_WORKING_BLOCKED_A AND NOT "DB2120_MPP_ITC_IPC".RESET_FAULTS)) AND "DB7253_UNIT_1_STA_3_MEAS_ENABLE_DISABLE".ENABLED;
   "DB426_ALARMS_WARNINGS".ALARMS.UNIT_01.STATION_3_MEASURING."716555" := "DB16000_OPC_UA_TRIGGER_ALARM".CLIENT.U1_STA3_MEAS.ALARMS.MEAS_STOP_LAYER_METHOD_WORKING_BLOCKED_A;
END_REGION

REGION Network 34: UNIT 1 STATION 3 MEASURING CALIBRATING METHOD CONNECTION ALARM
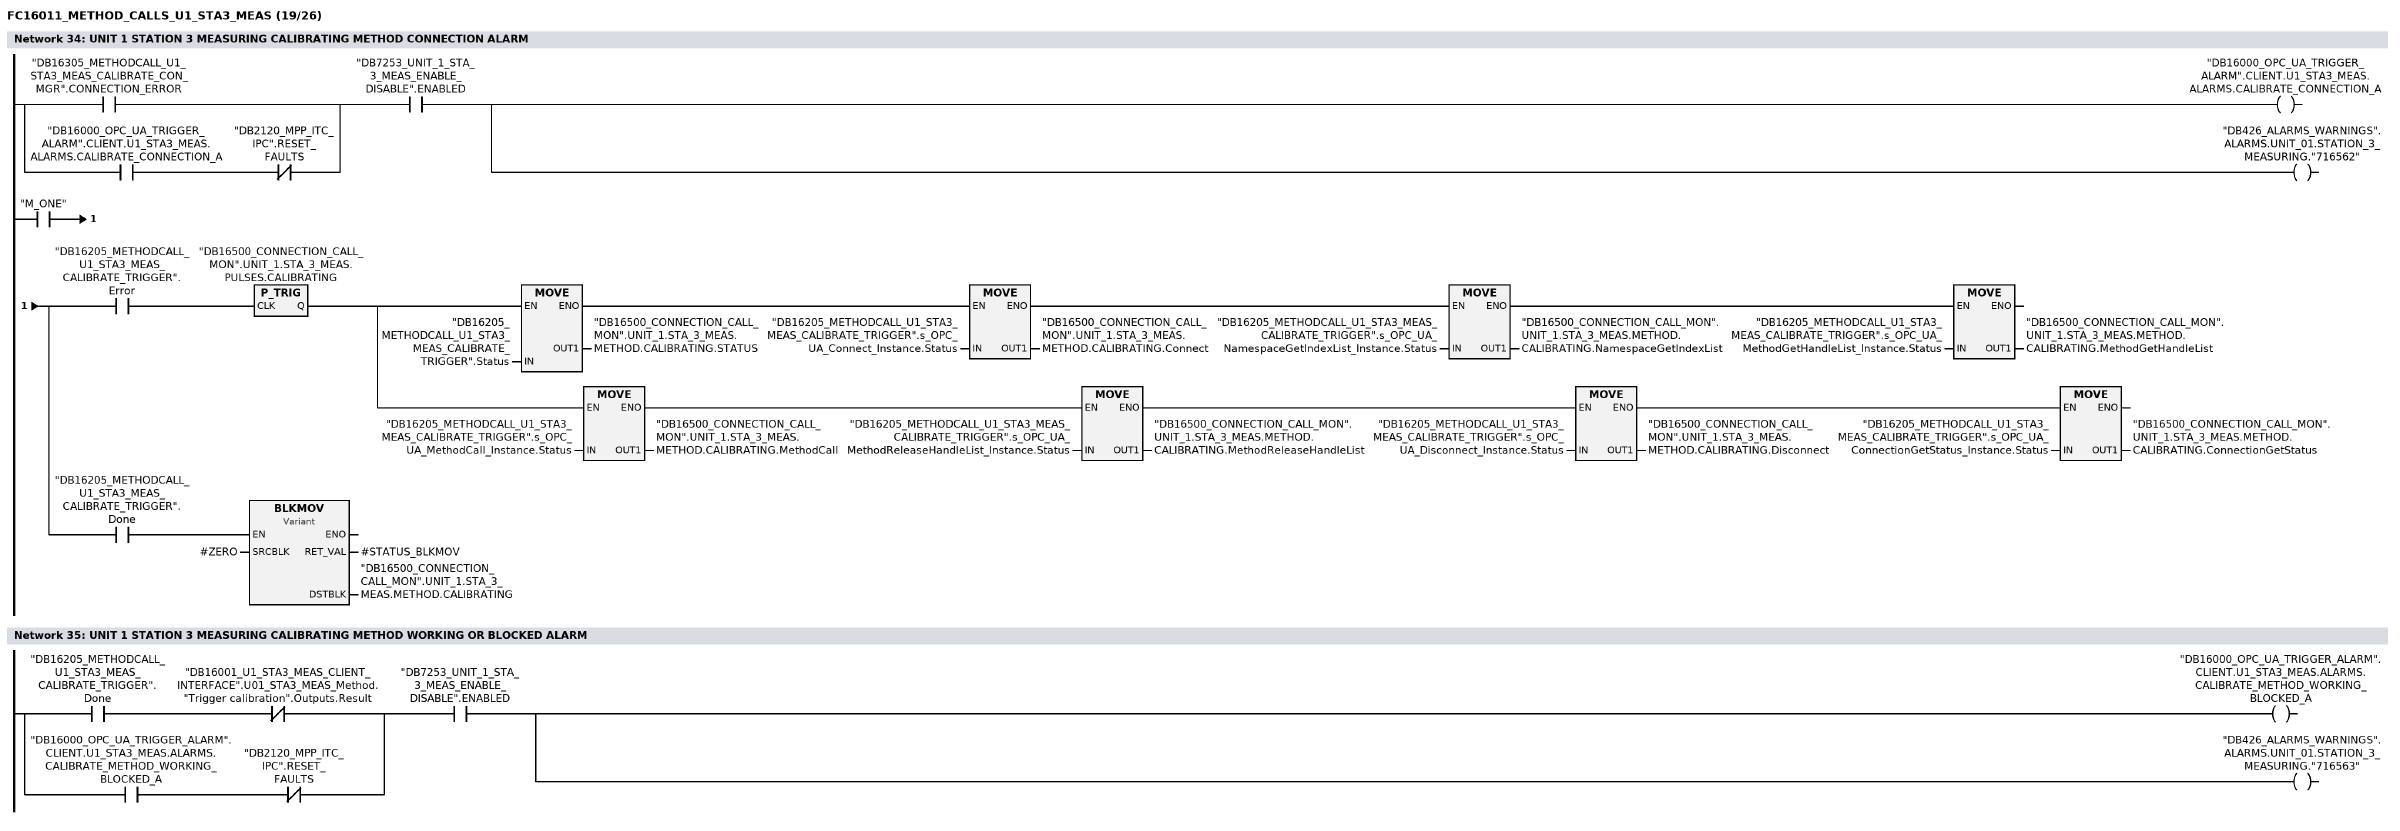
   RUNG wire#powerrail
      Contact( "DB16305_METHODCALL_U1_STA3_MEAS_CALIBRATE_CON_MGR".CONNECTION_ERROR )
      wire#w1
      Contact( "DB7253_UNIT_1_STA_3_MEAS_ENABLE_DISABLE".ENABLED )
      wire#w2
      Coil( "DB16000_OPC_UA_TRIGGER_ALARM".CLIENT.U1_STA3_MEAS.ALARMS.CALIBRATE_CONNECTION_A )
   END_RUNG
   RUNG wire#powerrail
      Contact( "DB16000_OPC_UA_TRIGGER_ALARM".CLIENT.U1_STA3_MEAS.ALARMS.CALIBRATE_CONNECTION_A )
      I_Contact( "DB2120_MPP_ITC_IPC".RESET_FAULTS )
   END_RUNG wire#w1
   RUNG wire#w2
      Coil( "DB426_ALARMS_WARNINGS".ALARMS.UNIT_01.STATION_3_MEASURING."716562" )
   END_RUNG
   RUNG wire#powerrail
      Contact( "M_ONE" )
      wire#w3
      Contact( "DB16205_METHODCALL_U1_STA3_MEAS_CALIBRATE_TRIGGER".Error )
      P_Trig( "DB16500_CONNECTION_CALL_MON".UNIT_1.STA_3_MEAS.PULSES.CALIBRATING )
      wire#w4
      Move(in := "DB16205_METHODCALL_U1_STA3_MEAS_CALIBRATE_TRIGGER".Status, out1 => "DB16500_CONNECTION_CALL_MON".UNIT_1.STA_3_MEAS.METHOD.CALIBRATING.STATUS)
      Move(in := "DB16205_METHODCALL_U1_STA3_MEAS_CALIBRATE_TRIGGER".s_OPC_UA_Connect_Instance.Status, out1 => "DB16500_CONNECTION_CALL_MON".UNIT_1.STA_3_MEAS.METHOD.CALIBRATING.Connect)
      Move(in := "DB16205_METHODCALL_U1_STA3_MEAS_CALIBRATE_TRIGGER".s_OPC_UA_NamespaceGetIndexList_Instance.Status, out1 => "DB16500_CONNECTION_CALL_MON".UNIT_1.STA_3_MEAS.METHOD.CALIBRATING.NamespaceGetIndexList)
      Move(in := "DB16205_METHODCALL_U1_STA3_MEAS_CALIBRATE_TRIGGER".s_OPC_UA_MethodGetHandleList_Instance.Status, out1 => "DB16500_CONNECTION_CALL_MON".UNIT_1.STA_3_MEAS.METHOD.CALIBRATING.MethodGetHandleList)
   END_RUNG
   RUNG wire#w4
      Move(in := "DB16205_METHODCALL_U1_STA3_MEAS_CALIBRATE_TRIGGER".s_OPC_UA_MethodCall_Instance.Status, out1 => "DB16500_CONNECTION_CALL_MON".UNIT_1.STA_3_MEAS.METHOD.CALIBRATING.MethodCall)
      Move(in := "DB16205_METHODCALL_U1_STA3_MEAS_CALIBRATE_TRIGGER".s_OPC_UA_MethodReleaseHandleList_Instance.Status, out1 => "DB16500_CONNECTION_CALL_MON".UNIT_1.STA_3_MEAS.METHOD.CALIBRATING.MethodReleaseHandleList)
      Move(in := "DB16205_METHODCALL_U1_STA3_MEAS_CALIBRATE_TRIGGER".s_OPC_UA_Disconnect_Instance.Status, out1 => "DB16500_CONNECTION_CALL_MON".UNIT_1.STA_3_MEAS.METHOD.CALIBRATING.Disconnect)
      Move(in := "DB16205_METHODCALL_U1_STA3_MEAS_CALIBRATE_TRIGGER".s_OPC_UA_ConnectionGetStatus_Instance.Status, out1 => "DB16500_CONNECTION_CALL_MON".UNIT_1.STA_3_MEAS.METHOD.CALIBRATING.ConnectionGetStatus)
   END_RUNG
   RUNG wire#w3
      Contact( "DB16205_METHODCALL_U1_STA3_MEAS_CALIBRATE_TRIGGER".Done )
      { S7_Templates := "blk_type := Variant" } BLKMOV(SRCBLK := #ZERO, RET_VAL => #STATUS_BLKMOV, DSTBLK => "DB16500_CONNECTION_CALL_MON".UNIT_1.STA_3_MEAS.METHOD.CALIBRATING)
   END_RUNG
   // the same network as SCL:
   "DB16000_OPC_UA_TRIGGER_ALARM".CLIENT.U1_STA3_MEAS.ALARMS.CALIBRATE_CONNECTION_A := ("DB16305_METHODCALL_U1_STA3_MEAS_CALIBRATE_CON_MGR".CONNECTION_ERROR OR ("DB16000_OPC_UA_TRIGGER_ALARM".CLIENT.U1_STA3_MEAS.ALARMS.CALIBRATE_CONNECTION_A AND NOT "DB2120_MPP_ITC_IPC".RESET_FAULTS)) AND "DB7253_UNIT_1_STA_3_MEAS_ENABLE_DISABLE".ENABLED;
   "DB426_ALARMS_WARNINGS".ALARMS.UNIT_01.STATION_3_MEASURING."716562" := "DB16000_OPC_UA_TRIGGER_ALARM".CLIENT.U1_STA3_MEAS.ALARMS.CALIBRATE_CONNECTION_A;
   #_w1 := "M_ONE" AND "DB16205_METHODCALL_U1_STA3_MEAS_CALIBRATE_TRIGGER".Error;
   #_w2 := #_w1 AND NOT "DB16500_CONNECTION_CALL_MON".UNIT_1.STA_3_MEAS.PULSES.CALIBRATING;   // rising edge
   "DB16500_CONNECTION_CALL_MON".UNIT_1.STA_3_MEAS.PULSES.CALIBRATING := #_w1;
   IF #_w2 THEN
       "DB16500_CONNECTION_CALL_MON".UNIT_1.STA_3_MEAS.METHOD.CALIBRATING.STATUS := "DB16205_METHODCALL_U1_STA3_MEAS_CALIBRATE_TRIGGER".Status;
       "DB16500_CONNECTION_CALL_MON".UNIT_1.STA_3_MEAS.METHOD.CALIBRATING.Connect := "DB16205_METHODCALL_U1_STA3_MEAS_CALIBRATE_TRIGGER".s_OPC_UA_Connect_Instance.Status;
       "DB16500_CONNECTION_CALL_MON".UNIT_1.STA_3_MEAS.METHOD.CALIBRATING.NamespaceGetIndexList := "DB16205_METHODCALL_U1_STA3_MEAS_CALIBRATE_TRIGGER".s_OPC_UA_NamespaceGetIndexList_Instance.Status;
       "DB16500_CONNECTION_CALL_MON".UNIT_1.STA_3_MEAS.METHOD.CALIBRATING.MethodGetHandleList := "DB16205_METHODCALL_U1_STA3_MEAS_CALIBRATE_TRIGGER".s_OPC_UA_MethodGetHandleList_Instance.Status;
       "DB16500_CONNECTION_CALL_MON".UNIT_1.STA_3_MEAS.METHOD.CALIBRATING.MethodCall := "DB16205_METHODCALL_U1_STA3_MEAS_CALIBRATE_TRIGGER".s_OPC_UA_MethodCall_Instance.Status;
       "DB16500_CONNECTION_CALL_MON".UNIT_1.STA_3_MEAS.METHOD.CALIBRATING.MethodReleaseHandleList := "DB16205_METHODCALL_U1_STA3_MEAS_CALIBRATE_TRIGGER".s_OPC_UA_MethodReleaseHandleList_Instance.Status;
       "DB16500_CONNECTION_CALL_MON".UNIT_1.STA_3_MEAS.METHOD.CALIBRATING.Disconnect := "DB16205_METHODCALL_U1_STA3_MEAS_CALIBRATE_TRIGGER".s_OPC_UA_Disconnect_Instance.Status;
       "DB16500_CONNECTION_CALL_MON".UNIT_1.STA_3_MEAS.METHOD.CALIBRATING.ConnectionGetStatus := "DB16205_METHODCALL_U1_STA3_MEAS_CALIBRATE_TRIGGER".s_OPC_UA_ConnectionGetStatus_Instance.Status;
   END_IF;
   IF "M_ONE" AND "DB16205_METHODCALL_U1_STA3_MEAS_CALIBRATE_TRIGGER".Done THEN
       #STATUS_BLKMOV := BLKMOV(SRCBLK := #ZERO,
                               DSTBLK => "DB16500_CONNECTION_CALL_MON".UNIT_1.STA_3_MEAS.METHOD.CALIBRATING);
   END_IF;
END_REGION

REGION Network 35: UNIT 1 STATION 3 MEASURING CALIBRATING METHOD WORKING OR BLOCKED ALARM
   RUNG wire#powerrail
      Contact( "DB16205_METHODCALL_U1_STA3_MEAS_CALIBRATE_TRIGGER".Done )
      I_Contact( "DB16001_U1_STA3_MEAS_CLIENT_INTERFACE".U01_STA3_MEAS_Method."Trigger calibration".Outputs.Result )
      wire#w1
      Contact( "DB7253_UNIT_1_STA_3_MEAS_ENABLE_DISABLE".ENABLED )
      wire#w2
      Coil( "DB16000_OPC_UA_TRIGGER_ALARM".CLIENT.U1_STA3_MEAS.ALARMS.CALIBRATE_METHOD_WORKING_BLOCKED_A )
   END_RUNG
   RUNG wire#powerrail
      Contact( "DB16000_OPC_UA_TRIGGER_ALARM".CLIENT.U1_STA3_MEAS.ALARMS.CALIBRATE_METHOD_WORKING_BLOCKED_A )
      I_Contact( "DB2120_MPP_ITC_IPC".RESET_FAULTS )
   END_RUNG wire#w1
   RUNG wire#w2
      Coil( "DB426_ALARMS_WARNINGS".ALARMS.UNIT_01.STATION_3_MEASURING."716563" )
   END_RUNG
   // the same network as SCL:
   "DB16000_OPC_UA_TRIGGER_ALARM".CLIENT.U1_STA3_MEAS.ALARMS.CALIBRATE_METHOD_WORKING_BLOCKED_A := (("DB16205_METHODCALL_U1_STA3_MEAS_CALIBRATE_TRIGGER".Done AND NOT "DB16001_U1_STA3_MEAS_CLIENT_INTERFACE".U01_STA3_MEAS_Method."Trigger calibration".Outputs.Result) OR ("DB16000_OPC_UA_TRIGGER_ALARM".CLIENT.U1_STA3_MEAS.ALARMS.CALIBRATE_METHOD_WORKING_BLOCKED_A AND NOT "DB2120_MPP_ITC_IPC".RESET_FAULTS)) AND "DB7253_UNIT_1_STA_3_MEAS_ENABLE_DISABLE".ENABLED;
   "DB426_ALARMS_WARNINGS".ALARMS.UNIT_01.STATION_3_MEASURING."716563" := "DB16000_OPC_UA_TRIGGER_ALARM".CLIENT.U1_STA3_MEAS.ALARMS.CALIBRATE_METHOD_WORKING_BLOCKED_A;
END_REGION

